REGION Network 42: Step [1102] : JOB[11] Check QR & Vision before move
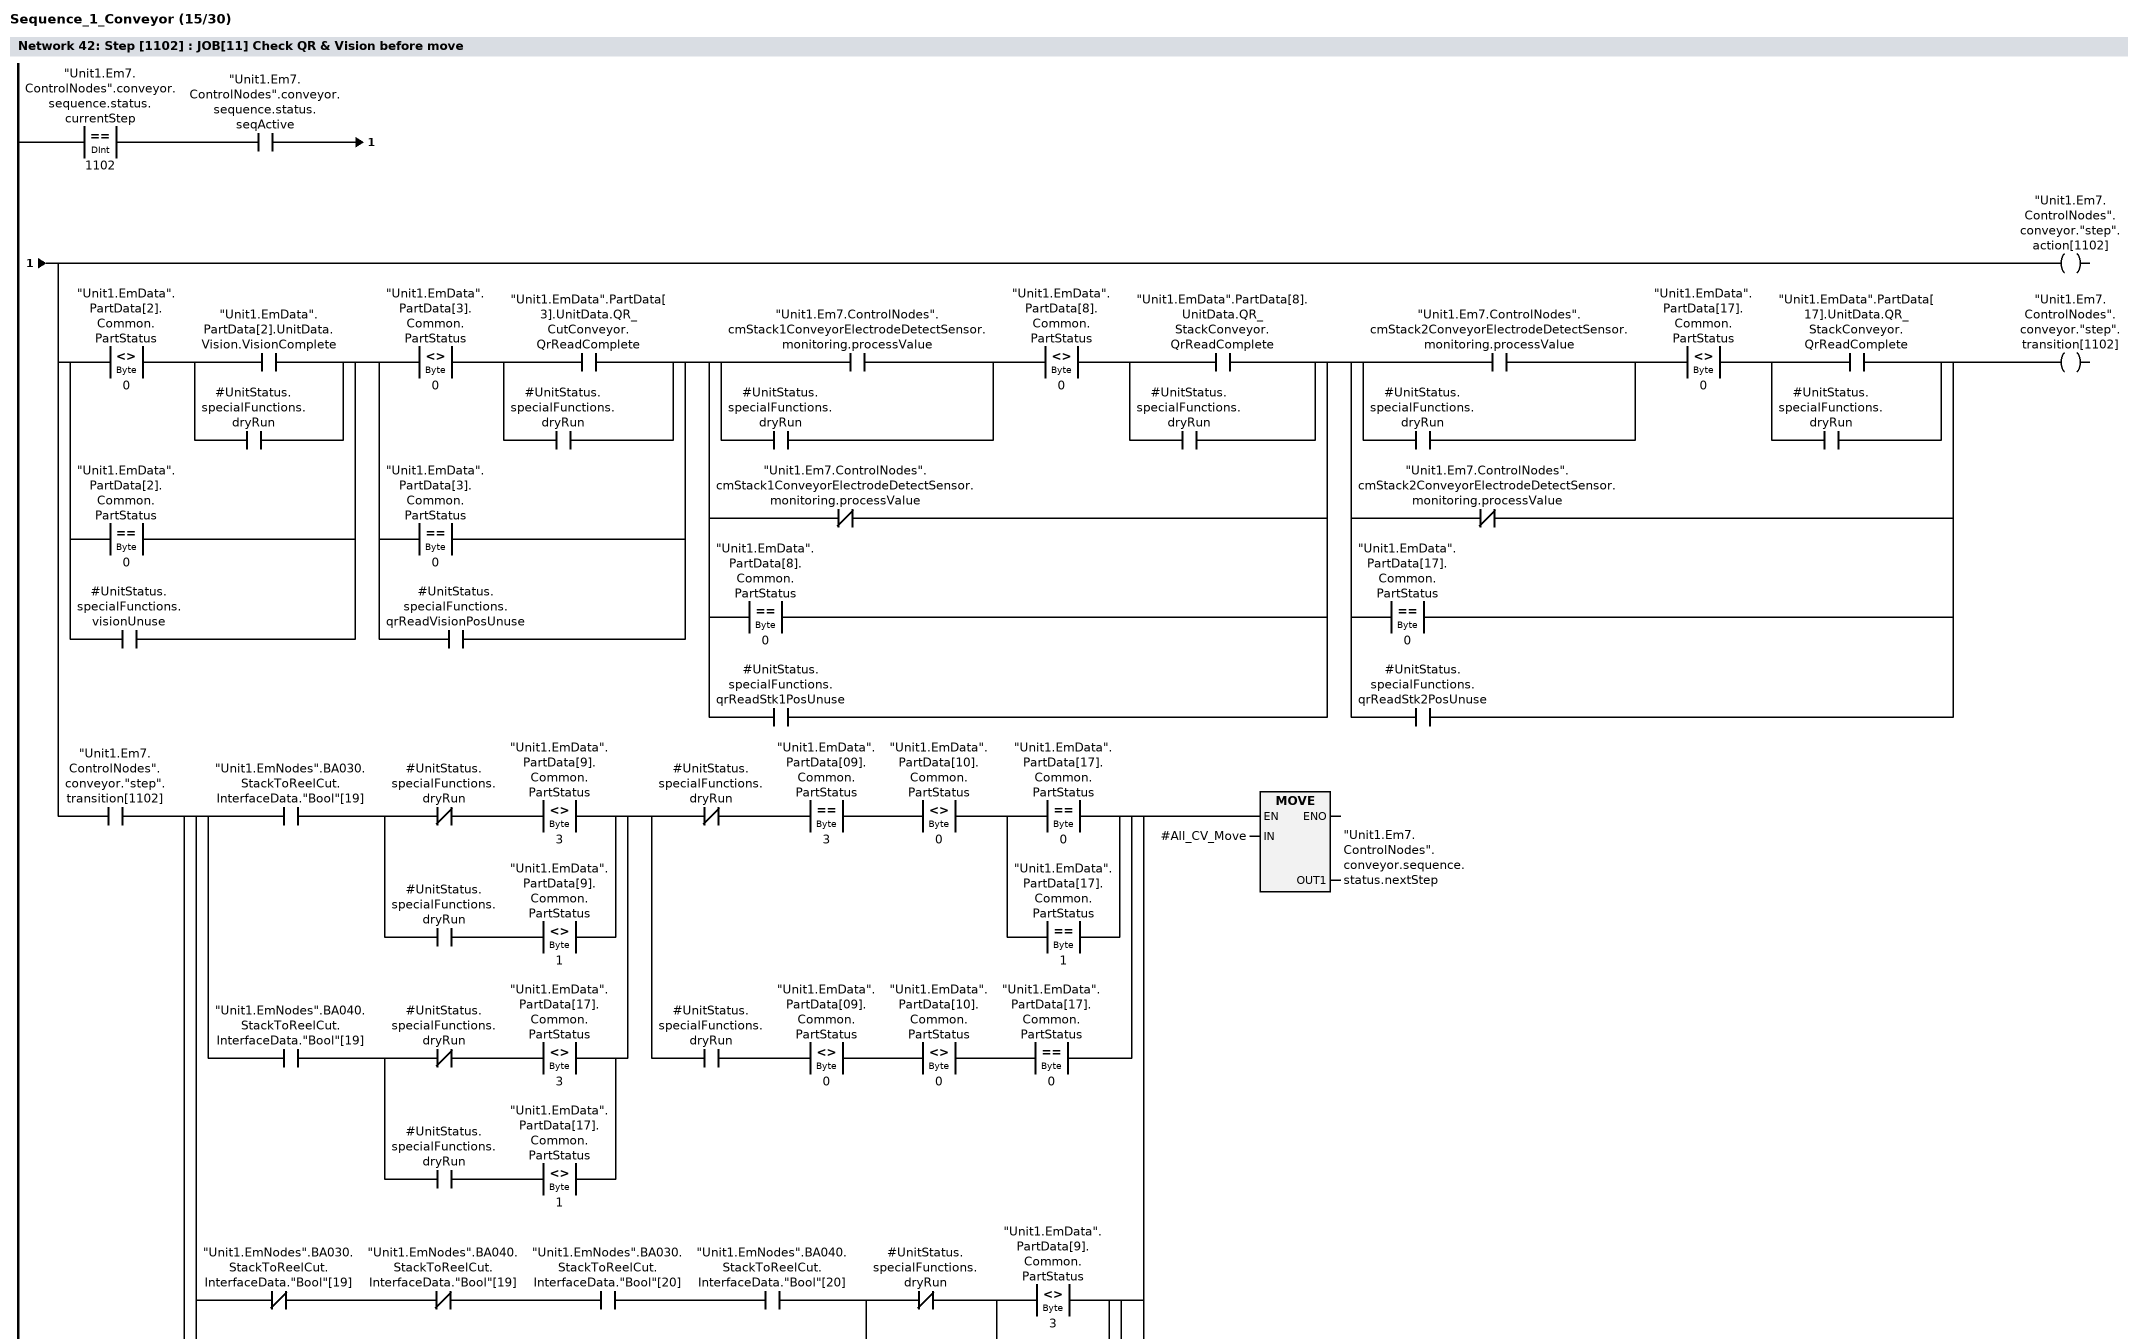
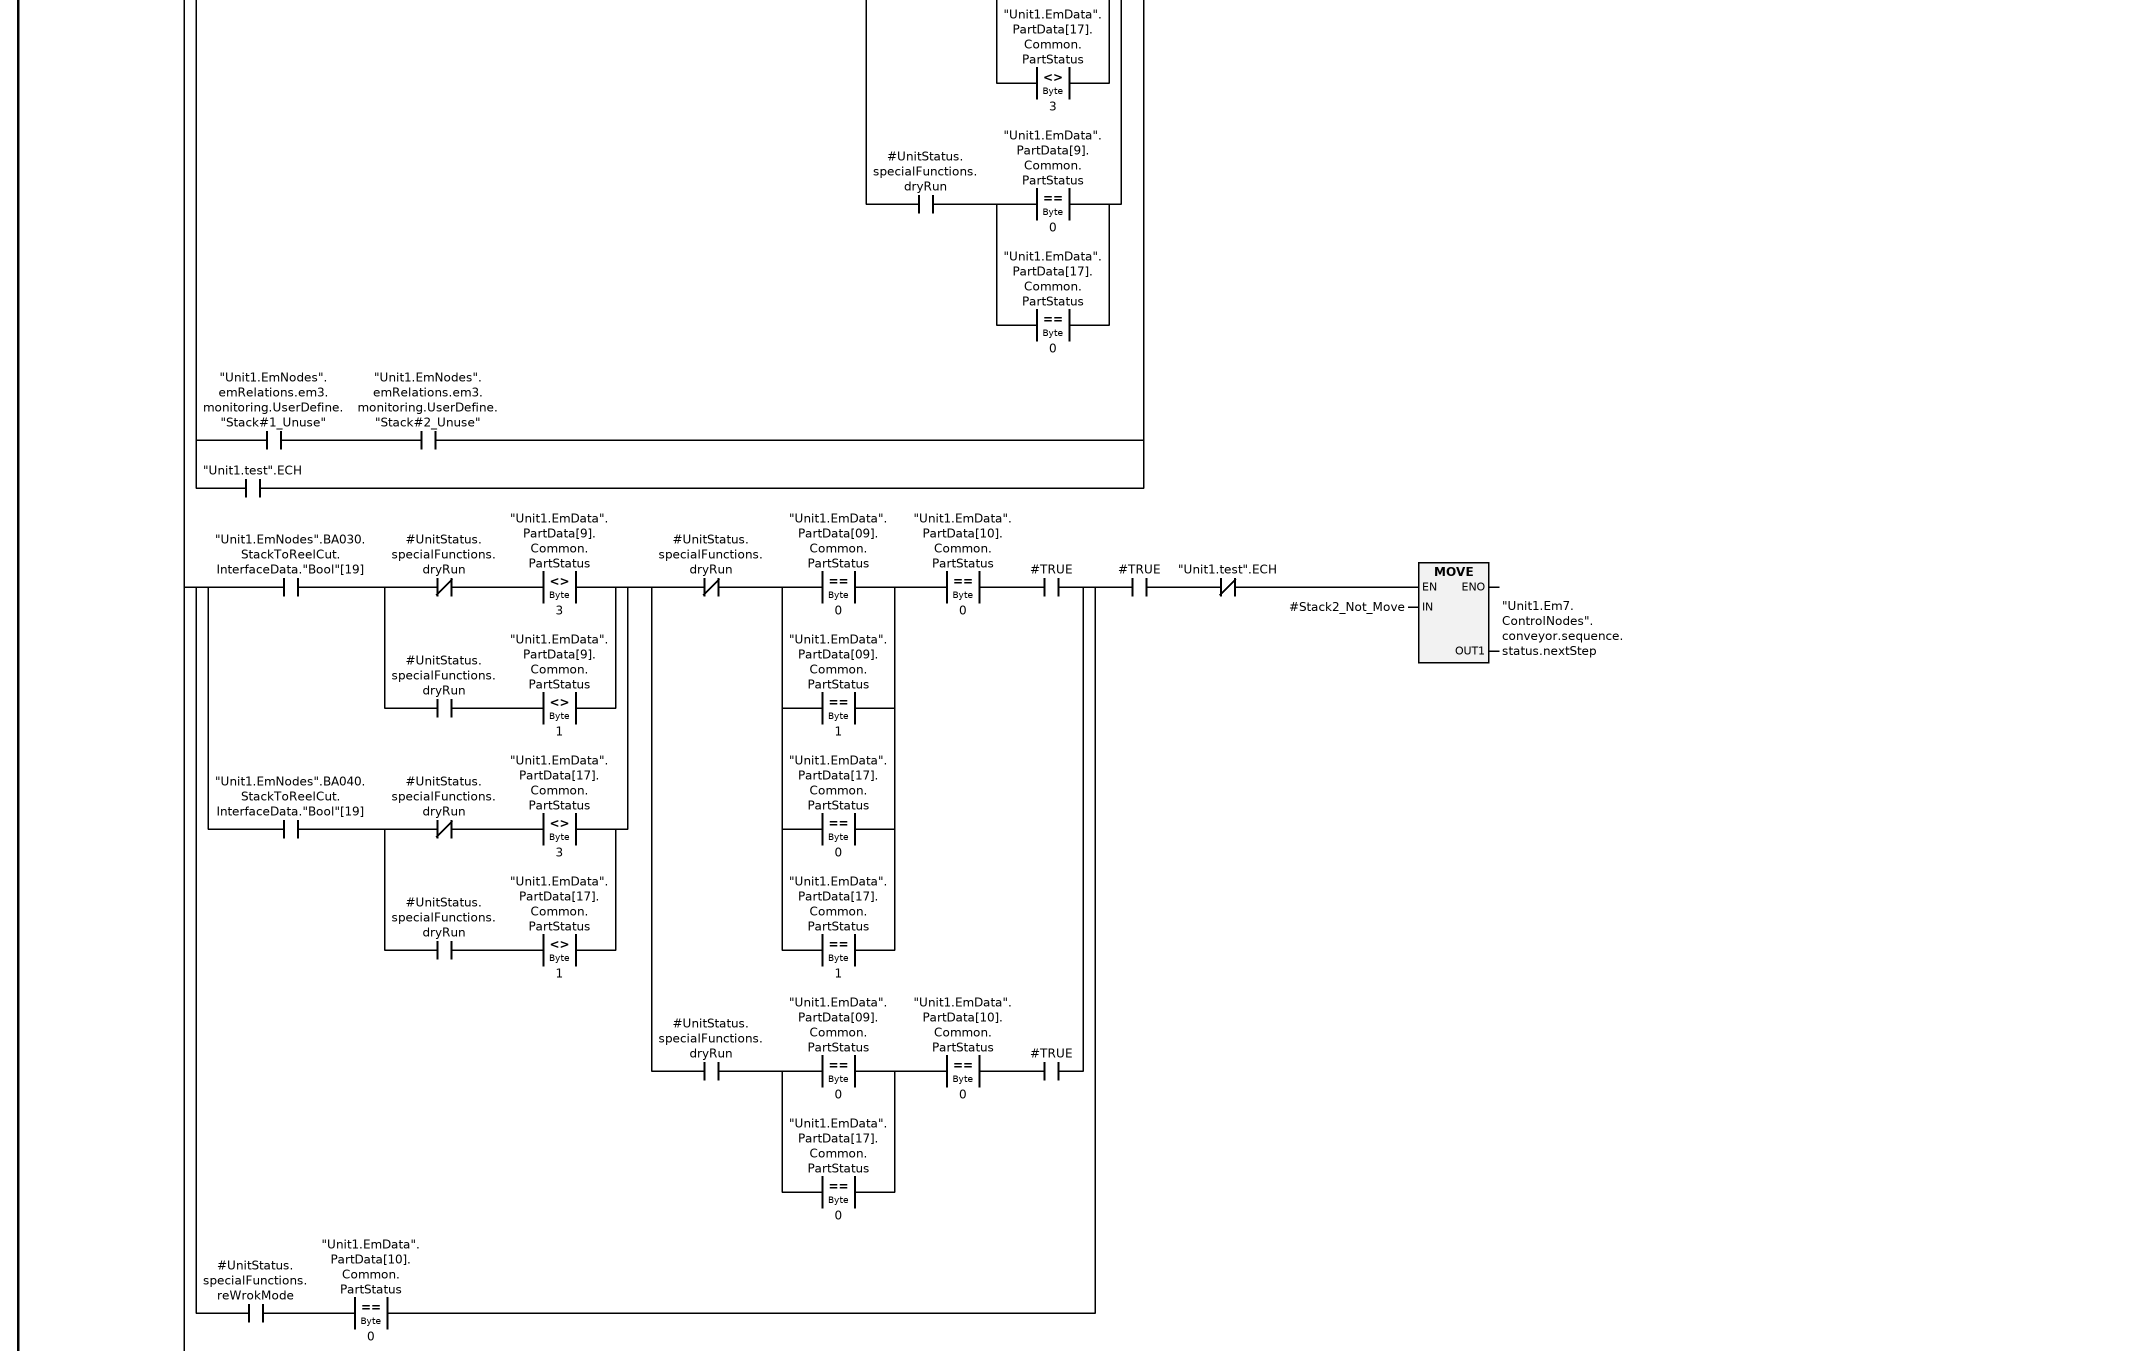
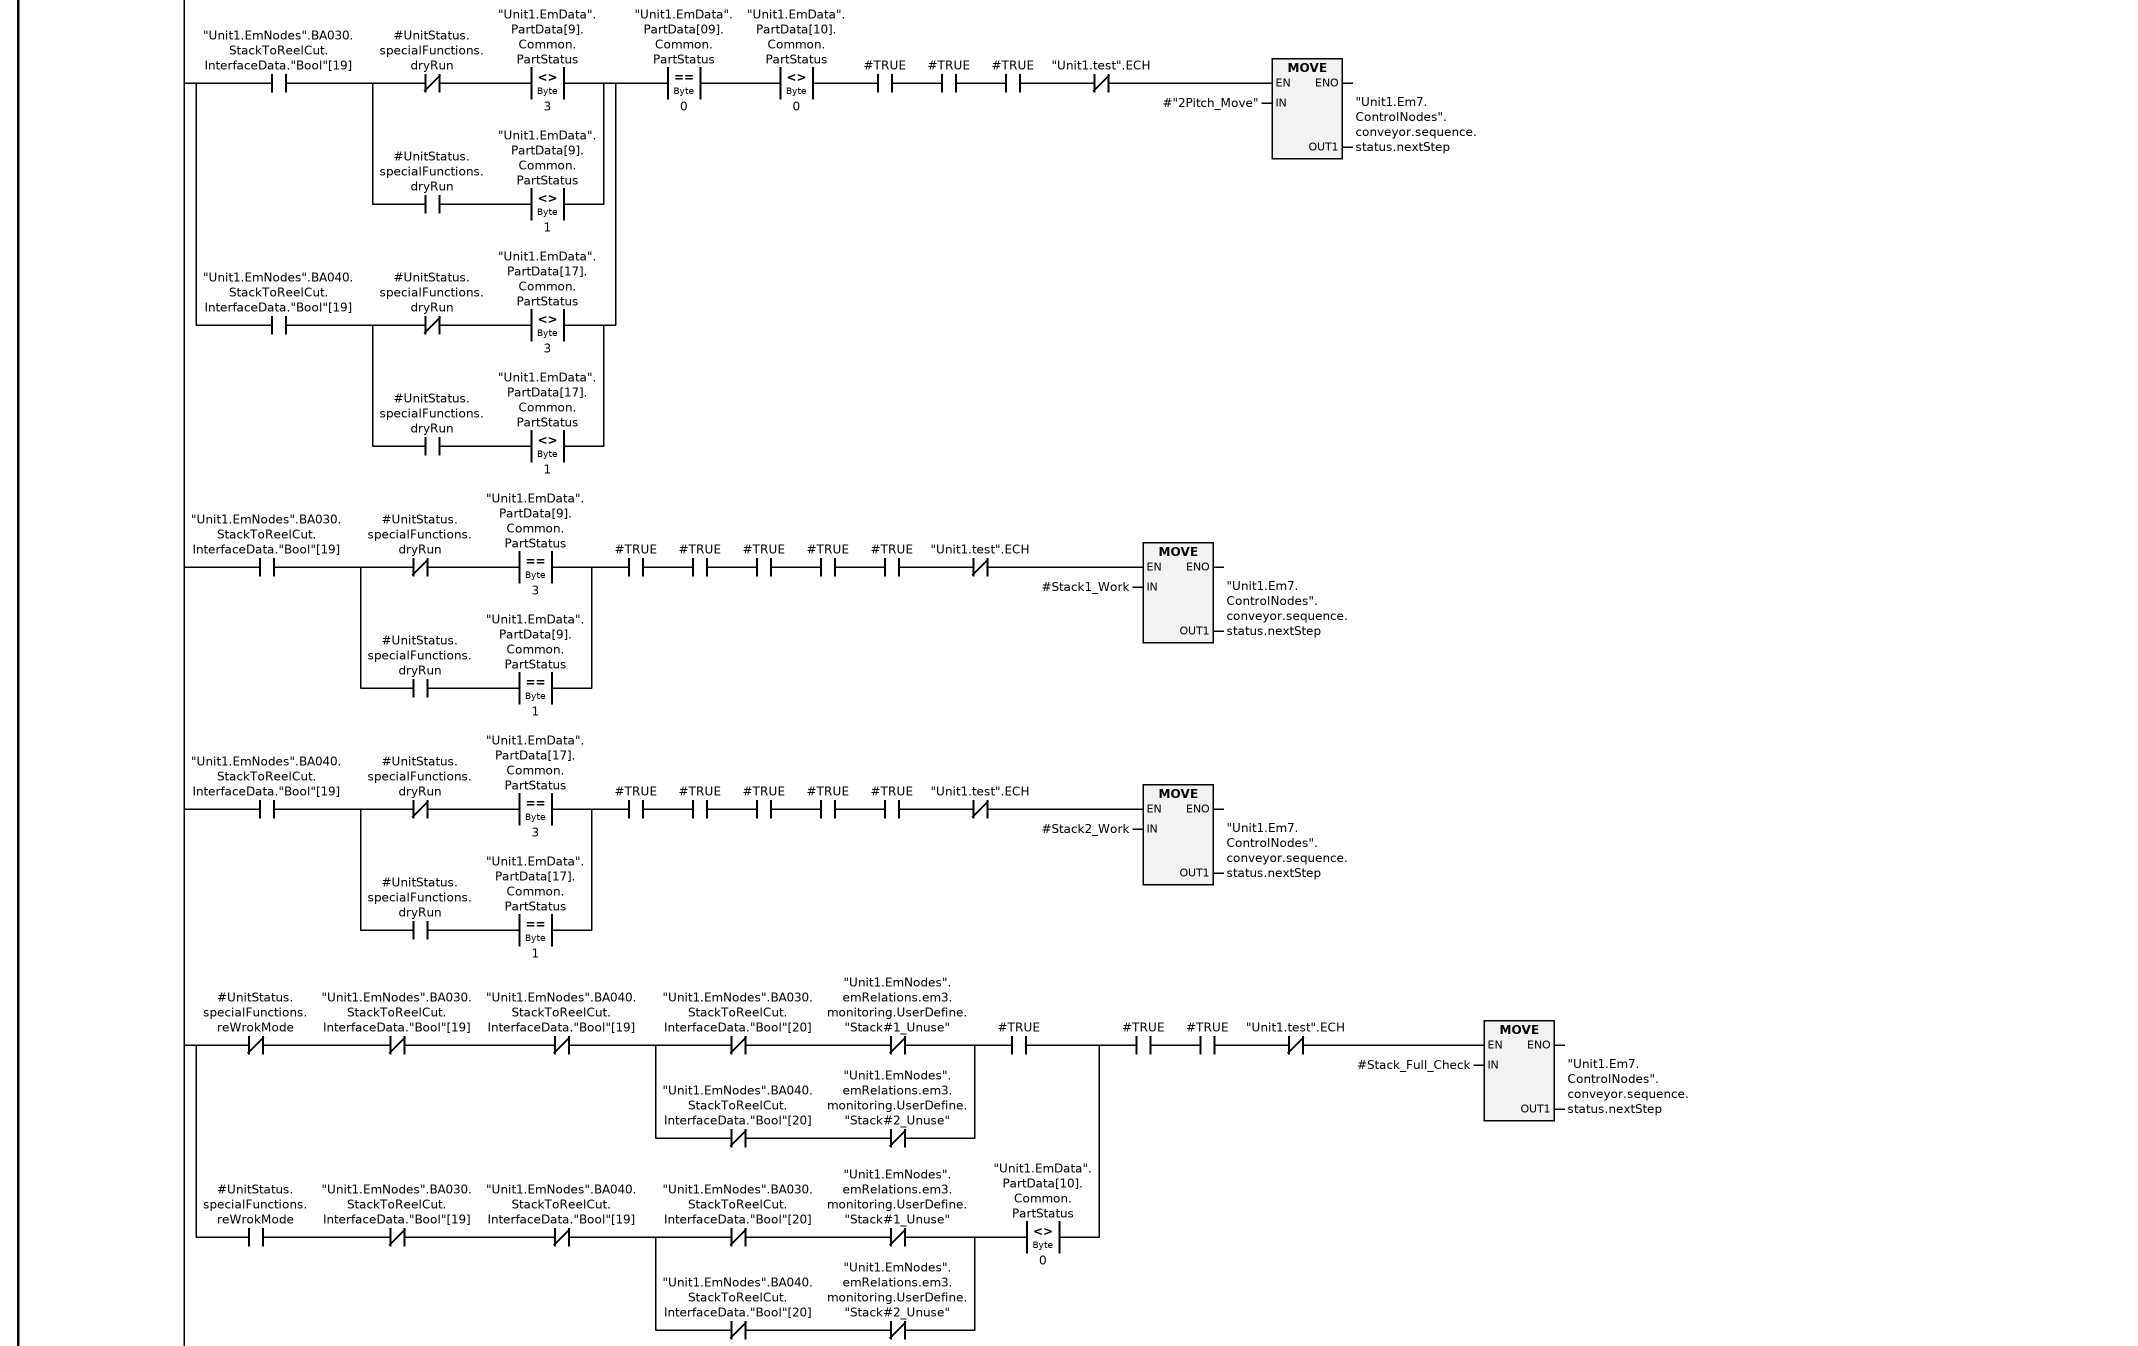
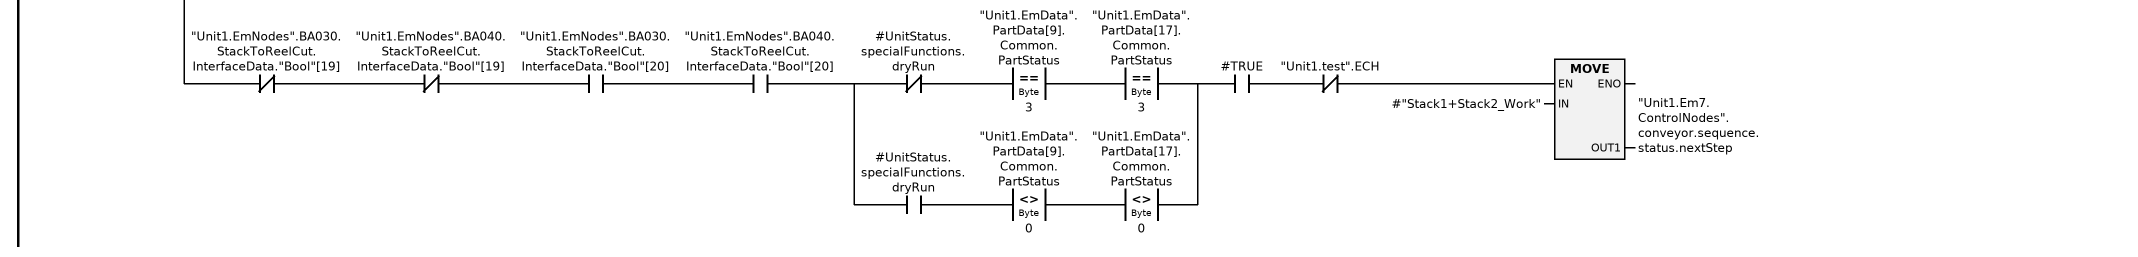
   RUNG wire#powerrail
      { S7_Templates := "SrcType := DInt" } EQ_Contact(in1 := "Unit1.Em7.ControlNodes".conveyor.sequence.status.currentStep, in2 := 1102)
      Contact( "Unit1.Em7.ControlNodes".conveyor.sequence.status.seqActive )
      wire#w1
      Coil( "Unit1.Em7.ControlNodes".conveyor."step".action[1102] )
   END_RUNG
   RUNG wire#w1
      { S7_Templates := "SrcType := Byte" } NE_Contact(in1 := "Unit1.EmData".PartData[2].Common.PartStatus, in2 := 0)
      wire#w2
      Contact( "Unit1.EmData".PartData[2].UnitData.Vision.VisionComplete )
      wire#w3
      { S7_Templates := "SrcType := Byte" } NE_Contact(in1 := "Unit1.EmData".PartData[3].Common.PartStatus, in2 := 0)
      wire#w4
      Contact( "Unit1.EmData".PartData[3].UnitData.QR_CutConveyor.QrReadComplete )
      wire#w5
      Contact( "Unit1.Em7.ControlNodes".cmStack1ConveyorElectrodeDetectSensor.monitoring.processValue )
      wire#w6
      { S7_Templates := "SrcType := Byte" } NE_Contact(in1 := "Unit1.EmData".PartData[8].Common.PartStatus, in2 := 0)
      wire#w7
      Contact( "Unit1.EmData".PartData[8].UnitData.QR_StackConveyor.QrReadComplete )
      wire#w8
      Contact( "Unit1.Em7.ControlNodes".cmStack2ConveyorElectrodeDetectSensor.monitoring.processValue )
      wire#w9
      { S7_Templates := "SrcType := Byte" } NE_Contact(in1 := "Unit1.EmData".PartData[17].Common.PartStatus, in2 := 0)
      wire#w10
      Contact( "Unit1.EmData".PartData[17].UnitData.QR_StackConveyor.QrReadComplete )
      wire#w11
      Coil( "Unit1.Em7.ControlNodes".conveyor."step".transition[1102] )
   END_RUNG
   RUNG wire#w2
      Contact( #UnitStatus.specialFunctions.dryRun )
   END_RUNG wire#w3
   RUNG wire#w1
      { S7_Templates := "SrcType := Byte" } EQ_Contact(in1 := "Unit1.EmData".PartData[2].Common.PartStatus, in2 := 0)
   END_RUNG wire#w3
   RUNG wire#w1
      Contact( #UnitStatus.specialFunctions.visionUnuse )
   END_RUNG wire#w3
   RUNG wire#w4
      Contact( #UnitStatus.specialFunctions.dryRun )
   END_RUNG wire#w5
   RUNG wire#w3
      { S7_Templates := "SrcType := Byte" } EQ_Contact(in1 := "Unit1.EmData".PartData[3].Common.PartStatus, in2 := 0)
   END_RUNG wire#w5
   RUNG wire#w3
      Contact( #UnitStatus.specialFunctions.qrReadVisionPosUnuse )
   END_RUNG wire#w5
   RUNG wire#w5
      Contact( #UnitStatus.specialFunctions.dryRun )
   END_RUNG wire#w6
   RUNG wire#w7
      Contact( #UnitStatus.specialFunctions.dryRun )
   END_RUNG wire#w8
   RUNG wire#w5
      I_Contact( "Unit1.Em7.ControlNodes".cmStack1ConveyorElectrodeDetectSensor.monitoring.processValue )
   END_RUNG wire#w8
   RUNG wire#w5
      { S7_Templates := "SrcType := Byte" } EQ_Contact(in1 := "Unit1.EmData".PartData[8].Common.PartStatus, in2 := 0)
   END_RUNG wire#w8
   RUNG wire#w5
      Contact( #UnitStatus.specialFunctions.qrReadStk1PosUnuse )
   END_RUNG wire#w8
   RUNG wire#w8
      Contact( #UnitStatus.specialFunctions.dryRun )
   END_RUNG wire#w9
   RUNG wire#w10
      Contact( #UnitStatus.specialFunctions.dryRun )
   END_RUNG wire#w11
   RUNG wire#w8
      I_Contact( "Unit1.Em7.ControlNodes".cmStack2ConveyorElectrodeDetectSensor.monitoring.processValue )
   END_RUNG wire#w11
   RUNG wire#w8
      { S7_Templates := "SrcType := Byte" } EQ_Contact(in1 := "Unit1.EmData".PartData[17].Common.PartStatus, in2 := 0)
   END_RUNG wire#w11
   RUNG wire#w8
      Contact( #UnitStatus.specialFunctions.qrReadStk2PosUnuse )
   END_RUNG wire#w11
   RUNG wire#w1
      Contact( "Unit1.Em7.ControlNodes".conveyor."step".transition[1102] )
      wire#w12
      Contact( "Unit1.EmNodes".BA030.StackToReelCut.InterfaceData."Bool"[19] )
      wire#w13
      I_Contact( #UnitStatus.specialFunctions.dryRun )
      { S7_Templates := "SrcType := Byte" } NE_Contact(in1 := "Unit1.EmData".PartData[9].Common.PartStatus, in2 := 3)
      wire#w14
      I_Contact( #UnitStatus.specialFunctions.dryRun )
      { S7_Templates := "SrcType := Byte" } EQ_Contact(in1 := "Unit1.EmData".PartData[09].Common.PartStatus, in2 := 3)
      { S7_Templates := "SrcType := Byte" } NE_Contact(in1 := "Unit1.EmData".PartData[10].Common.PartStatus, in2 := 0)
      wire#w16
      { S7_Templates := "SrcType := Byte" } EQ_Contact(in1 := "Unit1.EmData".PartData[17].Common.PartStatus, in2 := 0)
      wire#w17
      Move(in := #All_CV_Move, out1 => "Unit1.Em7.ControlNodes".conveyor.sequence.status.nextStep)
   END_RUNG
   RUNG wire#w13
      Contact( #UnitStatus.specialFunctions.dryRun )
      { S7_Templates := "SrcType := Byte" } NE_Contact(in1 := "Unit1.EmData".PartData[9].Common.PartStatus, in2 := 1)
   END_RUNG wire#w14
   RUNG wire#w12
      Contact( "Unit1.EmNodes".BA040.StackToReelCut.InterfaceData."Bool"[19] )
      wire#w15
      I_Contact( #UnitStatus.specialFunctions.dryRun )
      { S7_Templates := "SrcType := Byte" } NE_Contact(in1 := "Unit1.EmData".PartData[17].Common.PartStatus, in2 := 3)
   END_RUNG wire#w14
   RUNG wire#w15
      Contact( #UnitStatus.specialFunctions.dryRun )
      { S7_Templates := "SrcType := Byte" } NE_Contact(in1 := "Unit1.EmData".PartData[17].Common.PartStatus, in2 := 1)
   END_RUNG wire#w14
   RUNG wire#w16
      { S7_Templates := "SrcType := Byte" } EQ_Contact(in1 := "Unit1.EmData".PartData[17].Common.PartStatus, in2 := 1)
   END_RUNG wire#w17
   RUNG wire#w14
      Contact( #UnitStatus.specialFunctions.dryRun )
      { S7_Templates := "SrcType := Byte" } NE_Contact(in1 := "Unit1.EmData".PartData[09].Common.PartStatus, in2 := 0)
      { S7_Templates := "SrcType := Byte" } NE_Contact(in1 := "Unit1.EmData".PartData[10].Common.PartStatus, in2 := 0)
      { S7_Templates := "SrcType := Byte" } EQ_Contact(in1 := "Unit1.EmData".PartData[17].Common.PartStatus, in2 := 0)
   END_RUNG wire#w17
   RUNG wire#w12
      I_Contact( "Unit1.EmNodes".BA030.StackToReelCut.InterfaceData."Bool"[19] )
      I_Contact( "Unit1.EmNodes".BA040.StackToReelCut.InterfaceData."Bool"[19] )
      Contact( "Unit1.EmNodes".BA030.StackToReelCut.InterfaceData."Bool"[20] )
      Contact( "Unit1.EmNodes".BA040.StackToReelCut.InterfaceData."Bool"[20] )
      wire#w18
      I_Contact( #UnitStatus.specialFunctions.dryRun )
      wire#w19
      { S7_Templates := "SrcType := Byte" } NE_Contact(in1 := "Unit1.EmData".PartData[9].Common.PartStatus, in2 := 3)
   END_RUNG wire#w17
   RUNG wire#w19
      { S7_Templates := "SrcType := Byte" } NE_Contact(in1 := "Unit1.EmData".PartData[17].Common.PartStatus, in2 := 3)
   END_RUNG wire#w17
   RUNG wire#w18
      Contact( #UnitStatus.specialFunctions.dryRun )
      wire#w20
      { S7_Templates := "SrcType := Byte" } EQ_Contact(in1 := "Unit1.EmData".PartData[9].Common.PartStatus, in2 := 0)
   END_RUNG wire#w17
   RUNG wire#w20
      { S7_Templates := "SrcType := Byte" } EQ_Contact(in1 := "Unit1.EmData".PartData[17].Common.PartStatus, in2 := 0)
   END_RUNG wire#w17
   RUNG wire#w12
      Contact( "Unit1.EmNodes".emRelations.em3.monitoring.UserDefine."Stack#1_Unuse" )
      Contact( "Unit1.EmNodes".emRelations.em3.monitoring.UserDefine."Stack#2_Unuse" )
   END_RUNG wire#w17
   RUNG wire#w12
      Contact( "Unit1.test".ECH )
   END_RUNG wire#w17
   RUNG wire#w12
      Contact( "Unit1.EmNodes".BA030.StackToReelCut.InterfaceData."Bool"[19] )
      wire#w21
      I_Contact( #UnitStatus.specialFunctions.dryRun )
      { S7_Templates := "SrcType := Byte" } NE_Contact(in1 := "Unit1.EmData".PartData[9].Common.PartStatus, in2 := 3)
      wire#w22
      I_Contact( #UnitStatus.specialFunctions.dryRun )
      wire#w24
      { S7_Templates := "SrcType := Byte" } EQ_Contact(in1 := "Unit1.EmData".PartData[09].Common.PartStatus, in2 := 0)
      wire#w25
      { S7_Templates := "SrcType := Byte" } EQ_Contact(in1 := "Unit1.EmData".PartData[10].Common.PartStatus, in2 := 0)
      Contact( #TRUE )
      wire#w26
      Contact( #TRUE )
      I_Contact( "Unit1.test".ECH )
      Move(in := #Stack2_Not_Move, out1 => "Unit1.Em7.ControlNodes".conveyor.sequence.status.nextStep)
   END_RUNG
   RUNG wire#w21
      Contact( #UnitStatus.specialFunctions.dryRun )
      { S7_Templates := "SrcType := Byte" } NE_Contact(in1 := "Unit1.EmData".PartData[9].Common.PartStatus, in2 := 1)
   END_RUNG wire#w22
   RUNG wire#w12
      Contact( "Unit1.EmNodes".BA040.StackToReelCut.InterfaceData."Bool"[19] )
      wire#w23
      I_Contact( #UnitStatus.specialFunctions.dryRun )
      { S7_Templates := "SrcType := Byte" } NE_Contact(in1 := "Unit1.EmData".PartData[17].Common.PartStatus, in2 := 3)
   END_RUNG wire#w22
   RUNG wire#w23
      Contact( #UnitStatus.specialFunctions.dryRun )
      { S7_Templates := "SrcType := Byte" } NE_Contact(in1 := "Unit1.EmData".PartData[17].Common.PartStatus, in2 := 1)
   END_RUNG wire#w22
   RUNG wire#w24
      { S7_Templates := "SrcType := Byte" } EQ_Contact(in1 := "Unit1.EmData".PartData[09].Common.PartStatus, in2 := 1)
   END_RUNG wire#w25
   RUNG wire#w24
      { S7_Templates := "SrcType := Byte" } EQ_Contact(in1 := "Unit1.EmData".PartData[17].Common.PartStatus, in2 := 0)
   END_RUNG wire#w25
   RUNG wire#w24
      { S7_Templates := "SrcType := Byte" } EQ_Contact(in1 := "Unit1.EmData".PartData[17].Common.PartStatus, in2 := 1)
   END_RUNG wire#w25
   RUNG wire#w22
      Contact( #UnitStatus.specialFunctions.dryRun )
      wire#w27
      { S7_Templates := "SrcType := Byte" } EQ_Contact(in1 := "Unit1.EmData".PartData[09].Common.PartStatus, in2 := 0)
      wire#w28
      { S7_Templates := "SrcType := Byte" } EQ_Contact(in1 := "Unit1.EmData".PartData[10].Common.PartStatus, in2 := 0)
      Contact( #TRUE )
   END_RUNG wire#w26
   RUNG wire#w27
      { S7_Templates := "SrcType := Byte" } EQ_Contact(in1 := "Unit1.EmData".PartData[17].Common.PartStatus, in2 := 0)
   END_RUNG wire#w28
   RUNG wire#w12
      Contact( #UnitStatus.specialFunctions.reWrokMode )
      { S7_Templates := "SrcType := Byte" } EQ_Contact(in1 := "Unit1.EmData".PartData[10].Common.PartStatus, in2 := 0)
   END_RUNG wire#w26
   RUNG wire#w12
      Contact( "Unit1.EmNodes".BA030.StackToReelCut.InterfaceData."Bool"[19] )
      wire#w29
      I_Contact( #UnitStatus.specialFunctions.dryRun )
      { S7_Templates := "SrcType := Byte" } NE_Contact(in1 := "Unit1.EmData".PartData[9].Common.PartStatus, in2 := 3)
      wire#w30
      { S7_Templates := "SrcType := Byte" } EQ_Contact(in1 := "Unit1.EmData".PartData[09].Common.PartStatus, in2 := 0)
      { S7_Templates := "SrcType := Byte" } NE_Contact(in1 := "Unit1.EmData".PartData[10].Common.PartStatus, in2 := 0)
      Contact( #TRUE )
      Contact( #TRUE )
      Contact( #TRUE )
      I_Contact( "Unit1.test".ECH )
      Move(in := #"2Pitch_Move", out1 => "Unit1.Em7.ControlNodes".conveyor.sequence.status.nextStep)
   END_RUNG
   RUNG wire#w29
      Contact( #UnitStatus.specialFunctions.dryRun )
      { S7_Templates := "SrcType := Byte" } NE_Contact(in1 := "Unit1.EmData".PartData[9].Common.PartStatus, in2 := 1)
   END_RUNG wire#w30
   RUNG wire#w12
      Contact( "Unit1.EmNodes".BA040.StackToReelCut.InterfaceData."Bool"[19] )
      wire#w31
      I_Contact( #UnitStatus.specialFunctions.dryRun )
      { S7_Templates := "SrcType := Byte" } NE_Contact(in1 := "Unit1.EmData".PartData[17].Common.PartStatus, in2 := 3)
   END_RUNG wire#w30
   RUNG wire#w31
      Contact( #UnitStatus.specialFunctions.dryRun )
      { S7_Templates := "SrcType := Byte" } NE_Contact(in1 := "Unit1.EmData".PartData[17].Common.PartStatus, in2 := 1)
   END_RUNG wire#w30
   RUNG wire#w12
      Contact( "Unit1.EmNodes".BA030.StackToReelCut.InterfaceData."Bool"[19] )
      wire#w32
      I_Contact( #UnitStatus.specialFunctions.dryRun )
      { S7_Templates := "SrcType := Byte" } EQ_Contact(in1 := "Unit1.EmData".PartData[9].Common.PartStatus, in2 := 3)
      wire#w33
      Contact( #TRUE )
      Contact( #TRUE )
      Contact( #TRUE )
      Contact( #TRUE )
      Contact( #TRUE )
      I_Contact( "Unit1.test".ECH )
      Move(in := #Stack1_Work, out1 => "Unit1.Em7.ControlNodes".conveyor.sequence.status.nextStep)
   END_RUNG
   RUNG wire#w32
      Contact( #UnitStatus.specialFunctions.dryRun )
      { S7_Templates := "SrcType := Byte" } EQ_Contact(in1 := "Unit1.EmData".PartData[9].Common.PartStatus, in2 := 1)
   END_RUNG wire#w33
   RUNG wire#w12
      Contact( "Unit1.EmNodes".BA040.StackToReelCut.InterfaceData."Bool"[19] )
      wire#w34
      I_Contact( #UnitStatus.specialFunctions.dryRun )
      { S7_Templates := "SrcType := Byte" } EQ_Contact(in1 := "Unit1.EmData".PartData[17].Common.PartStatus, in2 := 3)
      wire#w35
      Contact( #TRUE )
      Contact( #TRUE )
      Contact( #TRUE )
      Contact( #TRUE )
      Contact( #TRUE )
      I_Contact( "Unit1.test".ECH )
      Move(in := #Stack2_Work, out1 => "Unit1.Em7.ControlNodes".conveyor.sequence.status.nextStep)
   END_RUNG
   RUNG wire#w34
      Contact( #UnitStatus.specialFunctions.dryRun )
      { S7_Templates := "SrcType := Byte" } EQ_Contact(in1 := "Unit1.EmData".PartData[17].Common.PartStatus, in2 := 1)
   END_RUNG wire#w35
   RUNG wire#w12
      I_Contact( #UnitStatus.specialFunctions.reWrokMode )
      I_Contact( "Unit1.EmNodes".BA030.StackToReelCut.InterfaceData."Bool"[19] )
      I_Contact( "Unit1.EmNodes".BA040.StackToReelCut.InterfaceData."Bool"[19] )
      wire#w36
      I_Contact( "Unit1.EmNodes".BA030.StackToReelCut.InterfaceData."Bool"[20] )
      I_Contact( "Unit1.EmNodes".emRelations.em3.monitoring.UserDefine."Stack#1_Unuse" )
      wire#w37
      Contact( #TRUE )
      wire#w38
      Contact( #TRUE )
      Contact( #TRUE )
      I_Contact( "Unit1.test".ECH )
      Move(in := #Stack_Full_Check, out1 => "Unit1.Em7.ControlNodes".conveyor.sequence.status.nextStep)
   END_RUNG
   RUNG wire#w36
      I_Contact( "Unit1.EmNodes".BA040.StackToReelCut.InterfaceData."Bool"[20] )
      I_Contact( "Unit1.EmNodes".emRelations.em3.monitoring.UserDefine."Stack#2_Unuse" )
   END_RUNG wire#w37
   RUNG wire#w12
      Contact( #UnitStatus.specialFunctions.reWrokMode )
      I_Contact( "Unit1.EmNodes".BA030.StackToReelCut.InterfaceData."Bool"[19] )
      I_Contact( "Unit1.EmNodes".BA040.StackToReelCut.InterfaceData."Bool"[19] )
      wire#w39
      I_Contact( "Unit1.EmNodes".BA030.StackToReelCut.InterfaceData."Bool"[20] )
      I_Contact( "Unit1.EmNodes".emRelations.em3.monitoring.UserDefine."Stack#1_Unuse" )
      wire#w40
      { S7_Templates := "SrcType := Byte" } NE_Contact(in1 := "Unit1.EmData".PartData[10].Common.PartStatus, in2 := 0)
   END_RUNG wire#w38
   RUNG wire#w39
      I_Contact( "Unit1.EmNodes".BA040.StackToReelCut.InterfaceData."Bool"[20] )
      I_Contact( "Unit1.EmNodes".emRelations.em3.monitoring.UserDefine."Stack#2_Unuse" )
   END_RUNG wire#w40
   RUNG wire#w12
      I_Contact( "Unit1.EmNodes".BA030.StackToReelCut.InterfaceData."Bool"[19] )
      I_Contact( "Unit1.EmNodes".BA040.StackToReelCut.InterfaceData."Bool"[19] )
      Contact( "Unit1.EmNodes".BA030.StackToReelCut.InterfaceData."Bool"[20] )
      Contact( "Unit1.EmNodes".BA040.StackToReelCut.InterfaceData."Bool"[20] )
      wire#w41
      I_Contact( #UnitStatus.specialFunctions.dryRun )
      { S7_Templates := "SrcType := Byte" } EQ_Contact(in1 := "Unit1.EmData".PartData[9].Common.PartStatus, in2 := 3)
      { S7_Templates := "SrcType := Byte" } EQ_Contact(in1 := "Unit1.EmData".PartData[17].Common.PartStatus, in2 := 3)
      wire#w42
      Contact( #TRUE )
      I_Contact( "Unit1.test".ECH )
      Move(in := #"Stack1+Stack2_Work", out1 => "Unit1.Em7.ControlNodes".conveyor.sequence.status.nextStep)
   END_RUNG
   RUNG wire#w41
      Contact( #UnitStatus.specialFunctions.dryRun )
      { S7_Templates := "SrcType := Byte" } NE_Contact(in1 := "Unit1.EmData".PartData[9].Common.PartStatus, in2 := 0)
      { S7_Templates := "SrcType := Byte" } NE_Contact(in1 := "Unit1.EmData".PartData[17].Common.PartStatus, in2 := 0)
   END_RUNG wire#w42
   // the same network as SCL:
   "Unit1.Em7.ControlNodes".conveyor."step".action[1102] := ("Unit1.Em7.ControlNodes".conveyor.sequence.status.currentStep = 1102) AND "Unit1.Em7.ControlNodes".conveyor.sequence.status.seqActive;
   "Unit1.Em7.ControlNodes".conveyor."step".transition[1102] := ("Unit1.Em7.ControlNodes".conveyor.sequence.status.currentStep = 1102) AND "Unit1.Em7.ControlNodes".conveyor.sequence.status.seqActive AND ((("Unit1.EmData".PartData[2].Common.PartStatus <> 0) AND ("Unit1.EmData".PartData[2].UnitData.Vision.VisionComplete OR #UnitStatus.specialFunctions.dryRun)) OR ("Unit1.EmData".PartData[2].Common.PartStatus = 0) OR #UnitStatus.specialFunctions.visionUnuse) AND ((("Unit1.EmData".PartData[3].Common.PartStatus <> 0) AND ("Unit1.EmData".PartData[3].UnitData.QR_CutConveyor.QrReadComplete OR #UnitStatus.specialFunctions.dryRun)) OR ("Unit1.EmData".PartData[3].Common.PartStatus = 0) OR #UnitStatus.specialFunctions.qrReadVisionPosUnuse) AND ((("Unit1.Em7.ControlNodes".cmStack1ConveyorElectrodeDetectSensor.monitoring.processValue OR #UnitStatus.specialFunctions.dryRun) AND ("Unit1.EmData".PartData[8].Common.PartStatus <> 0) AND ("Unit1.EmData".PartData[8].UnitData.QR_StackConveyor.QrReadComplete OR #UnitStatus.specialFunctions.dryRun)) OR NOT "Unit1.Em7.ControlNodes".cmStack1ConveyorElectrodeDetectSensor.monitoring.processValue OR ("Unit1.EmData".PartData[8].Common.PartStatus = 0) OR #UnitStatus.specialFunctions.qrReadStk1PosUnuse) AND ((("Unit1.Em7.ControlNodes".cmStack2ConveyorElectrodeDetectSensor.monitoring.processValue OR #UnitStatus.specialFunctions.dryRun) AND ("Unit1.EmData".PartData[17].Common.PartStatus <> 0) AND ("Unit1.EmData".PartData[17].UnitData.QR_StackConveyor.QrReadComplete OR #UnitStatus.specialFunctions.dryRun)) OR NOT "Unit1.Em7.ControlNodes".cmStack2ConveyorElectrodeDetectSensor.monitoring.processValue OR ("Unit1.EmData".PartData[17].Common.PartStatus = 0) OR #UnitStatus.specialFunctions.qrReadStk2PosUnuse);
   #_w1 := ("Unit1.Em7.ControlNodes".conveyor.sequence.status.currentStep = 1102) AND "Unit1.Em7.ControlNodes".conveyor.sequence.status.seqActive AND "Unit1.Em7.ControlNodes".conveyor."step".transition[1102];
   IF #_w1 AND (((("Unit1.EmNodes".BA030.StackToReelCut.InterfaceData."Bool"[19] AND ((NOT #UnitStatus.specialFunctions.dryRun AND ("Unit1.EmData".PartData[9].Common.PartStatus <> 3)) OR (#UnitStatus.specialFunctions.dryRun AND ("Unit1.EmData".PartData[9].Common.PartStatus <> 1)))) OR ("Unit1.EmNodes".BA040.StackToReelCut.InterfaceData."Bool"[19] AND ((NOT #UnitStatus.specialFunctions.dryRun AND ("Unit1.EmData".PartData[17].Common.PartStatus <> 3)) OR (#UnitStatus.specialFunctions.dryRun AND ("Unit1.EmData".PartData[17].Common.PartStatus <> 1))))) AND ((NOT #UnitStatus.specialFunctions.dryRun AND ("Unit1.EmData".PartData[09].Common.PartStatus = 3) AND ("Unit1.EmData".PartData[10].Common.PartStatus <> 0) AND (("Unit1.EmData".PartData[17].Common.PartStatus = 0) OR ("Unit1.EmData".PartData[17].Common.PartStatus = 1))) OR (#UnitStatus.specialFunctions.dryRun AND ("Unit1.EmData".PartData[09].Common.PartStatus <> 0) AND ("Unit1.EmData".PartData[10].Common.PartStatus <> 0) AND ("Unit1.EmData".PartData[17].Common.PartStatus = 0)))) OR (NOT "Unit1.EmNodes".BA030.StackToReelCut.InterfaceData."Bool"[19] AND NOT "Unit1.EmNodes".BA040.StackToReelCut.InterfaceData."Bool"[19] AND "Unit1.EmNodes".BA030.StackToReelCut.InterfaceData."Bool"[20] AND "Unit1.EmNodes".BA040.StackToReelCut.InterfaceData."Bool"[20] AND ((NOT #UnitStatus.specialFunctions.dryRun AND (("Unit1.EmData".PartData[9].Common.PartStatus <> 3) OR ("Unit1.EmData".PartData[17].Common.PartStatus <> 3))) OR (#UnitStatus.specialFunctions.dryRun AND (("Unit1.EmData".PartData[9].Common.PartStatus = 0) OR ("Unit1.EmData".PartData[17].Common.PartStatus = 0))))) OR ("Unit1.EmNodes".emRelations.em3.monitoring.UserDefine."Stack#1_Unuse" AND "Unit1.EmNodes".emRelations.em3.monitoring.UserDefine."Stack#2_Unuse") OR "Unit1.test".ECH) THEN
       "Unit1.Em7.ControlNodes".conveyor.sequence.status.nextStep := #All_CV_Move;
   END_IF;
   IF #_w1 AND (((("Unit1.EmNodes".BA030.StackToReelCut.InterfaceData."Bool"[19] AND ((NOT #UnitStatus.specialFunctions.dryRun AND ("Unit1.EmData".PartData[9].Common.PartStatus <> 3)) OR (#UnitStatus.specialFunctions.dryRun AND ("Unit1.EmData".PartData[9].Common.PartStatus <> 1)))) OR ("Unit1.EmNodes".BA040.StackToReelCut.InterfaceData."Bool"[19] AND ((NOT #UnitStatus.specialFunctions.dryRun AND ("Unit1.EmData".PartData[17].Common.PartStatus <> 3)) OR (#UnitStatus.specialFunctions.dryRun AND ("Unit1.EmData".PartData[17].Common.PartStatus <> 1))))) AND ((NOT #UnitStatus.specialFunctions.dryRun AND (("Unit1.EmData".PartData[09].Common.PartStatus = 0) OR ("Unit1.EmData".PartData[09].Common.PartStatus = 1) OR ("Unit1.EmData".PartData[17].Common.PartStatus = 0) OR ("Unit1.EmData".PartData[17].Common.PartStatus = 1)) AND ("Unit1.EmData".PartData[10].Common.PartStatus = 0) AND #TRUE) OR (#UnitStatus.specialFunctions.dryRun AND (("Unit1.EmData".PartData[09].Common.PartStatus = 0) OR ("Unit1.EmData".PartData[17].Common.PartStatus = 0)) AND ("Unit1.EmData".PartData[10].Common.PartStatus = 0) AND #TRUE))) OR (#UnitStatus.specialFunctions.reWrokMode AND ("Unit1.EmData".PartData[10].Common.PartStatus = 0))) AND #TRUE AND NOT "Unit1.test".ECH THEN
       "Unit1.Em7.ControlNodes".conveyor.sequence.status.nextStep := #Stack2_Not_Move;
   END_IF;
   IF #_w1 AND (("Unit1.EmNodes".BA030.StackToReelCut.InterfaceData."Bool"[19] AND ((NOT #UnitStatus.specialFunctions.dryRun AND ("Unit1.EmData".PartData[9].Common.PartStatus <> 3)) OR (#UnitStatus.specialFunctions.dryRun AND ("Unit1.EmData".PartData[9].Common.PartStatus <> 1)))) OR ("Unit1.EmNodes".BA040.StackToReelCut.InterfaceData."Bool"[19] AND ((NOT #UnitStatus.specialFunctions.dryRun AND ("Unit1.EmData".PartData[17].Common.PartStatus <> 3)) OR (#UnitStatus.specialFunctions.dryRun AND ("Unit1.EmData".PartData[17].Common.PartStatus <> 1))))) AND ("Unit1.EmData".PartData[09].Common.PartStatus = 0) AND ("Unit1.EmData".PartData[10].Common.PartStatus <> 0) AND #TRUE AND #TRUE AND #TRUE AND NOT "Unit1.test".ECH THEN
       "Unit1.Em7.ControlNodes".conveyor.sequence.status.nextStep := #"2Pitch_Move";
   END_IF;
   IF #_w1 AND "Unit1.EmNodes".BA030.StackToReelCut.InterfaceData."Bool"[19] AND ((NOT #UnitStatus.specialFunctions.dryRun AND ("Unit1.EmData".PartData[9].Common.PartStatus = 3)) OR (#UnitStatus.specialFunctions.dryRun AND ("Unit1.EmData".PartData[9].Common.PartStatus = 1))) AND #TRUE AND #TRUE AND #TRUE AND #TRUE AND #TRUE AND NOT "Unit1.test".ECH THEN
       "Unit1.Em7.ControlNodes".conveyor.sequence.status.nextStep := #Stack1_Work;
   END_IF;
   IF #_w1 AND "Unit1.EmNodes".BA040.StackToReelCut.InterfaceData."Bool"[19] AND ((NOT #UnitStatus.specialFunctions.dryRun AND ("Unit1.EmData".PartData[17].Common.PartStatus = 3)) OR (#UnitStatus.specialFunctions.dryRun AND ("Unit1.EmData".PartData[17].Common.PartStatus = 1))) AND #TRUE AND #TRUE AND #TRUE AND #TRUE AND #TRUE AND NOT "Unit1.test".ECH THEN
       "Unit1.Em7.ControlNodes".conveyor.sequence.status.nextStep := #Stack2_Work;
   END_IF;
   IF #_w1 AND ((NOT #UnitStatus.specialFunctions.reWrokMode AND NOT "Unit1.EmNodes".BA030.StackToReelCut.InterfaceData."Bool"[19] AND NOT "Unit1.EmNodes".BA040.StackToReelCut.InterfaceData."Bool"[19] AND ((NOT "Unit1.EmNodes".BA030.StackToReelCut.InterfaceData."Bool"[20] AND NOT "Unit1.EmNodes".emRelations.em3.monitoring.UserDefine."Stack#1_Unuse") OR (NOT "Unit1.EmNodes".BA040.StackToReelCut.InterfaceData."Bool"[20] AND NOT "Unit1.EmNodes".emRelations.em3.monitoring.UserDefine."Stack#2_Unuse")) AND #TRUE) OR (#UnitStatus.specialFunctions.reWrokMode AND NOT "Unit1.EmNodes".BA030.StackToReelCut.InterfaceData."Bool"[19] AND NOT "Unit1.EmNodes".BA040.StackToReelCut.InterfaceData."Bool"[19] AND ((NOT "Unit1.EmNodes".BA030.StackToReelCut.InterfaceData."Bool"[20] AND NOT "Unit1.EmNodes".emRelations.em3.monitoring.UserDefine."Stack#1_Unuse") OR (NOT "Unit1.EmNodes".BA040.StackToReelCut.InterfaceData."Bool"[20] AND NOT "Unit1.EmNodes".emRelations.em3.monitoring.UserDefine."Stack#2_Unuse")) AND ("Unit1.EmData".PartData[10].Common.PartStatus <> 0))) AND #TRUE AND #TRUE AND NOT "Unit1.test".ECH THEN
       "Unit1.Em7.ControlNodes".conveyor.sequence.status.nextStep := #Stack_Full_Check;
   END_IF;
   IF #_w1 AND NOT "Unit1.EmNodes".BA030.StackToReelCut.InterfaceData."Bool"[19] AND NOT "Unit1.EmNodes".BA040.StackToReelCut.InterfaceData."Bool"[19] AND "Unit1.EmNodes".BA030.StackToReelCut.InterfaceData."Bool"[20] AND "Unit1.EmNodes".BA040.StackToReelCut.InterfaceData."Bool"[20] AND ((NOT #UnitStatus.specialFunctions.dryRun AND ("Unit1.EmData".PartData[9].Common.PartStatus = 3) AND ("Unit1.EmData".PartData[17].Common.PartStatus = 3)) OR (#UnitStatus.specialFunctions.dryRun AND ("Unit1.EmData".PartData[9].Common.PartStatus <> 0) AND ("Unit1.EmData".PartData[17].Common.PartStatus <> 0))) AND #TRUE AND NOT "Unit1.test".ECH THEN
       "Unit1.Em7.ControlNodes".conveyor.sequence.status.nextStep := #"Stack1+Stack2_Work";
   END_IF;
END_REGION

REGION Network 43: Step [1103] : JOB[11] All C/V Move One Pitch Feeding
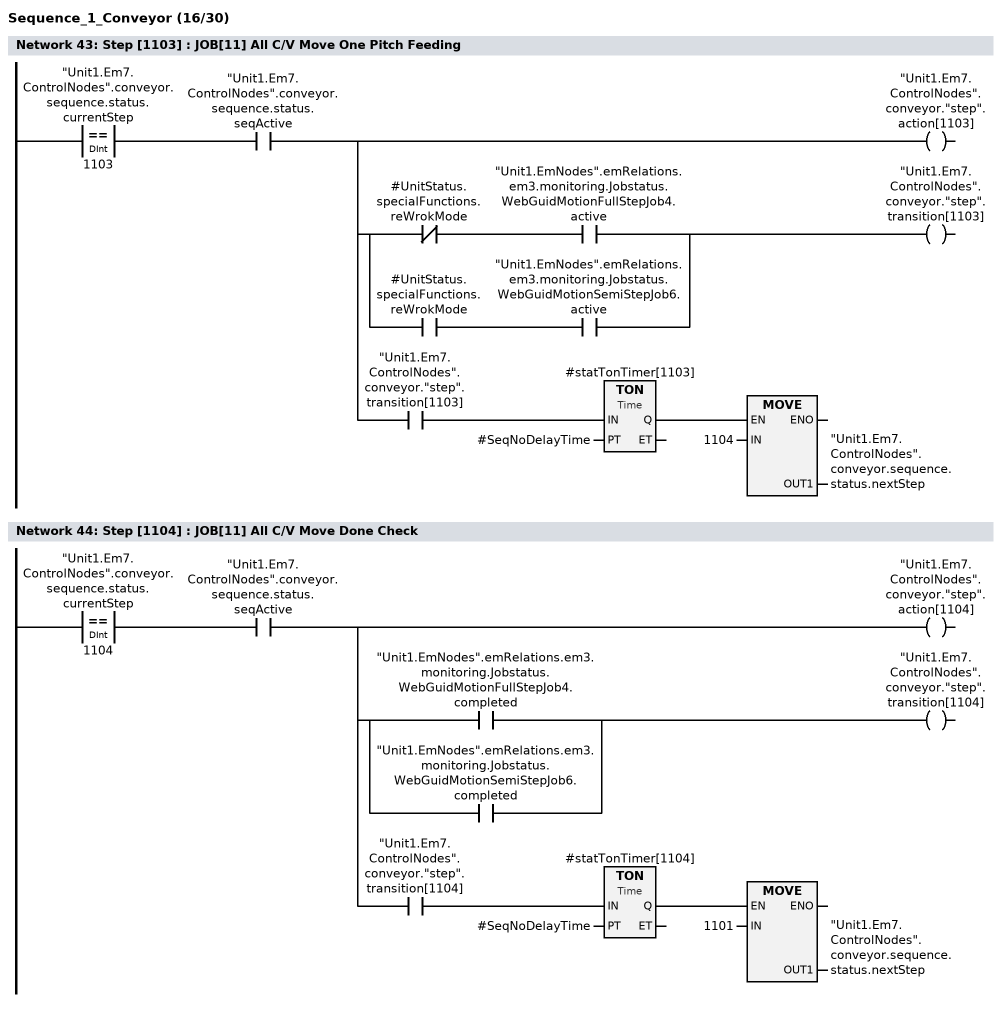
   RUNG wire#powerrail
      { S7_Templates := "SrcType := DInt" } EQ_Contact(in1 := "Unit1.Em7.ControlNodes".conveyor.sequence.status.currentStep, in2 := 1103)
      Contact( "Unit1.Em7.ControlNodes".conveyor.sequence.status.seqActive )
      wire#w1
      Coil( "Unit1.Em7.ControlNodes".conveyor."step".action[1103] )
   END_RUNG
   RUNG wire#w1
      I_Contact( #UnitStatus.specialFunctions.reWrokMode )
      Contact( "Unit1.EmNodes".emRelations.em3.monitoring.Jobstatus.WebGuidMotionFullStepJob4.active )
      wire#w2
      Coil( "Unit1.Em7.ControlNodes".conveyor."step".transition[1103] )
   END_RUNG
   RUNG wire#w1
      Contact( #UnitStatus.specialFunctions.reWrokMode )
      Contact( "Unit1.EmNodes".emRelations.em3.monitoring.Jobstatus.WebGuidMotionSemiStepJob6.active )
   END_RUNG wire#w2
   RUNG wire#w1
      Contact( "Unit1.Em7.ControlNodes".conveyor."step".transition[1103] )
      { S7_Templates := "time_type := Time" } #statTonTimer[1103].TON(pt := #SeqNoDelayTime, et =>)
      Move(in := 1104, out1 => "Unit1.Em7.ControlNodes".conveyor.sequence.status.nextStep)
   END_RUNG
   // the same network as SCL:
   "Unit1.Em7.ControlNodes".conveyor."step".action[1103] := ("Unit1.Em7.ControlNodes".conveyor.sequence.status.currentStep = 1103) AND "Unit1.Em7.ControlNodes".conveyor.sequence.status.seqActive;
   "Unit1.Em7.ControlNodes".conveyor."step".transition[1103] := ("Unit1.Em7.ControlNodes".conveyor.sequence.status.currentStep = 1103) AND "Unit1.Em7.ControlNodes".conveyor.sequence.status.seqActive AND ((NOT #UnitStatus.specialFunctions.reWrokMode AND "Unit1.EmNodes".emRelations.em3.monitoring.Jobstatus.WebGuidMotionFullStepJob4.active) OR (#UnitStatus.specialFunctions.reWrokMode AND "Unit1.EmNodes".emRelations.em3.monitoring.Jobstatus.WebGuidMotionSemiStepJob6.active));
   #statTonTimer[1103].TON(IN := ("Unit1.Em7.ControlNodes".conveyor.sequence.status.currentStep = 1103) AND "Unit1.Em7.ControlNodes".conveyor.sequence.status.seqActive AND "Unit1.Em7.ControlNodes".conveyor."step".transition[1103],
                           PT := #SeqNoDelayTime);
   IF #statTonTimer[1103].Q THEN "Unit1.Em7.ControlNodes".conveyor.sequence.status.nextStep := 1104; END_IF;
END_REGION

REGION Network 44: Step [1104] : JOB[11] All C/V Move Done Check
   RUNG wire#powerrail
      { S7_Templates := "SrcType := DInt" } EQ_Contact(in1 := "Unit1.Em7.ControlNodes".conveyor.sequence.status.currentStep, in2 := 1104)
      Contact( "Unit1.Em7.ControlNodes".conveyor.sequence.status.seqActive )
      wire#w1
      Coil( "Unit1.Em7.ControlNodes".conveyor."step".action[1104] )
   END_RUNG
   RUNG wire#w1
      Contact( "Unit1.EmNodes".emRelations.em3.monitoring.Jobstatus.WebGuidMotionFullStepJob4.completed )
      wire#w2
      Coil( "Unit1.Em7.ControlNodes".conveyor."step".transition[1104] )
   END_RUNG
   RUNG wire#w1
      Contact( "Unit1.EmNodes".emRelations.em3.monitoring.Jobstatus.WebGuidMotionSemiStepJob6.completed )
   END_RUNG wire#w2
   RUNG wire#w1
      Contact( "Unit1.Em7.ControlNodes".conveyor."step".transition[1104] )
      { S7_Templates := "time_type := Time" } #statTonTimer[1104].TON(pt := #SeqNoDelayTime, et =>)
      Move(in := 1101, out1 => "Unit1.Em7.ControlNodes".conveyor.sequence.status.nextStep)
   END_RUNG
   // the same network as SCL:
   "Unit1.Em7.ControlNodes".conveyor."step".action[1104] := ("Unit1.Em7.ControlNodes".conveyor.sequence.status.currentStep = 1104) AND "Unit1.Em7.ControlNodes".conveyor.sequence.status.seqActive;
   "Unit1.Em7.ControlNodes".conveyor."step".transition[1104] := ("Unit1.Em7.ControlNodes".conveyor.sequence.status.currentStep = 1104) AND "Unit1.Em7.ControlNodes".conveyor.sequence.status.seqActive AND ("Unit1.EmNodes".emRelations.em3.monitoring.Jobstatus.WebGuidMotionFullStepJob4.completed OR "Unit1.EmNodes".emRelations.em3.monitoring.Jobstatus.WebGuidMotionSemiStepJob6.completed);
   #statTonTimer[1104].TON(IN := ("Unit1.Em7.ControlNodes".conveyor.sequence.status.currentStep = 1104) AND "Unit1.Em7.ControlNodes".conveyor.sequence.status.seqActive AND "Unit1.Em7.ControlNodes".conveyor."step".transition[1104],
                           PT := #SeqNoDelayTime);
   IF #statTonTimer[1104].Q THEN "Unit1.Em7.ControlNodes".conveyor.sequence.status.nextStep := 1101; END_IF;
END_REGION

REGION Network 45: Step [1105] : JOB[11] Stack#2 C/V Not move / The others C/V move 1 pitch
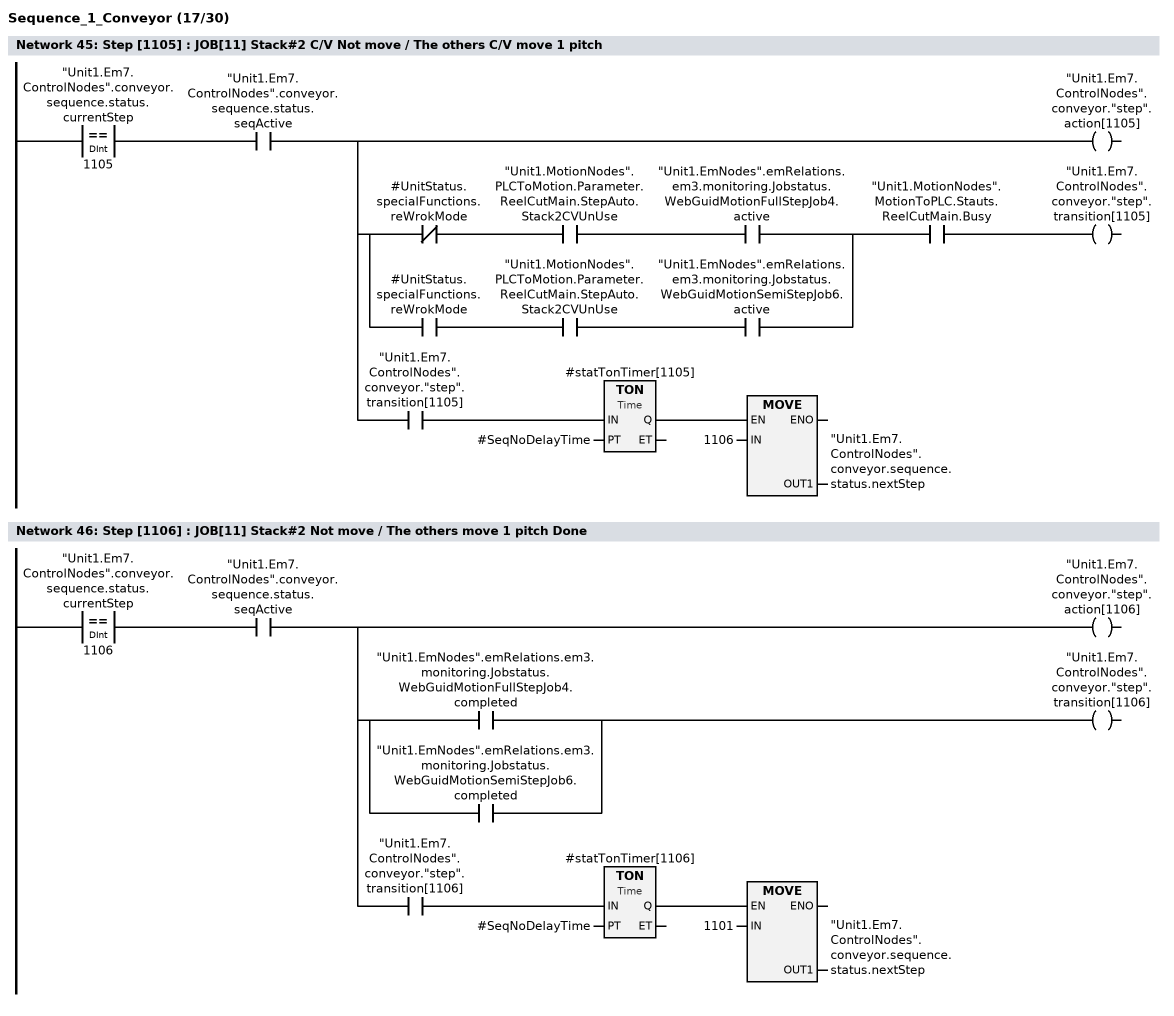
   RUNG wire#powerrail
      { S7_Templates := "SrcType := DInt" } EQ_Contact(in1 := "Unit1.Em7.ControlNodes".conveyor.sequence.status.currentStep, in2 := 1105)
      Contact( "Unit1.Em7.ControlNodes".conveyor.sequence.status.seqActive )
      wire#w1
      Coil( "Unit1.Em7.ControlNodes".conveyor."step".action[1105] )
   END_RUNG
   RUNG wire#w1
      I_Contact( #UnitStatus.specialFunctions.reWrokMode )
      Contact( "Unit1.MotionNodes".PLCToMotion.Parameter.ReelCutMain.StepAuto.Stack2CVUnUse )
      Contact( "Unit1.EmNodes".emRelations.em3.monitoring.Jobstatus.WebGuidMotionFullStepJob4.active )
      wire#w2
      Contact( "Unit1.MotionNodes".MotionToPLC.Stauts.ReelCutMain.Busy )
      Coil( "Unit1.Em7.ControlNodes".conveyor."step".transition[1105] )
   END_RUNG
   RUNG wire#w1
      Contact( #UnitStatus.specialFunctions.reWrokMode )
      Contact( "Unit1.MotionNodes".PLCToMotion.Parameter.ReelCutMain.StepAuto.Stack2CVUnUse )
      Contact( "Unit1.EmNodes".emRelations.em3.monitoring.Jobstatus.WebGuidMotionSemiStepJob6.active )
   END_RUNG wire#w2
   RUNG wire#w1
      Contact( "Unit1.Em7.ControlNodes".conveyor."step".transition[1105] )
      { S7_Templates := "time_type := Time" } #statTonTimer[1105].TON(pt := #SeqNoDelayTime, et =>)
      Move(in := 1106, out1 => "Unit1.Em7.ControlNodes".conveyor.sequence.status.nextStep)
   END_RUNG
   // the same network as SCL:
   "Unit1.Em7.ControlNodes".conveyor."step".action[1105] := ("Unit1.Em7.ControlNodes".conveyor.sequence.status.currentStep = 1105) AND "Unit1.Em7.ControlNodes".conveyor.sequence.status.seqActive;
   "Unit1.Em7.ControlNodes".conveyor."step".transition[1105] := ("Unit1.Em7.ControlNodes".conveyor.sequence.status.currentStep = 1105) AND "Unit1.Em7.ControlNodes".conveyor.sequence.status.seqActive AND ((NOT #UnitStatus.specialFunctions.reWrokMode AND "Unit1.MotionNodes".PLCToMotion.Parameter.ReelCutMain.StepAuto.Stack2CVUnUse AND "Unit1.EmNodes".emRelations.em3.monitoring.Jobstatus.WebGuidMotionFullStepJob4.active) OR (#UnitStatus.specialFunctions.reWrokMode AND "Unit1.MotionNodes".PLCToMotion.Parameter.ReelCutMain.StepAuto.Stack2CVUnUse AND "Unit1.EmNodes".emRelations.em3.monitoring.Jobstatus.WebGuidMotionSemiStepJob6.active)) AND "Unit1.MotionNodes".MotionToPLC.Stauts.ReelCutMain.Busy;
   #statTonTimer[1105].TON(IN := ("Unit1.Em7.ControlNodes".conveyor.sequence.status.currentStep = 1105) AND "Unit1.Em7.ControlNodes".conveyor.sequence.status.seqActive AND "Unit1.Em7.ControlNodes".conveyor."step".transition[1105],
                           PT := #SeqNoDelayTime);
   IF #statTonTimer[1105].Q THEN "Unit1.Em7.ControlNodes".conveyor.sequence.status.nextStep := 1106; END_IF;
END_REGION

REGION Network 46: Step [1106] : JOB[11] Stack#2 Not move / The others move 1 pitch Done
   RUNG wire#powerrail
      { S7_Templates := "SrcType := DInt" } EQ_Contact(in1 := "Unit1.Em7.ControlNodes".conveyor.sequence.status.currentStep, in2 := 1106)
      Contact( "Unit1.Em7.ControlNodes".conveyor.sequence.status.seqActive )
      wire#w1
      Coil( "Unit1.Em7.ControlNodes".conveyor."step".action[1106] )
   END_RUNG
   RUNG wire#w1
      Contact( "Unit1.EmNodes".emRelations.em3.monitoring.Jobstatus.WebGuidMotionFullStepJob4.completed )
      wire#w2
      Coil( "Unit1.Em7.ControlNodes".conveyor."step".transition[1106] )
   END_RUNG
   RUNG wire#w1
      Contact( "Unit1.EmNodes".emRelations.em3.monitoring.Jobstatus.WebGuidMotionSemiStepJob6.completed )
   END_RUNG wire#w2
   RUNG wire#w1
      Contact( "Unit1.Em7.ControlNodes".conveyor."step".transition[1106] )
      { S7_Templates := "time_type := Time" } #statTonTimer[1106].TON(pt := #SeqNoDelayTime, et =>)
      Move(in := 1101, out1 => "Unit1.Em7.ControlNodes".conveyor.sequence.status.nextStep)
   END_RUNG
   // the same network as SCL:
   "Unit1.Em7.ControlNodes".conveyor."step".action[1106] := ("Unit1.Em7.ControlNodes".conveyor.sequence.status.currentStep = 1106) AND "Unit1.Em7.ControlNodes".conveyor.sequence.status.seqActive;
   "Unit1.Em7.ControlNodes".conveyor."step".transition[1106] := ("Unit1.Em7.ControlNodes".conveyor.sequence.status.currentStep = 1106) AND "Unit1.Em7.ControlNodes".conveyor.sequence.status.seqActive AND ("Unit1.EmNodes".emRelations.em3.monitoring.Jobstatus.WebGuidMotionFullStepJob4.completed OR "Unit1.EmNodes".emRelations.em3.monitoring.Jobstatus.WebGuidMotionSemiStepJob6.completed);
   #statTonTimer[1106].TON(IN := ("Unit1.Em7.ControlNodes".conveyor.sequence.status.currentStep = 1106) AND "Unit1.Em7.ControlNodes".conveyor.sequence.status.seqActive AND "Unit1.Em7.ControlNodes".conveyor."step".transition[1106],
                           PT := #SeqNoDelayTime);
   IF #statTonTimer[1106].Q THEN "Unit1.Em7.ControlNodes".conveyor.sequence.status.nextStep := 1101; END_IF;
END_REGION

REGION Network 47: Step [1110] : JOB[11] Call Stack#1 Work CMD
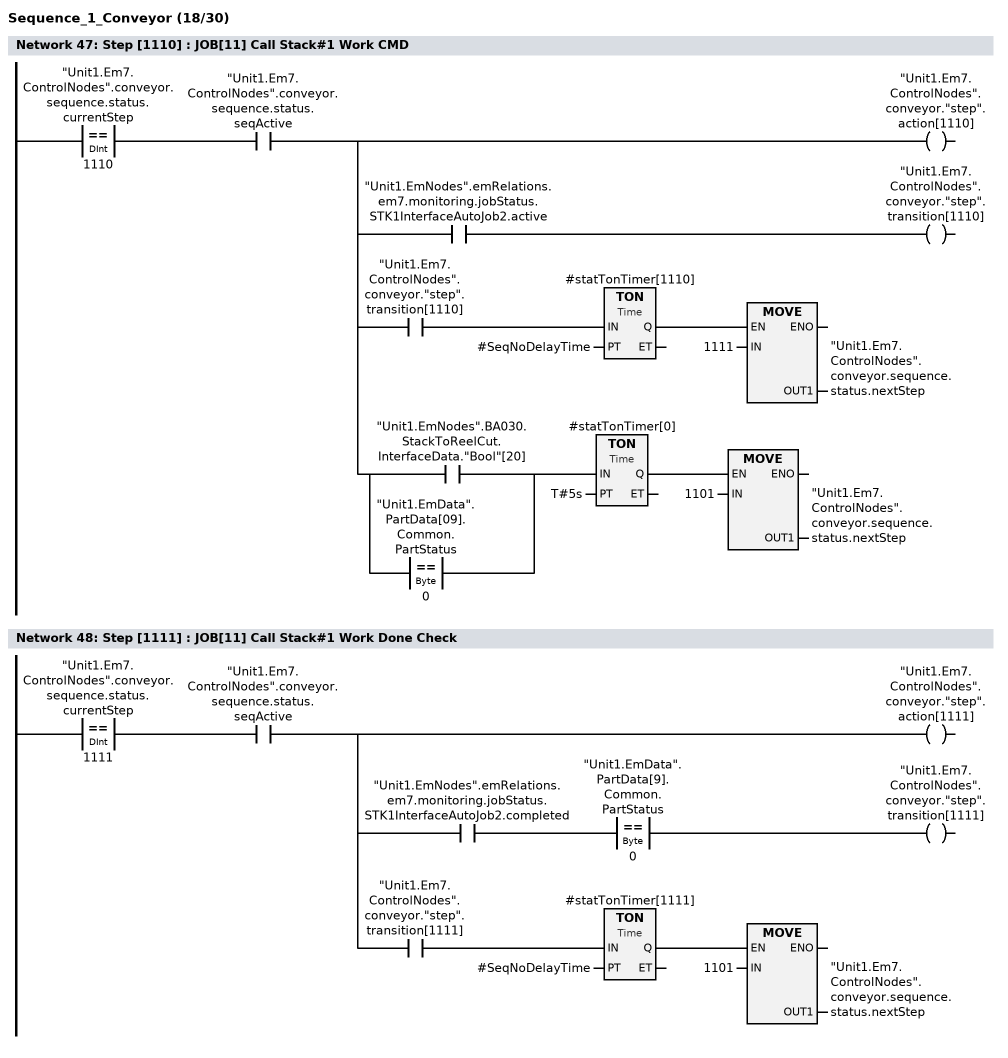
   RUNG wire#powerrail
      { S7_Templates := "SrcType := DInt" } EQ_Contact(in1 := "Unit1.Em7.ControlNodes".conveyor.sequence.status.currentStep, in2 := 1110)
      Contact( "Unit1.Em7.ControlNodes".conveyor.sequence.status.seqActive )
      wire#w1
      Coil( "Unit1.Em7.ControlNodes".conveyor."step".action[1110] )
   END_RUNG
   RUNG wire#w1
      Contact( "Unit1.EmNodes".emRelations.em7.monitoring.jobStatus.STK1InterfaceAutoJob2.active )
      Coil( "Unit1.Em7.ControlNodes".conveyor."step".transition[1110] )
   END_RUNG
   RUNG wire#w1
      Contact( "Unit1.Em7.ControlNodes".conveyor."step".transition[1110] )
      { S7_Templates := "time_type := Time" } #statTonTimer[1110].TON(pt := #SeqNoDelayTime, et =>)
      Move(in := 1111, out1 => "Unit1.Em7.ControlNodes".conveyor.sequence.status.nextStep)
   END_RUNG
   RUNG wire#w1
      Contact( "Unit1.EmNodes".BA030.StackToReelCut.InterfaceData."Bool"[20] )
      wire#w2
      { S7_Templates := "time_type := Time" } #statTonTimer[0].TON(pt := T#5s, et =>)
      Move(in := 1101, out1 => "Unit1.Em7.ControlNodes".conveyor.sequence.status.nextStep)
   END_RUNG
   RUNG wire#w1
      { S7_Templates := "SrcType := Byte" } EQ_Contact(in1 := "Unit1.EmData".PartData[09].Common.PartStatus, in2 := 0)
   END_RUNG wire#w2
   // the same network as SCL:
   "Unit1.Em7.ControlNodes".conveyor."step".action[1110] := ("Unit1.Em7.ControlNodes".conveyor.sequence.status.currentStep = 1110) AND "Unit1.Em7.ControlNodes".conveyor.sequence.status.seqActive;
   "Unit1.Em7.ControlNodes".conveyor."step".transition[1110] := ("Unit1.Em7.ControlNodes".conveyor.sequence.status.currentStep = 1110) AND "Unit1.Em7.ControlNodes".conveyor.sequence.status.seqActive AND "Unit1.EmNodes".emRelations.em7.monitoring.jobStatus.STK1InterfaceAutoJob2.active;
   #statTonTimer[1110].TON(IN := ("Unit1.Em7.ControlNodes".conveyor.sequence.status.currentStep = 1110) AND "Unit1.Em7.ControlNodes".conveyor.sequence.status.seqActive AND "Unit1.Em7.ControlNodes".conveyor."step".transition[1110],
                           PT := #SeqNoDelayTime);
   IF #statTonTimer[1110].Q THEN "Unit1.Em7.ControlNodes".conveyor.sequence.status.nextStep := 1111; END_IF;
   #statTonTimer[0].TON(IN := ("Unit1.Em7.ControlNodes".conveyor.sequence.status.currentStep = 1110) AND "Unit1.Em7.ControlNodes".conveyor.sequence.status.seqActive AND ("Unit1.EmNodes".BA030.StackToReelCut.InterfaceData."Bool"[20] OR ("Unit1.EmData".PartData[09].Common.PartStatus = 0)),
                        PT := T#5s);
   IF #statTonTimer[0].Q THEN "Unit1.Em7.ControlNodes".conveyor.sequence.status.nextStep := 1101; END_IF;
END_REGION

REGION Network 48: Step [1111] : JOB[11] Call Stack#1 Work Done Check
   RUNG wire#powerrail
      { S7_Templates := "SrcType := DInt" } EQ_Contact(in1 := "Unit1.Em7.ControlNodes".conveyor.sequence.status.currentStep, in2 := 1111)
      Contact( "Unit1.Em7.ControlNodes".conveyor.sequence.status.seqActive )
      wire#w1
      Coil( "Unit1.Em7.ControlNodes".conveyor."step".action[1111] )
   END_RUNG
   RUNG wire#w1
      Contact( "Unit1.EmNodes".emRelations.em7.monitoring.jobStatus.STK1InterfaceAutoJob2.completed )
      { S7_Templates := "SrcType := Byte" } EQ_Contact(in1 := "Unit1.EmData".PartData[9].Common.PartStatus, in2 := 0)
      Coil( "Unit1.Em7.ControlNodes".conveyor."step".transition[1111] )
   END_RUNG
   RUNG wire#w1
      Contact( "Unit1.Em7.ControlNodes".conveyor."step".transition[1111] )
      { S7_Templates := "time_type := Time" } #statTonTimer[1111].TON(pt := #SeqNoDelayTime, et =>)
      Move(in := 1101, out1 => "Unit1.Em7.ControlNodes".conveyor.sequence.status.nextStep)
   END_RUNG
   // the same network as SCL:
   "Unit1.Em7.ControlNodes".conveyor."step".action[1111] := ("Unit1.Em7.ControlNodes".conveyor.sequence.status.currentStep = 1111) AND "Unit1.Em7.ControlNodes".conveyor.sequence.status.seqActive;
   "Unit1.Em7.ControlNodes".conveyor."step".transition[1111] := ("Unit1.Em7.ControlNodes".conveyor.sequence.status.currentStep = 1111) AND "Unit1.Em7.ControlNodes".conveyor.sequence.status.seqActive AND "Unit1.EmNodes".emRelations.em7.monitoring.jobStatus.STK1InterfaceAutoJob2.completed AND ("Unit1.EmData".PartData[9].Common.PartStatus = 0);
   #statTonTimer[1111].TON(IN := ("Unit1.Em7.ControlNodes".conveyor.sequence.status.currentStep = 1111) AND "Unit1.Em7.ControlNodes".conveyor.sequence.status.seqActive AND "Unit1.Em7.ControlNodes".conveyor."step".transition[1111],
                           PT := #SeqNoDelayTime);
   IF #statTonTimer[1111].Q THEN "Unit1.Em7.ControlNodes".conveyor.sequence.status.nextStep := 1101; END_IF;
END_REGION

REGION Network 49: Step [1115] : JOB[11] Call Stack#2 Work CMD
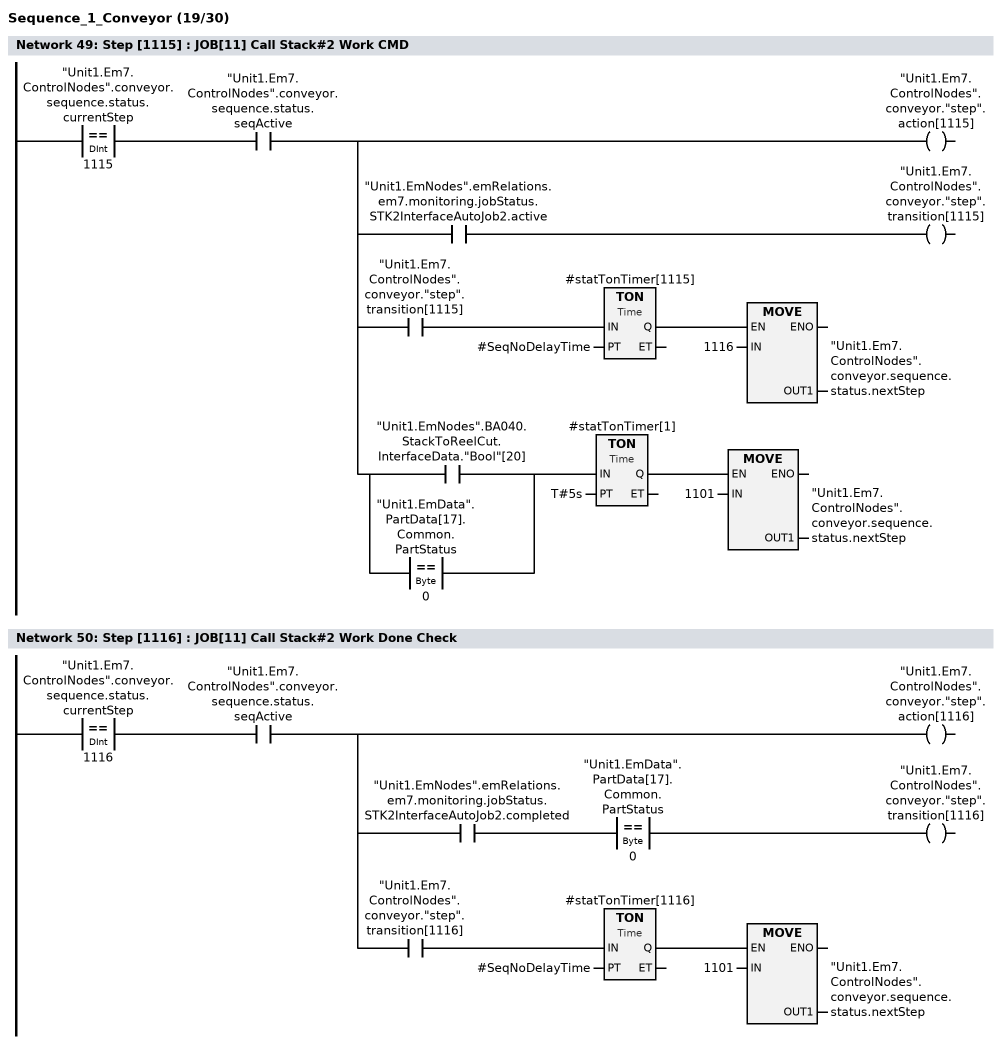
   RUNG wire#powerrail
      { S7_Templates := "SrcType := DInt" } EQ_Contact(in1 := "Unit1.Em7.ControlNodes".conveyor.sequence.status.currentStep, in2 := 1115)
      Contact( "Unit1.Em7.ControlNodes".conveyor.sequence.status.seqActive )
      wire#w1
      Coil( "Unit1.Em7.ControlNodes".conveyor."step".action[1115] )
   END_RUNG
   RUNG wire#w1
      Contact( "Unit1.EmNodes".emRelations.em7.monitoring.jobStatus.STK2InterfaceAutoJob2.active )
      Coil( "Unit1.Em7.ControlNodes".conveyor."step".transition[1115] )
   END_RUNG
   RUNG wire#w1
      Contact( "Unit1.Em7.ControlNodes".conveyor."step".transition[1115] )
      { S7_Templates := "time_type := Time" } #statTonTimer[1115].TON(pt := #SeqNoDelayTime, et =>)
      Move(in := 1116, out1 => "Unit1.Em7.ControlNodes".conveyor.sequence.status.nextStep)
   END_RUNG
   RUNG wire#w1
      Contact( "Unit1.EmNodes".BA040.StackToReelCut.InterfaceData."Bool"[20] )
      wire#w2
      { S7_Templates := "time_type := Time" } #statTonTimer[1].TON(pt := T#5s, et =>)
      Move(in := 1101, out1 => "Unit1.Em7.ControlNodes".conveyor.sequence.status.nextStep)
   END_RUNG
   RUNG wire#w1
      { S7_Templates := "SrcType := Byte" } EQ_Contact(in1 := "Unit1.EmData".PartData[17].Common.PartStatus, in2 := 0)
   END_RUNG wire#w2
   // the same network as SCL:
   "Unit1.Em7.ControlNodes".conveyor."step".action[1115] := ("Unit1.Em7.ControlNodes".conveyor.sequence.status.currentStep = 1115) AND "Unit1.Em7.ControlNodes".conveyor.sequence.status.seqActive;
   "Unit1.Em7.ControlNodes".conveyor."step".transition[1115] := ("Unit1.Em7.ControlNodes".conveyor.sequence.status.currentStep = 1115) AND "Unit1.Em7.ControlNodes".conveyor.sequence.status.seqActive AND "Unit1.EmNodes".emRelations.em7.monitoring.jobStatus.STK2InterfaceAutoJob2.active;
   #statTonTimer[1115].TON(IN := ("Unit1.Em7.ControlNodes".conveyor.sequence.status.currentStep = 1115) AND "Unit1.Em7.ControlNodes".conveyor.sequence.status.seqActive AND "Unit1.Em7.ControlNodes".conveyor."step".transition[1115],
                           PT := #SeqNoDelayTime);
   IF #statTonTimer[1115].Q THEN "Unit1.Em7.ControlNodes".conveyor.sequence.status.nextStep := 1116; END_IF;
   #statTonTimer[1].TON(IN := ("Unit1.Em7.ControlNodes".conveyor.sequence.status.currentStep = 1115) AND "Unit1.Em7.ControlNodes".conveyor.sequence.status.seqActive AND ("Unit1.EmNodes".BA040.StackToReelCut.InterfaceData."Bool"[20] OR ("Unit1.EmData".PartData[17].Common.PartStatus = 0)),
                        PT := T#5s);
   IF #statTonTimer[1].Q THEN "Unit1.Em7.ControlNodes".conveyor.sequence.status.nextStep := 1101; END_IF;
END_REGION

REGION Network 50: Step [1116] : JOB[11] Call Stack#2 Work Done Check
   RUNG wire#powerrail
      { S7_Templates := "SrcType := DInt" } EQ_Contact(in1 := "Unit1.Em7.ControlNodes".conveyor.sequence.status.currentStep, in2 := 1116)
      Contact( "Unit1.Em7.ControlNodes".conveyor.sequence.status.seqActive )
      wire#w1
      Coil( "Unit1.Em7.ControlNodes".conveyor."step".action[1116] )
   END_RUNG
   RUNG wire#w1
      Contact( "Unit1.EmNodes".emRelations.em7.monitoring.jobStatus.STK2InterfaceAutoJob2.completed )
      { S7_Templates := "SrcType := Byte" } EQ_Contact(in1 := "Unit1.EmData".PartData[17].Common.PartStatus, in2 := 0)
      Coil( "Unit1.Em7.ControlNodes".conveyor."step".transition[1116] )
   END_RUNG
   RUNG wire#w1
      Contact( "Unit1.Em7.ControlNodes".conveyor."step".transition[1116] )
      { S7_Templates := "time_type := Time" } #statTonTimer[1116].TON(pt := #SeqNoDelayTime, et =>)
      Move(in := 1101, out1 => "Unit1.Em7.ControlNodes".conveyor.sequence.status.nextStep)
   END_RUNG
   // the same network as SCL:
   "Unit1.Em7.ControlNodes".conveyor."step".action[1116] := ("Unit1.Em7.ControlNodes".conveyor.sequence.status.currentStep = 1116) AND "Unit1.Em7.ControlNodes".conveyor.sequence.status.seqActive;
   "Unit1.Em7.ControlNodes".conveyor."step".transition[1116] := ("Unit1.Em7.ControlNodes".conveyor.sequence.status.currentStep = 1116) AND "Unit1.Em7.ControlNodes".conveyor.sequence.status.seqActive AND "Unit1.EmNodes".emRelations.em7.monitoring.jobStatus.STK2InterfaceAutoJob2.completed AND ("Unit1.EmData".PartData[17].Common.PartStatus = 0);
   #statTonTimer[1116].TON(IN := ("Unit1.Em7.ControlNodes".conveyor.sequence.status.currentStep = 1116) AND "Unit1.Em7.ControlNodes".conveyor.sequence.status.seqActive AND "Unit1.Em7.ControlNodes".conveyor."step".transition[1116],
                           PT := #SeqNoDelayTime);
   IF #statTonTimer[1116].Q THEN "Unit1.Em7.ControlNodes".conveyor.sequence.status.nextStep := 1101; END_IF;
END_REGION

REGION Network 51: Step [1120] : JOB[11] Call Success -> Stack Full Check
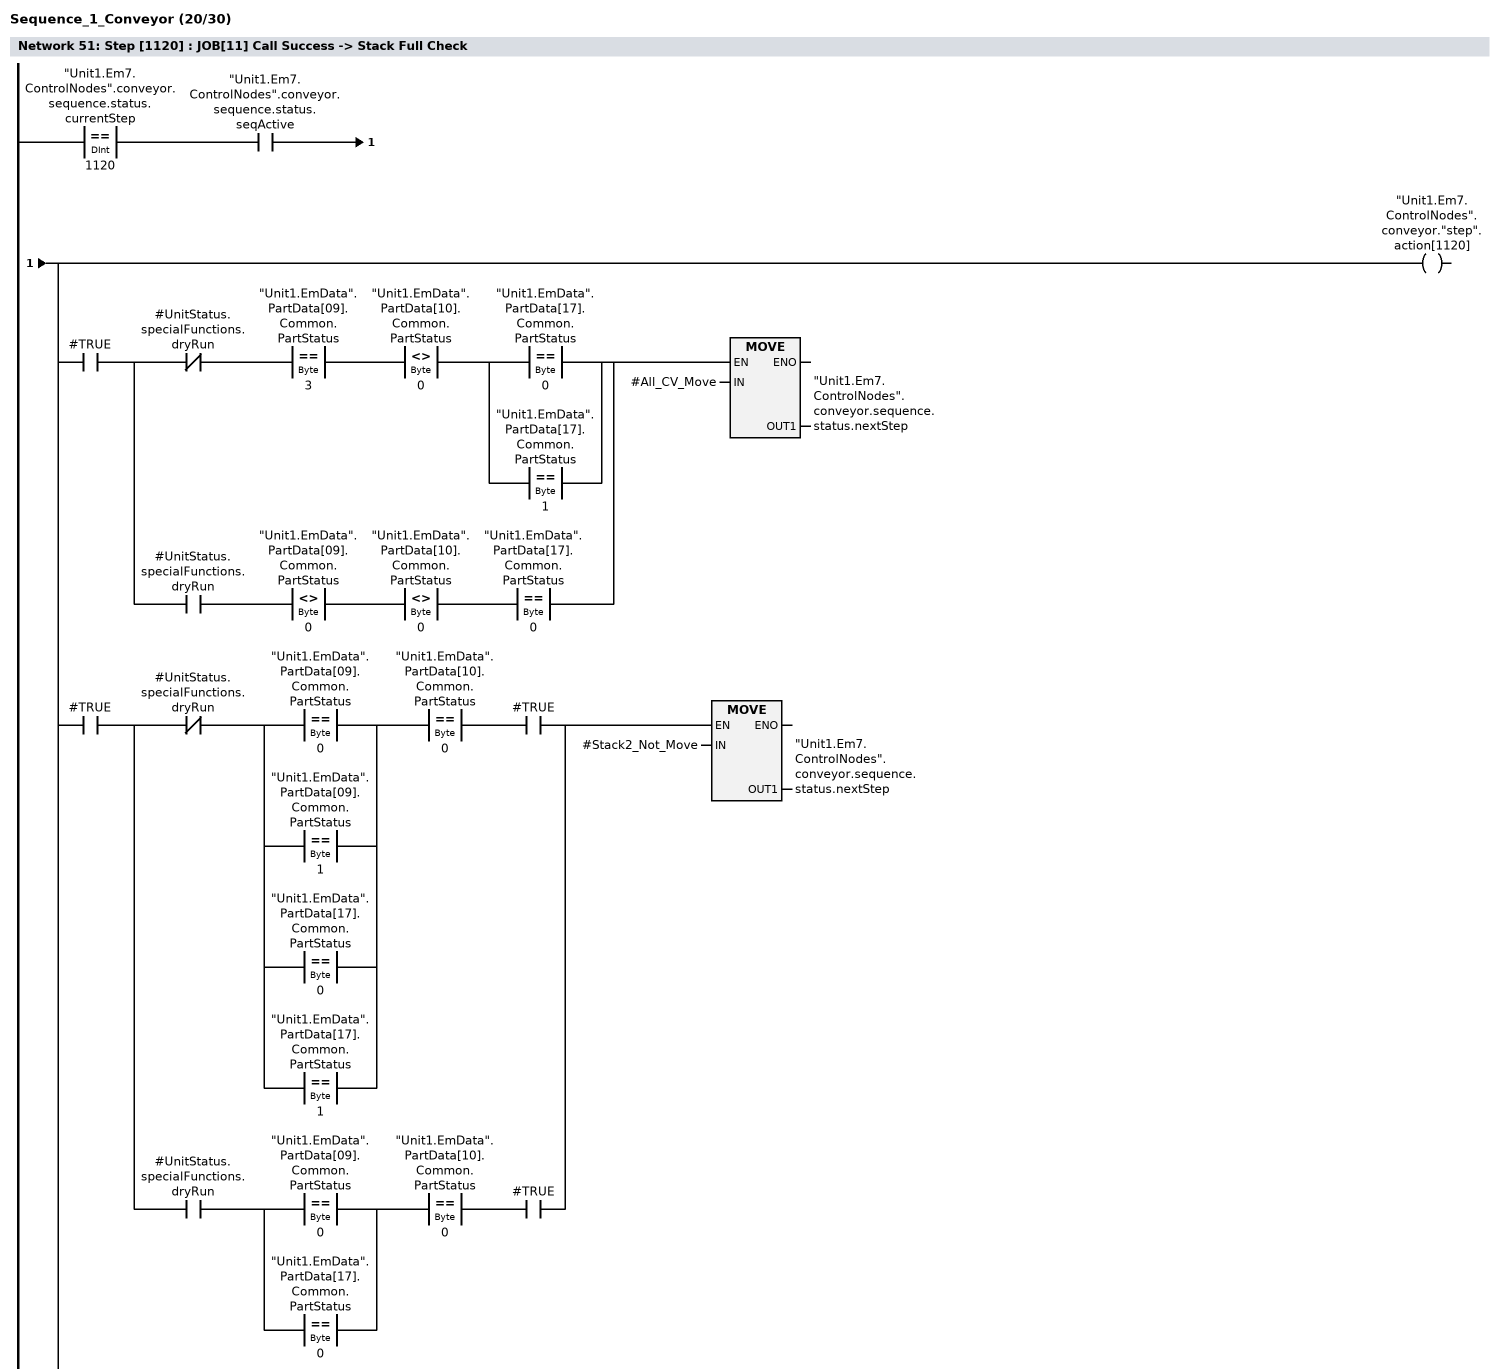
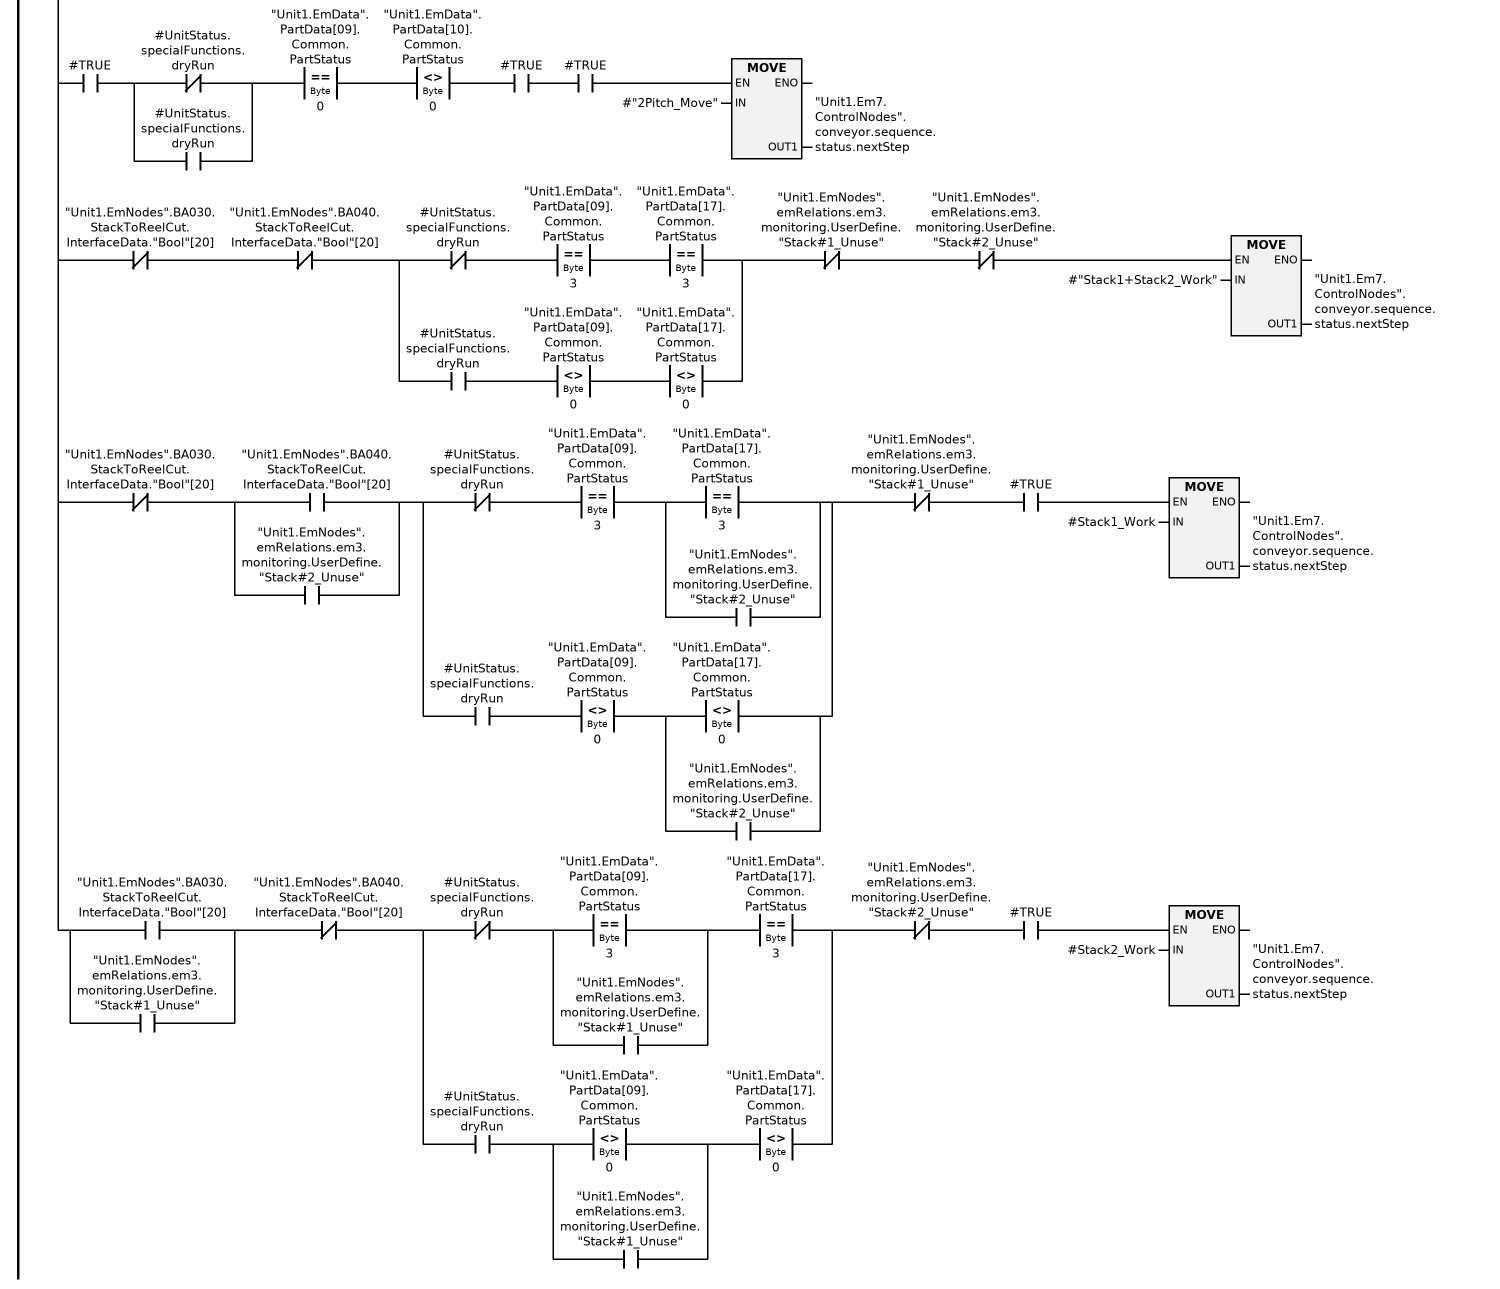
   RUNG wire#powerrail
      { S7_Templates := "SrcType := DInt" } EQ_Contact(in1 := "Unit1.Em7.ControlNodes".conveyor.sequence.status.currentStep, in2 := 1120)
      Contact( "Unit1.Em7.ControlNodes".conveyor.sequence.status.seqActive )
      wire#w1
      Coil( "Unit1.Em7.ControlNodes".conveyor."step".action[1120] )
   END_RUNG
   RUNG wire#w1
      Contact( #TRUE )
      wire#w2
      I_Contact( #UnitStatus.specialFunctions.dryRun )
      { S7_Templates := "SrcType := Byte" } EQ_Contact(in1 := "Unit1.EmData".PartData[09].Common.PartStatus, in2 := 3)
      { S7_Templates := "SrcType := Byte" } NE_Contact(in1 := "Unit1.EmData".PartData[10].Common.PartStatus, in2 := 0)
      wire#w3
      { S7_Templates := "SrcType := Byte" } EQ_Contact(in1 := "Unit1.EmData".PartData[17].Common.PartStatus, in2 := 0)
      wire#w4
      Move(in := #All_CV_Move, out1 => "Unit1.Em7.ControlNodes".conveyor.sequence.status.nextStep)
   END_RUNG
   RUNG wire#w3
      { S7_Templates := "SrcType := Byte" } EQ_Contact(in1 := "Unit1.EmData".PartData[17].Common.PartStatus, in2 := 1)
   END_RUNG wire#w4
   RUNG wire#w2
      Contact( #UnitStatus.specialFunctions.dryRun )
      { S7_Templates := "SrcType := Byte" } NE_Contact(in1 := "Unit1.EmData".PartData[09].Common.PartStatus, in2 := 0)
      { S7_Templates := "SrcType := Byte" } NE_Contact(in1 := "Unit1.EmData".PartData[10].Common.PartStatus, in2 := 0)
      { S7_Templates := "SrcType := Byte" } EQ_Contact(in1 := "Unit1.EmData".PartData[17].Common.PartStatus, in2 := 0)
   END_RUNG wire#w4
   RUNG wire#w1
      Contact( #TRUE )
      wire#w5
      I_Contact( #UnitStatus.specialFunctions.dryRun )
      wire#w6
      { S7_Templates := "SrcType := Byte" } EQ_Contact(in1 := "Unit1.EmData".PartData[09].Common.PartStatus, in2 := 0)
      wire#w7
      { S7_Templates := "SrcType := Byte" } EQ_Contact(in1 := "Unit1.EmData".PartData[10].Common.PartStatus, in2 := 0)
      Contact( #TRUE )
      wire#w8
      Move(in := #Stack2_Not_Move, out1 => "Unit1.Em7.ControlNodes".conveyor.sequence.status.nextStep)
   END_RUNG
   RUNG wire#w6
      { S7_Templates := "SrcType := Byte" } EQ_Contact(in1 := "Unit1.EmData".PartData[09].Common.PartStatus, in2 := 1)
   END_RUNG wire#w7
   RUNG wire#w6
      { S7_Templates := "SrcType := Byte" } EQ_Contact(in1 := "Unit1.EmData".PartData[17].Common.PartStatus, in2 := 0)
   END_RUNG wire#w7
   RUNG wire#w6
      { S7_Templates := "SrcType := Byte" } EQ_Contact(in1 := "Unit1.EmData".PartData[17].Common.PartStatus, in2 := 1)
   END_RUNG wire#w7
   RUNG wire#w5
      Contact( #UnitStatus.specialFunctions.dryRun )
      wire#w9
      { S7_Templates := "SrcType := Byte" } EQ_Contact(in1 := "Unit1.EmData".PartData[09].Common.PartStatus, in2 := 0)
      wire#w10
      { S7_Templates := "SrcType := Byte" } EQ_Contact(in1 := "Unit1.EmData".PartData[10].Common.PartStatus, in2 := 0)
      Contact( #TRUE )
   END_RUNG wire#w8
   RUNG wire#w9
      { S7_Templates := "SrcType := Byte" } EQ_Contact(in1 := "Unit1.EmData".PartData[17].Common.PartStatus, in2 := 0)
   END_RUNG wire#w10
   RUNG wire#w1
      Contact( #TRUE )
      wire#w11
      I_Contact( #UnitStatus.specialFunctions.dryRun )
      wire#w12
      { S7_Templates := "SrcType := Byte" } EQ_Contact(in1 := "Unit1.EmData".PartData[09].Common.PartStatus, in2 := 0)
      { S7_Templates := "SrcType := Byte" } NE_Contact(in1 := "Unit1.EmData".PartData[10].Common.PartStatus, in2 := 0)
      Contact( #TRUE )
      Contact( #TRUE )
      Move(in := #"2Pitch_Move", out1 => "Unit1.Em7.ControlNodes".conveyor.sequence.status.nextStep)
   END_RUNG
   RUNG wire#w11
      Contact( #UnitStatus.specialFunctions.dryRun )
   END_RUNG wire#w12
   RUNG wire#w1
      I_Contact( "Unit1.EmNodes".BA030.StackToReelCut.InterfaceData."Bool"[20] )
      I_Contact( "Unit1.EmNodes".BA040.StackToReelCut.InterfaceData."Bool"[20] )
      wire#w13
      I_Contact( #UnitStatus.specialFunctions.dryRun )
      { S7_Templates := "SrcType := Byte" } EQ_Contact(in1 := "Unit1.EmData".PartData[09].Common.PartStatus, in2 := 3)
      { S7_Templates := "SrcType := Byte" } EQ_Contact(in1 := "Unit1.EmData".PartData[17].Common.PartStatus, in2 := 3)
      wire#w14
      I_Contact( "Unit1.EmNodes".emRelations.em3.monitoring.UserDefine."Stack#1_Unuse" )
      I_Contact( "Unit1.EmNodes".emRelations.em3.monitoring.UserDefine."Stack#2_Unuse" )
      Move(in := #"Stack1+Stack2_Work", out1 => "Unit1.Em7.ControlNodes".conveyor.sequence.status.nextStep)
   END_RUNG
   RUNG wire#w13
      Contact( #UnitStatus.specialFunctions.dryRun )
      { S7_Templates := "SrcType := Byte" } NE_Contact(in1 := "Unit1.EmData".PartData[09].Common.PartStatus, in2 := 0)
      { S7_Templates := "SrcType := Byte" } NE_Contact(in1 := "Unit1.EmData".PartData[17].Common.PartStatus, in2 := 0)
   END_RUNG wire#w14
   RUNG wire#w1
      I_Contact( "Unit1.EmNodes".BA030.StackToReelCut.InterfaceData."Bool"[20] )
      wire#w15
      Contact( "Unit1.EmNodes".BA040.StackToReelCut.InterfaceData."Bool"[20] )
      wire#w16
      I_Contact( #UnitStatus.specialFunctions.dryRun )
      { S7_Templates := "SrcType := Byte" } EQ_Contact(in1 := "Unit1.EmData".PartData[09].Common.PartStatus, in2 := 3)
      wire#w17
      { S7_Templates := "SrcType := Byte" } EQ_Contact(in1 := "Unit1.EmData".PartData[17].Common.PartStatus, in2 := 3)
      wire#w18
      I_Contact( "Unit1.EmNodes".emRelations.em3.monitoring.UserDefine."Stack#1_Unuse" )
      Contact( #TRUE )
      Move(in := #Stack1_Work, out1 => "Unit1.Em7.ControlNodes".conveyor.sequence.status.nextStep)
   END_RUNG
   RUNG wire#w15
      Contact( "Unit1.EmNodes".emRelations.em3.monitoring.UserDefine."Stack#2_Unuse" )
   END_RUNG wire#w16
   RUNG wire#w17
      Contact( "Unit1.EmNodes".emRelations.em3.monitoring.UserDefine."Stack#2_Unuse" )
   END_RUNG wire#w18
   RUNG wire#w16
      Contact( #UnitStatus.specialFunctions.dryRun )
      { S7_Templates := "SrcType := Byte" } NE_Contact(in1 := "Unit1.EmData".PartData[09].Common.PartStatus, in2 := 0)
      wire#w19
      { S7_Templates := "SrcType := Byte" } NE_Contact(in1 := "Unit1.EmData".PartData[17].Common.PartStatus, in2 := 0)
   END_RUNG wire#w18
   RUNG wire#w19
      Contact( "Unit1.EmNodes".emRelations.em3.monitoring.UserDefine."Stack#2_Unuse" )
   END_RUNG wire#w18
   RUNG wire#w1
      Contact( "Unit1.EmNodes".BA030.StackToReelCut.InterfaceData."Bool"[20] )
      wire#w20
      I_Contact( "Unit1.EmNodes".BA040.StackToReelCut.InterfaceData."Bool"[20] )
      wire#w21
      I_Contact( #UnitStatus.specialFunctions.dryRun )
      wire#w22
      { S7_Templates := "SrcType := Byte" } EQ_Contact(in1 := "Unit1.EmData".PartData[09].Common.PartStatus, in2 := 3)
      wire#w23
      { S7_Templates := "SrcType := Byte" } EQ_Contact(in1 := "Unit1.EmData".PartData[17].Common.PartStatus, in2 := 3)
      wire#w24
      I_Contact( "Unit1.EmNodes".emRelations.em3.monitoring.UserDefine."Stack#2_Unuse" )
      Contact( #TRUE )
      Move(in := #Stack2_Work, out1 => "Unit1.Em7.ControlNodes".conveyor.sequence.status.nextStep)
   END_RUNG
   RUNG wire#w1
      Contact( "Unit1.EmNodes".emRelations.em3.monitoring.UserDefine."Stack#1_Unuse" )
   END_RUNG wire#w20
   RUNG wire#w22
      Contact( "Unit1.EmNodes".emRelations.em3.monitoring.UserDefine."Stack#1_Unuse" )
   END_RUNG wire#w23
   RUNG wire#w21
      Contact( #UnitStatus.specialFunctions.dryRun )
      wire#w25
      { S7_Templates := "SrcType := Byte" } NE_Contact(in1 := "Unit1.EmData".PartData[09].Common.PartStatus, in2 := 0)
      wire#w26
      { S7_Templates := "SrcType := Byte" } NE_Contact(in1 := "Unit1.EmData".PartData[17].Common.PartStatus, in2 := 0)
   END_RUNG wire#w24
   RUNG wire#w25
      Contact( "Unit1.EmNodes".emRelations.em3.monitoring.UserDefine."Stack#1_Unuse" )
   END_RUNG wire#w26
   // the same network as SCL:
   "Unit1.Em7.ControlNodes".conveyor."step".action[1120] := ("Unit1.Em7.ControlNodes".conveyor.sequence.status.currentStep = 1120) AND "Unit1.Em7.ControlNodes".conveyor.sequence.status.seqActive;
   IF ("Unit1.Em7.ControlNodes".conveyor.sequence.status.currentStep = 1120) AND "Unit1.Em7.ControlNodes".conveyor.sequence.status.seqActive AND #TRUE AND ((NOT #UnitStatus.specialFunctions.dryRun AND ("Unit1.EmData".PartData[09].Common.PartStatus = 3) AND ("Unit1.EmData".PartData[10].Common.PartStatus <> 0) AND (("Unit1.EmData".PartData[17].Common.PartStatus = 0) OR ("Unit1.EmData".PartData[17].Common.PartStatus = 1))) OR (#UnitStatus.specialFunctions.dryRun AND ("Unit1.EmData".PartData[09].Common.PartStatus <> 0) AND ("Unit1.EmData".PartData[10].Common.PartStatus <> 0) AND ("Unit1.EmData".PartData[17].Common.PartStatus = 0))) THEN
       "Unit1.Em7.ControlNodes".conveyor.sequence.status.nextStep := #All_CV_Move;
   END_IF;
   IF ("Unit1.Em7.ControlNodes".conveyor.sequence.status.currentStep = 1120) AND "Unit1.Em7.ControlNodes".conveyor.sequence.status.seqActive AND #TRUE AND ((NOT #UnitStatus.specialFunctions.dryRun AND (("Unit1.EmData".PartData[09].Common.PartStatus = 0) OR ("Unit1.EmData".PartData[09].Common.PartStatus = 1) OR ("Unit1.EmData".PartData[17].Common.PartStatus = 0) OR ("Unit1.EmData".PartData[17].Common.PartStatus = 1)) AND ("Unit1.EmData".PartData[10].Common.PartStatus = 0) AND #TRUE) OR (#UnitStatus.specialFunctions.dryRun AND (("Unit1.EmData".PartData[09].Common.PartStatus = 0) OR ("Unit1.EmData".PartData[17].Common.PartStatus = 0)) AND ("Unit1.EmData".PartData[10].Common.PartStatus = 0) AND #TRUE)) THEN
       "Unit1.Em7.ControlNodes".conveyor.sequence.status.nextStep := #Stack2_Not_Move;
   END_IF;
   IF ("Unit1.Em7.ControlNodes".conveyor.sequence.status.currentStep = 1120) AND "Unit1.Em7.ControlNodes".conveyor.sequence.status.seqActive AND #TRUE AND (NOT #UnitStatus.specialFunctions.dryRun OR #UnitStatus.specialFunctions.dryRun) AND ("Unit1.EmData".PartData[09].Common.PartStatus = 0) AND ("Unit1.EmData".PartData[10].Common.PartStatus <> 0) AND #TRUE AND #TRUE THEN
       "Unit1.Em7.ControlNodes".conveyor.sequence.status.nextStep := #"2Pitch_Move";
   END_IF;
   IF ("Unit1.Em7.ControlNodes".conveyor.sequence.status.currentStep = 1120) AND "Unit1.Em7.ControlNodes".conveyor.sequence.status.seqActive AND NOT "Unit1.EmNodes".BA030.StackToReelCut.InterfaceData."Bool"[20] AND NOT "Unit1.EmNodes".BA040.StackToReelCut.InterfaceData."Bool"[20] AND ((NOT #UnitStatus.specialFunctions.dryRun AND ("Unit1.EmData".PartData[09].Common.PartStatus = 3) AND ("Unit1.EmData".PartData[17].Common.PartStatus = 3)) OR (#UnitStatus.specialFunctions.dryRun AND ("Unit1.EmData".PartData[09].Common.PartStatus <> 0) AND ("Unit1.EmData".PartData[17].Common.PartStatus <> 0))) AND NOT "Unit1.EmNodes".emRelations.em3.monitoring.UserDefine."Stack#1_Unuse" AND NOT "Unit1.EmNodes".emRelations.em3.monitoring.UserDefine."Stack#2_Unuse" THEN
       "Unit1.Em7.ControlNodes".conveyor.sequence.status.nextStep := #"Stack1+Stack2_Work";
   END_IF;
   IF ("Unit1.Em7.ControlNodes".conveyor.sequence.status.currentStep = 1120) AND "Unit1.Em7.ControlNodes".conveyor.sequence.status.seqActive AND NOT "Unit1.EmNodes".BA030.StackToReelCut.InterfaceData."Bool"[20] AND ("Unit1.EmNodes".BA040.StackToReelCut.InterfaceData."Bool"[20] OR "Unit1.EmNodes".emRelations.em3.monitoring.UserDefine."Stack#2_Unuse") AND ((NOT #UnitStatus.specialFunctions.dryRun AND ("Unit1.EmData".PartData[09].Common.PartStatus = 3) AND (("Unit1.EmData".PartData[17].Common.PartStatus = 3) OR "Unit1.EmNodes".emRelations.em3.monitoring.UserDefine."Stack#2_Unuse")) OR (#UnitStatus.specialFunctions.dryRun AND ("Unit1.EmData".PartData[09].Common.PartStatus <> 0) AND (("Unit1.EmData".PartData[17].Common.PartStatus <> 0) OR "Unit1.EmNodes".emRelations.em3.monitoring.UserDefine."Stack#2_Unuse"))) AND NOT "Unit1.EmNodes".emRelations.em3.monitoring.UserDefine."Stack#1_Unuse" AND #TRUE THEN
       "Unit1.Em7.ControlNodes".conveyor.sequence.status.nextStep := #Stack1_Work;
   END_IF;
   IF ("Unit1.Em7.ControlNodes".conveyor.sequence.status.currentStep = 1120) AND "Unit1.Em7.ControlNodes".conveyor.sequence.status.seqActive AND ("Unit1.EmNodes".BA030.StackToReelCut.InterfaceData."Bool"[20] OR "Unit1.EmNodes".emRelations.em3.monitoring.UserDefine."Stack#1_Unuse") AND NOT "Unit1.EmNodes".BA040.StackToReelCut.InterfaceData."Bool"[20] AND ((NOT #UnitStatus.specialFunctions.dryRun AND (("Unit1.EmData".PartData[09].Common.PartStatus = 3) OR "Unit1.EmNodes".emRelations.em3.monitoring.UserDefine."Stack#1_Unuse") AND ("Unit1.EmData".PartData[17].Common.PartStatus = 3)) OR (#UnitStatus.specialFunctions.dryRun AND (("Unit1.EmData".PartData[09].Common.PartStatus <> 0) OR "Unit1.EmNodes".emRelations.em3.monitoring.UserDefine."Stack#1_Unuse") AND ("Unit1.EmData".PartData[17].Common.PartStatus <> 0))) AND NOT "Unit1.EmNodes".emRelations.em3.monitoring.UserDefine."Stack#2_Unuse" AND #TRUE THEN
       "Unit1.Em7.ControlNodes".conveyor.sequence.status.nextStep := #Stack2_Work;
   END_IF;
END_REGION

REGION Network 52: Step [1130] : All C/V Move One Pitch Feeding
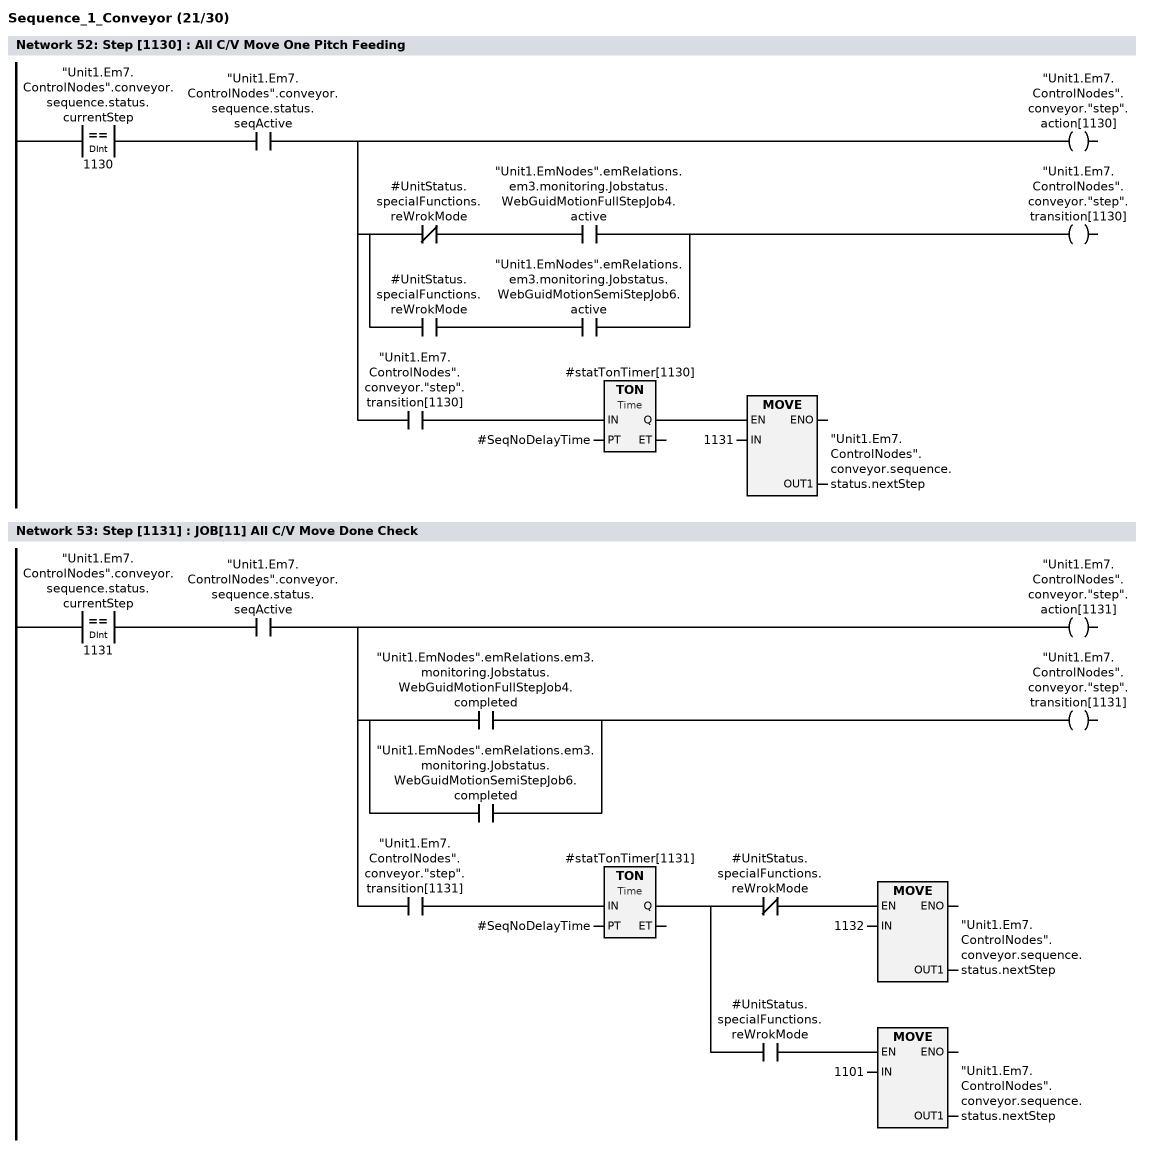
   RUNG wire#powerrail
      { S7_Templates := "SrcType := DInt" } EQ_Contact(in1 := "Unit1.Em7.ControlNodes".conveyor.sequence.status.currentStep, in2 := 1130)
      Contact( "Unit1.Em7.ControlNodes".conveyor.sequence.status.seqActive )
      wire#w1
      Coil( "Unit1.Em7.ControlNodes".conveyor."step".action[1130] )
   END_RUNG
   RUNG wire#w1
      I_Contact( #UnitStatus.specialFunctions.reWrokMode )
      Contact( "Unit1.EmNodes".emRelations.em3.monitoring.Jobstatus.WebGuidMotionFullStepJob4.active )
      wire#w2
      Coil( "Unit1.Em7.ControlNodes".conveyor."step".transition[1130] )
   END_RUNG
   RUNG wire#w1
      Contact( #UnitStatus.specialFunctions.reWrokMode )
      Contact( "Unit1.EmNodes".emRelations.em3.monitoring.Jobstatus.WebGuidMotionSemiStepJob6.active )
   END_RUNG wire#w2
   RUNG wire#w1
      Contact( "Unit1.Em7.ControlNodes".conveyor."step".transition[1130] )
      { S7_Templates := "time_type := Time" } #statTonTimer[1130].TON(pt := #SeqNoDelayTime, et =>)
      Move(in := 1131, out1 => "Unit1.Em7.ControlNodes".conveyor.sequence.status.nextStep)
   END_RUNG
   // the same network as SCL:
   "Unit1.Em7.ControlNodes".conveyor."step".action[1130] := ("Unit1.Em7.ControlNodes".conveyor.sequence.status.currentStep = 1130) AND "Unit1.Em7.ControlNodes".conveyor.sequence.status.seqActive;
   "Unit1.Em7.ControlNodes".conveyor."step".transition[1130] := ("Unit1.Em7.ControlNodes".conveyor.sequence.status.currentStep = 1130) AND "Unit1.Em7.ControlNodes".conveyor.sequence.status.seqActive AND ((NOT #UnitStatus.specialFunctions.reWrokMode AND "Unit1.EmNodes".emRelations.em3.monitoring.Jobstatus.WebGuidMotionFullStepJob4.active) OR (#UnitStatus.specialFunctions.reWrokMode AND "Unit1.EmNodes".emRelations.em3.monitoring.Jobstatus.WebGuidMotionSemiStepJob6.active));
   #statTonTimer[1130].TON(IN := ("Unit1.Em7.ControlNodes".conveyor.sequence.status.currentStep = 1130) AND "Unit1.Em7.ControlNodes".conveyor.sequence.status.seqActive AND "Unit1.Em7.ControlNodes".conveyor."step".transition[1130],
                           PT := #SeqNoDelayTime);
   IF #statTonTimer[1130].Q THEN "Unit1.Em7.ControlNodes".conveyor.sequence.status.nextStep := 1131; END_IF;
END_REGION

REGION Network 53: Step [1131] : JOB[11] All C/V Move Done Check
   RUNG wire#powerrail
      { S7_Templates := "SrcType := DInt" } EQ_Contact(in1 := "Unit1.Em7.ControlNodes".conveyor.sequence.status.currentStep, in2 := 1131)
      Contact( "Unit1.Em7.ControlNodes".conveyor.sequence.status.seqActive )
      wire#w1
      Coil( "Unit1.Em7.ControlNodes".conveyor."step".action[1131] )
   END_RUNG
   RUNG wire#w1
      Contact( "Unit1.EmNodes".emRelations.em3.monitoring.Jobstatus.WebGuidMotionFullStepJob4.completed )
      wire#w2
      Coil( "Unit1.Em7.ControlNodes".conveyor."step".transition[1131] )
   END_RUNG
   RUNG wire#w1
      Contact( "Unit1.EmNodes".emRelations.em3.monitoring.Jobstatus.WebGuidMotionSemiStepJob6.completed )
   END_RUNG wire#w2
   RUNG wire#w1
      Contact( "Unit1.Em7.ControlNodes".conveyor."step".transition[1131] )
      { S7_Templates := "time_type := Time" } #statTonTimer[1131].TON(pt := #SeqNoDelayTime, et =>)
      wire#w3
      I_Contact( #UnitStatus.specialFunctions.reWrokMode )
      Move(in := 1132, out1 => "Unit1.Em7.ControlNodes".conveyor.sequence.status.nextStep)
   END_RUNG
   RUNG wire#w3
      Contact( #UnitStatus.specialFunctions.reWrokMode )
      Move(in := 1101, out1 => "Unit1.Em7.ControlNodes".conveyor.sequence.status.nextStep)
   END_RUNG
   // the same network as SCL:
   "Unit1.Em7.ControlNodes".conveyor."step".action[1131] := ("Unit1.Em7.ControlNodes".conveyor.sequence.status.currentStep = 1131) AND "Unit1.Em7.ControlNodes".conveyor.sequence.status.seqActive;
   "Unit1.Em7.ControlNodes".conveyor."step".transition[1131] := ("Unit1.Em7.ControlNodes".conveyor.sequence.status.currentStep = 1131) AND "Unit1.Em7.ControlNodes".conveyor.sequence.status.seqActive AND ("Unit1.EmNodes".emRelations.em3.monitoring.Jobstatus.WebGuidMotionFullStepJob4.completed OR "Unit1.EmNodes".emRelations.em3.monitoring.Jobstatus.WebGuidMotionSemiStepJob6.completed);
   #statTonTimer[1131].TON(IN := ("Unit1.Em7.ControlNodes".conveyor.sequence.status.currentStep = 1131) AND "Unit1.Em7.ControlNodes".conveyor.sequence.status.seqActive AND "Unit1.Em7.ControlNodes".conveyor."step".transition[1131],
                           PT := #SeqNoDelayTime);
   IF #statTonTimer[1131].Q AND NOT #UnitStatus.specialFunctions.reWrokMode THEN
       "Unit1.Em7.ControlNodes".conveyor.sequence.status.nextStep := 1132;
   END_IF;
   IF #statTonTimer[1131].Q AND #UnitStatus.specialFunctions.reWrokMode THEN
       "Unit1.Em7.ControlNodes".conveyor.sequence.status.nextStep := 1101;
   END_IF;
END_REGION

REGION Network 54: Step [1132] : JOB[11] Stack#2 C/V Not move / The others C/V move 1 pitch
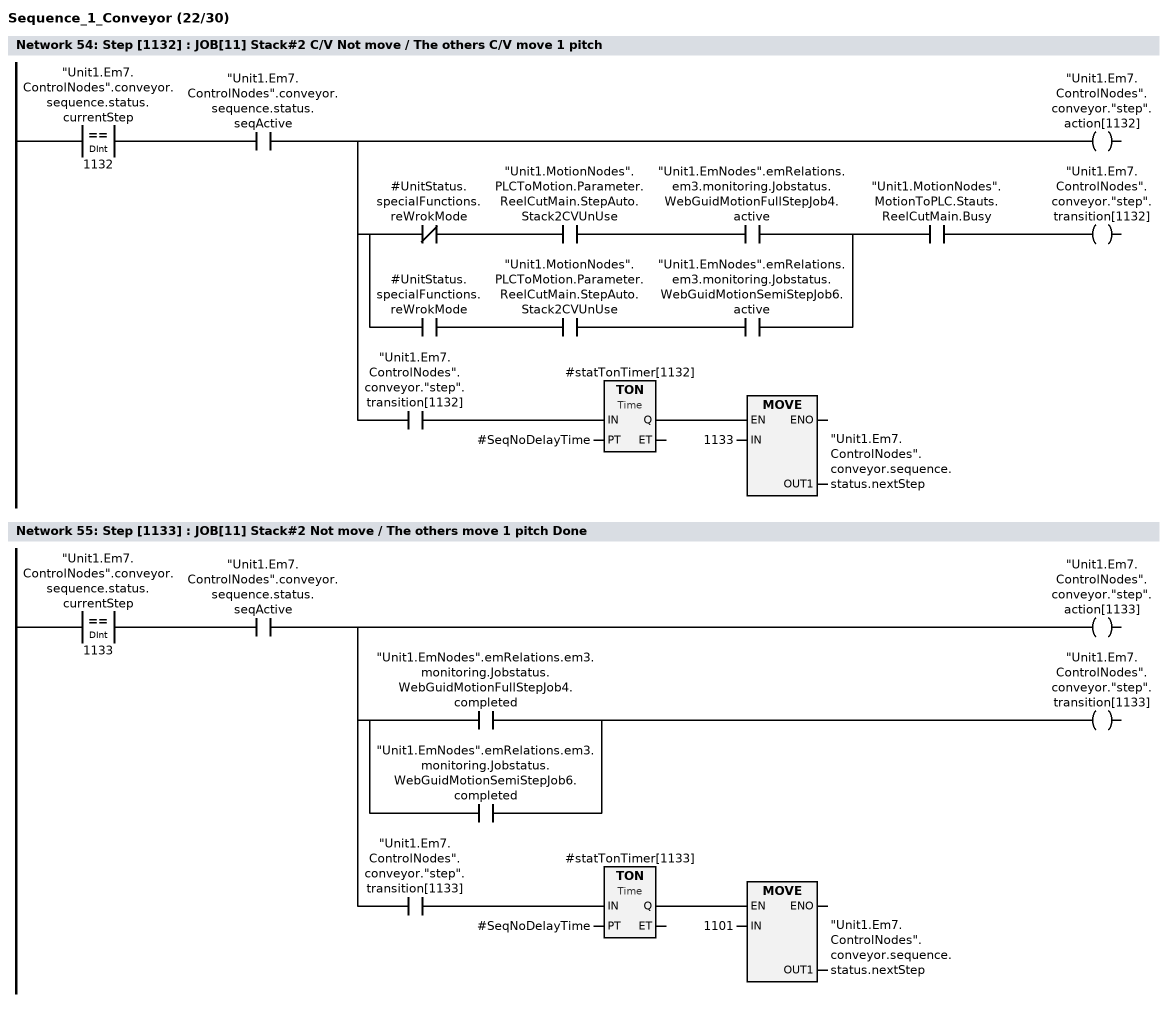
   RUNG wire#powerrail
      { S7_Templates := "SrcType := DInt" } EQ_Contact(in1 := "Unit1.Em7.ControlNodes".conveyor.sequence.status.currentStep, in2 := 1132)
      Contact( "Unit1.Em7.ControlNodes".conveyor.sequence.status.seqActive )
      wire#w1
      Coil( "Unit1.Em7.ControlNodes".conveyor."step".action[1132] )
   END_RUNG
   RUNG wire#w1
      I_Contact( #UnitStatus.specialFunctions.reWrokMode )
      Contact( "Unit1.MotionNodes".PLCToMotion.Parameter.ReelCutMain.StepAuto.Stack2CVUnUse )
      Contact( "Unit1.EmNodes".emRelations.em3.monitoring.Jobstatus.WebGuidMotionFullStepJob4.active )
      wire#w2
      Contact( "Unit1.MotionNodes".MotionToPLC.Stauts.ReelCutMain.Busy )
      Coil( "Unit1.Em7.ControlNodes".conveyor."step".transition[1132] )
   END_RUNG
   RUNG wire#w1
      Contact( #UnitStatus.specialFunctions.reWrokMode )
      Contact( "Unit1.MotionNodes".PLCToMotion.Parameter.ReelCutMain.StepAuto.Stack2CVUnUse )
      Contact( "Unit1.EmNodes".emRelations.em3.monitoring.Jobstatus.WebGuidMotionSemiStepJob6.active )
   END_RUNG wire#w2
   RUNG wire#w1
      Contact( "Unit1.Em7.ControlNodes".conveyor."step".transition[1132] )
      { S7_Templates := "time_type := Time" } #statTonTimer[1132].TON(pt := #SeqNoDelayTime, et =>)
      Move(in := 1133, out1 => "Unit1.Em7.ControlNodes".conveyor.sequence.status.nextStep)
   END_RUNG
   // the same network as SCL:
   "Unit1.Em7.ControlNodes".conveyor."step".action[1132] := ("Unit1.Em7.ControlNodes".conveyor.sequence.status.currentStep = 1132) AND "Unit1.Em7.ControlNodes".conveyor.sequence.status.seqActive;
   "Unit1.Em7.ControlNodes".conveyor."step".transition[1132] := ("Unit1.Em7.ControlNodes".conveyor.sequence.status.currentStep = 1132) AND "Unit1.Em7.ControlNodes".conveyor.sequence.status.seqActive AND ((NOT #UnitStatus.specialFunctions.reWrokMode AND "Unit1.MotionNodes".PLCToMotion.Parameter.ReelCutMain.StepAuto.Stack2CVUnUse AND "Unit1.EmNodes".emRelations.em3.monitoring.Jobstatus.WebGuidMotionFullStepJob4.active) OR (#UnitStatus.specialFunctions.reWrokMode AND "Unit1.MotionNodes".PLCToMotion.Parameter.ReelCutMain.StepAuto.Stack2CVUnUse AND "Unit1.EmNodes".emRelations.em3.monitoring.Jobstatus.WebGuidMotionSemiStepJob6.active)) AND "Unit1.MotionNodes".MotionToPLC.Stauts.ReelCutMain.Busy;
   #statTonTimer[1132].TON(IN := ("Unit1.Em7.ControlNodes".conveyor.sequence.status.currentStep = 1132) AND "Unit1.Em7.ControlNodes".conveyor.sequence.status.seqActive AND "Unit1.Em7.ControlNodes".conveyor."step".transition[1132],
                           PT := #SeqNoDelayTime);
   IF #statTonTimer[1132].Q THEN "Unit1.Em7.ControlNodes".conveyor.sequence.status.nextStep := 1133; END_IF;
END_REGION

REGION Network 55: Step [1133] : JOB[11] Stack#2 Not move / The others move 1 pitch Done
   RUNG wire#powerrail
      { S7_Templates := "SrcType := DInt" } EQ_Contact(in1 := "Unit1.Em7.ControlNodes".conveyor.sequence.status.currentStep, in2 := 1133)
      Contact( "Unit1.Em7.ControlNodes".conveyor.sequence.status.seqActive )
      wire#w1
      Coil( "Unit1.Em7.ControlNodes".conveyor."step".action[1133] )
   END_RUNG
   RUNG wire#w1
      Contact( "Unit1.EmNodes".emRelations.em3.monitoring.Jobstatus.WebGuidMotionFullStepJob4.completed )
      wire#w2
      Coil( "Unit1.Em7.ControlNodes".conveyor."step".transition[1133] )
   END_RUNG
   RUNG wire#w1
      Contact( "Unit1.EmNodes".emRelations.em3.monitoring.Jobstatus.WebGuidMotionSemiStepJob6.completed )
   END_RUNG wire#w2
   RUNG wire#w1
      Contact( "Unit1.Em7.ControlNodes".conveyor."step".transition[1133] )
      { S7_Templates := "time_type := Time" } #statTonTimer[1133].TON(pt := #SeqNoDelayTime, et =>)
      Move(in := 1101, out1 => "Unit1.Em7.ControlNodes".conveyor.sequence.status.nextStep)
   END_RUNG
   // the same network as SCL:
   "Unit1.Em7.ControlNodes".conveyor."step".action[1133] := ("Unit1.Em7.ControlNodes".conveyor.sequence.status.currentStep = 1133) AND "Unit1.Em7.ControlNodes".conveyor.sequence.status.seqActive;
   "Unit1.Em7.ControlNodes".conveyor."step".transition[1133] := ("Unit1.Em7.ControlNodes".conveyor.sequence.status.currentStep = 1133) AND "Unit1.Em7.ControlNodes".conveyor.sequence.status.seqActive AND ("Unit1.EmNodes".emRelations.em3.monitoring.Jobstatus.WebGuidMotionFullStepJob4.completed OR "Unit1.EmNodes".emRelations.em3.monitoring.Jobstatus.WebGuidMotionSemiStepJob6.completed);
   #statTonTimer[1133].TON(IN := ("Unit1.Em7.ControlNodes".conveyor.sequence.status.currentStep = 1133) AND "Unit1.Em7.ControlNodes".conveyor.sequence.status.seqActive AND "Unit1.Em7.ControlNodes".conveyor."step".transition[1133],
                           PT := #SeqNoDelayTime);
   IF #statTonTimer[1133].Q THEN "Unit1.Em7.ControlNodes".conveyor.sequence.status.nextStep := 1101; END_IF;
END_REGION

REGION Network 56: Step [1140] : JOB[11] Stack#1 Work CMD + Stack#2 Work CMD
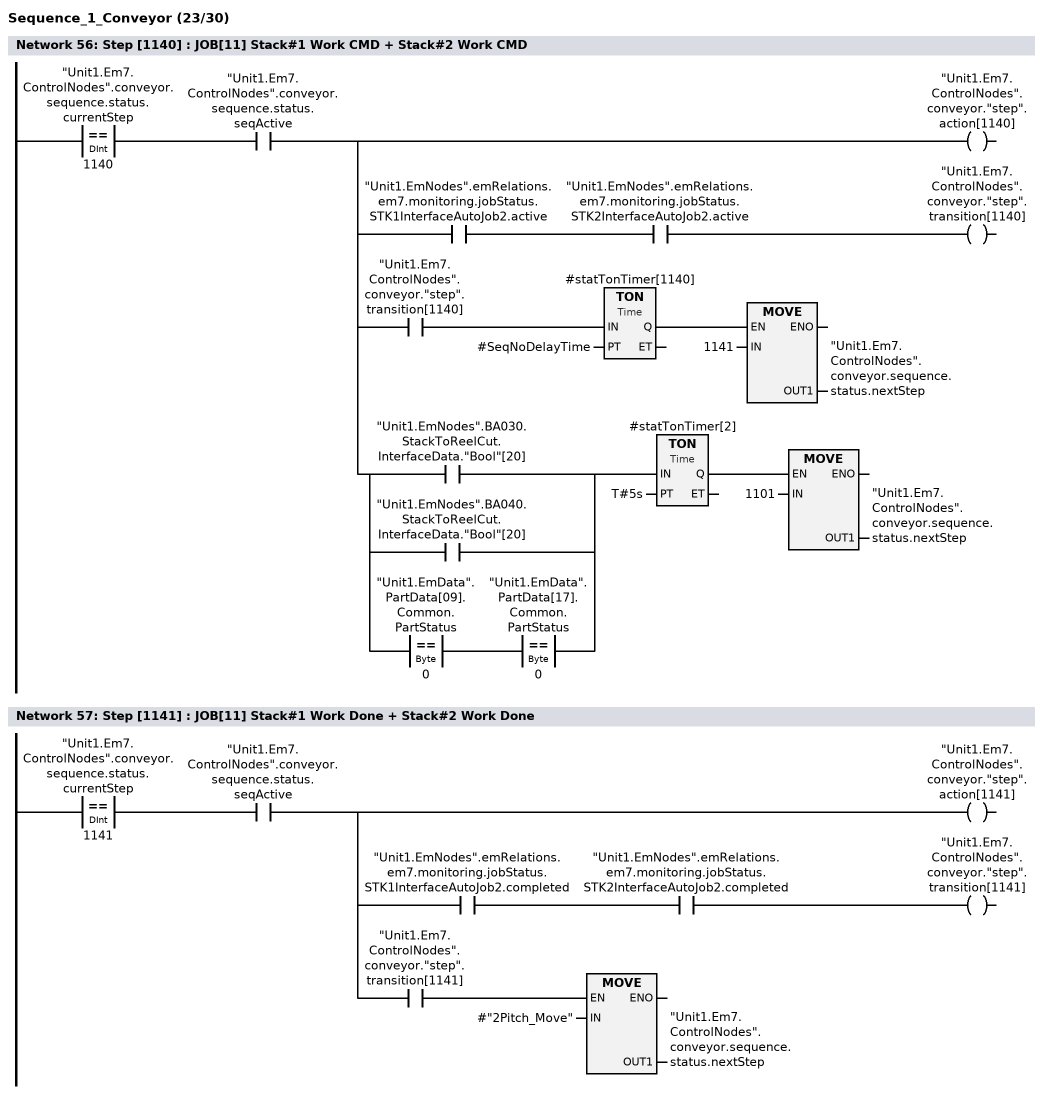
   RUNG wire#powerrail
      { S7_Templates := "SrcType := DInt" } EQ_Contact(in1 := "Unit1.Em7.ControlNodes".conveyor.sequence.status.currentStep, in2 := 1140)
      Contact( "Unit1.Em7.ControlNodes".conveyor.sequence.status.seqActive )
      wire#w1
      Coil( "Unit1.Em7.ControlNodes".conveyor."step".action[1140] )
   END_RUNG
   RUNG wire#w1
      Contact( "Unit1.EmNodes".emRelations.em7.monitoring.jobStatus.STK1InterfaceAutoJob2.active )
      Contact( "Unit1.EmNodes".emRelations.em7.monitoring.jobStatus.STK2InterfaceAutoJob2.active )
      Coil( "Unit1.Em7.ControlNodes".conveyor."step".transition[1140] )
   END_RUNG
   RUNG wire#w1
      Contact( "Unit1.Em7.ControlNodes".conveyor."step".transition[1140] )
      { S7_Templates := "time_type := Time" } #statTonTimer[1140].TON(pt := #SeqNoDelayTime, et =>)
      Move(in := 1141, out1 => "Unit1.Em7.ControlNodes".conveyor.sequence.status.nextStep)
   END_RUNG
   RUNG wire#w1
      Contact( "Unit1.EmNodes".BA030.StackToReelCut.InterfaceData."Bool"[20] )
      wire#w2
      { S7_Templates := "time_type := Time" } #statTonTimer[2].TON(pt := T#5s, et =>)
      Move(in := 1101, out1 => "Unit1.Em7.ControlNodes".conveyor.sequence.status.nextStep)
   END_RUNG
   RUNG wire#w1
      Contact( "Unit1.EmNodes".BA040.StackToReelCut.InterfaceData."Bool"[20] )
   END_RUNG wire#w2
   RUNG wire#w1
      { S7_Templates := "SrcType := Byte" } EQ_Contact(in1 := "Unit1.EmData".PartData[09].Common.PartStatus, in2 := 0)
      { S7_Templates := "SrcType := Byte" } EQ_Contact(in1 := "Unit1.EmData".PartData[17].Common.PartStatus, in2 := 0)
   END_RUNG wire#w2
   // the same network as SCL:
   "Unit1.Em7.ControlNodes".conveyor."step".action[1140] := ("Unit1.Em7.ControlNodes".conveyor.sequence.status.currentStep = 1140) AND "Unit1.Em7.ControlNodes".conveyor.sequence.status.seqActive;
   "Unit1.Em7.ControlNodes".conveyor."step".transition[1140] := ("Unit1.Em7.ControlNodes".conveyor.sequence.status.currentStep = 1140) AND "Unit1.Em7.ControlNodes".conveyor.sequence.status.seqActive AND "Unit1.EmNodes".emRelations.em7.monitoring.jobStatus.STK1InterfaceAutoJob2.active AND "Unit1.EmNodes".emRelations.em7.monitoring.jobStatus.STK2InterfaceAutoJob2.active;
   #statTonTimer[1140].TON(IN := ("Unit1.Em7.ControlNodes".conveyor.sequence.status.currentStep = 1140) AND "Unit1.Em7.ControlNodes".conveyor.sequence.status.seqActive AND "Unit1.Em7.ControlNodes".conveyor."step".transition[1140],
                           PT := #SeqNoDelayTime);
   IF #statTonTimer[1140].Q THEN "Unit1.Em7.ControlNodes".conveyor.sequence.status.nextStep := 1141; END_IF;
   #statTonTimer[2].TON(IN := ("Unit1.Em7.ControlNodes".conveyor.sequence.status.currentStep = 1140) AND "Unit1.Em7.ControlNodes".conveyor.sequence.status.seqActive AND ("Unit1.EmNodes".BA030.StackToReelCut.InterfaceData."Bool"[20] OR "Unit1.EmNodes".BA040.StackToReelCut.InterfaceData."Bool"[20] OR (("Unit1.EmData".PartData[09].Common.PartStatus = 0) AND ("Unit1.EmData".PartData[17].Common.PartStatus = 0))),
                        PT := T#5s);
   IF #statTonTimer[2].Q THEN "Unit1.Em7.ControlNodes".conveyor.sequence.status.nextStep := 1101; END_IF;
END_REGION

REGION Network 57: Step [1141] : JOB[11] Stack#1 Work Done + Stack#2 Work Done
   RUNG wire#powerrail
      { S7_Templates := "SrcType := DInt" } EQ_Contact(in1 := "Unit1.Em7.ControlNodes".conveyor.sequence.status.currentStep, in2 := 1141)
      Contact( "Unit1.Em7.ControlNodes".conveyor.sequence.status.seqActive )
      wire#w1
      Coil( "Unit1.Em7.ControlNodes".conveyor."step".action[1141] )
   END_RUNG
   RUNG wire#w1
      Contact( "Unit1.EmNodes".emRelations.em7.monitoring.jobStatus.STK1InterfaceAutoJob2.completed )
      Contact( "Unit1.EmNodes".emRelations.em7.monitoring.jobStatus.STK2InterfaceAutoJob2.completed )
      Coil( "Unit1.Em7.ControlNodes".conveyor."step".transition[1141] )
   END_RUNG
   RUNG wire#w1
      Contact( "Unit1.Em7.ControlNodes".conveyor."step".transition[1141] )
      Move(in := #"2Pitch_Move", out1 => "Unit1.Em7.ControlNodes".conveyor.sequence.status.nextStep)
   END_RUNG
   // the same network as SCL:
   "Unit1.Em7.ControlNodes".conveyor."step".action[1141] := ("Unit1.Em7.ControlNodes".conveyor.sequence.status.currentStep = 1141) AND "Unit1.Em7.ControlNodes".conveyor.sequence.status.seqActive;
   "Unit1.Em7.ControlNodes".conveyor."step".transition[1141] := ("Unit1.Em7.ControlNodes".conveyor.sequence.status.currentStep = 1141) AND "Unit1.Em7.ControlNodes".conveyor.sequence.status.seqActive AND "Unit1.EmNodes".emRelations.em7.monitoring.jobStatus.STK1InterfaceAutoJob2.completed AND "Unit1.EmNodes".emRelations.em7.monitoring.jobStatus.STK2InterfaceAutoJob2.completed;
   IF ("Unit1.Em7.ControlNodes".conveyor.sequence.status.currentStep = 1141) AND "Unit1.Em7.ControlNodes".conveyor.sequence.status.seqActive AND "Unit1.Em7.ControlNodes".conveyor."step".transition[1141] THEN
       "Unit1.Em7.ControlNodes".conveyor.sequence.status.nextStep := #"2Pitch_Move";
   END_IF;
END_REGION

REGION Network 58: Step [1190] : JOB[11] QR read & Vision Complete Check Before Step End
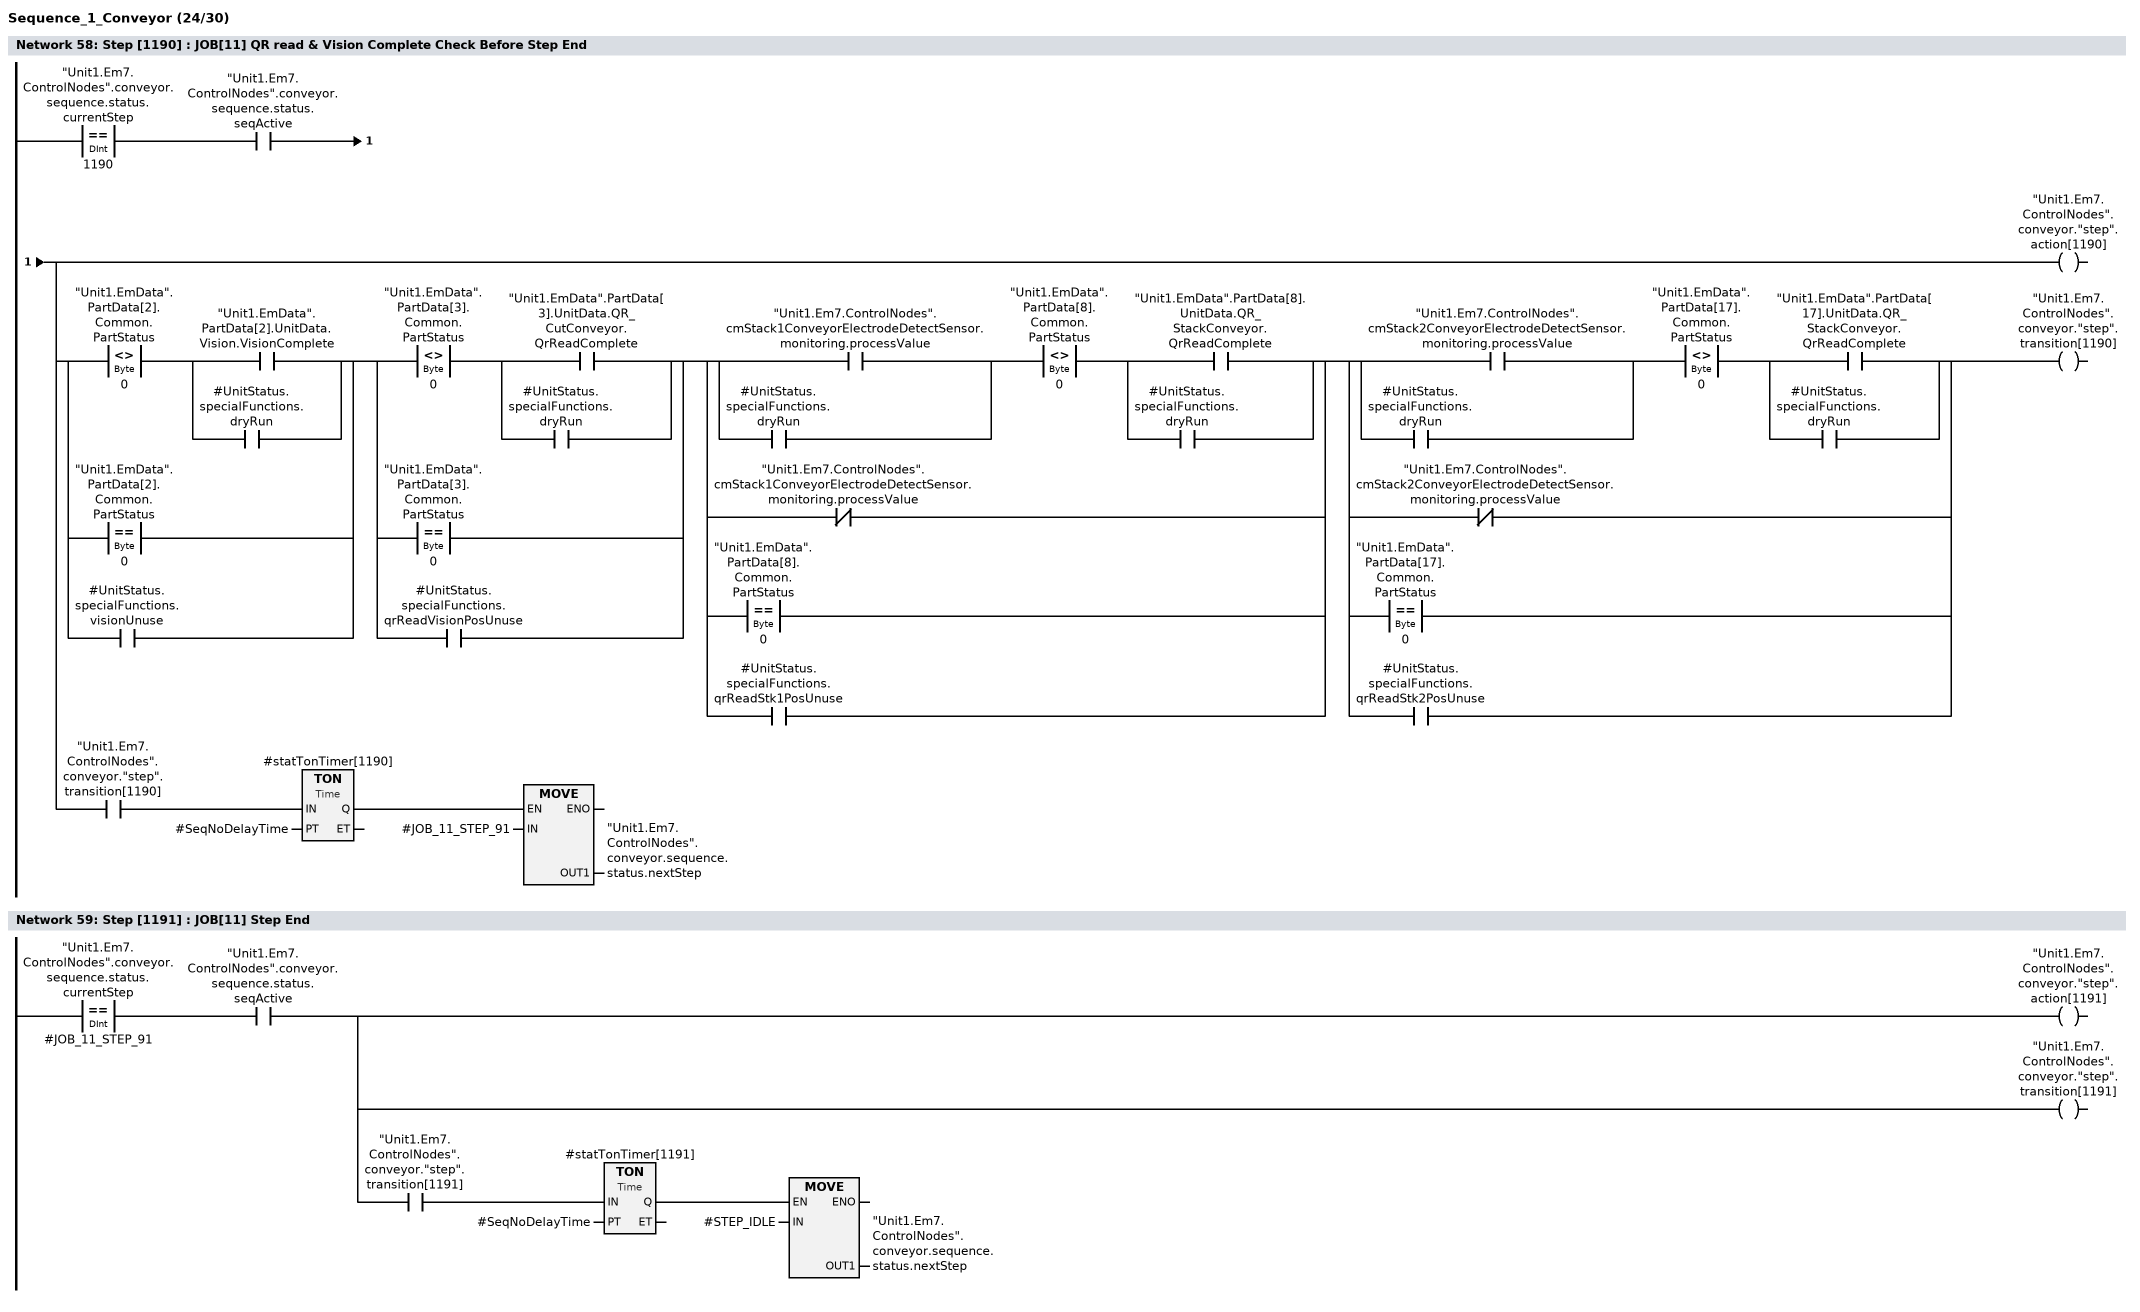
   RUNG wire#powerrail
      { S7_Templates := "SrcType := DInt" } EQ_Contact(in1 := "Unit1.Em7.ControlNodes".conveyor.sequence.status.currentStep, in2 := 1190)
      Contact( "Unit1.Em7.ControlNodes".conveyor.sequence.status.seqActive )
      wire#w1
      Coil( "Unit1.Em7.ControlNodes".conveyor."step".action[1190] )
   END_RUNG
   RUNG wire#w1
      { S7_Templates := "SrcType := Byte" } NE_Contact(in1 := "Unit1.EmData".PartData[2].Common.PartStatus, in2 := 0)
      wire#w2
      Contact( "Unit1.EmData".PartData[2].UnitData.Vision.VisionComplete )
      wire#w3
      { S7_Templates := "SrcType := Byte" } NE_Contact(in1 := "Unit1.EmData".PartData[3].Common.PartStatus, in2 := 0)
      wire#w4
      Contact( "Unit1.EmData".PartData[3].UnitData.QR_CutConveyor.QrReadComplete )
      wire#w5
      Contact( "Unit1.Em7.ControlNodes".cmStack1ConveyorElectrodeDetectSensor.monitoring.processValue )
      wire#w6
      { S7_Templates := "SrcType := Byte" } NE_Contact(in1 := "Unit1.EmData".PartData[8].Common.PartStatus, in2 := 0)
      wire#w7
      Contact( "Unit1.EmData".PartData[8].UnitData.QR_StackConveyor.QrReadComplete )
      wire#w8
      Contact( "Unit1.Em7.ControlNodes".cmStack2ConveyorElectrodeDetectSensor.monitoring.processValue )
      wire#w9
      { S7_Templates := "SrcType := Byte" } NE_Contact(in1 := "Unit1.EmData".PartData[17].Common.PartStatus, in2 := 0)
      wire#w10
      Contact( "Unit1.EmData".PartData[17].UnitData.QR_StackConveyor.QrReadComplete )
      wire#w11
      Coil( "Unit1.Em7.ControlNodes".conveyor."step".transition[1190] )
   END_RUNG
   RUNG wire#w2
      Contact( #UnitStatus.specialFunctions.dryRun )
   END_RUNG wire#w3
   RUNG wire#w1
      { S7_Templates := "SrcType := Byte" } EQ_Contact(in1 := "Unit1.EmData".PartData[2].Common.PartStatus, in2 := 0)
   END_RUNG wire#w3
   RUNG wire#w1
      Contact( #UnitStatus.specialFunctions.visionUnuse )
   END_RUNG wire#w3
   RUNG wire#w4
      Contact( #UnitStatus.specialFunctions.dryRun )
   END_RUNG wire#w5
   RUNG wire#w3
      { S7_Templates := "SrcType := Byte" } EQ_Contact(in1 := "Unit1.EmData".PartData[3].Common.PartStatus, in2 := 0)
   END_RUNG wire#w5
   RUNG wire#w3
      Contact( #UnitStatus.specialFunctions.qrReadVisionPosUnuse )
   END_RUNG wire#w5
   RUNG wire#w5
      Contact( #UnitStatus.specialFunctions.dryRun )
   END_RUNG wire#w6
   RUNG wire#w7
      Contact( #UnitStatus.specialFunctions.dryRun )
   END_RUNG wire#w8
   RUNG wire#w5
      I_Contact( "Unit1.Em7.ControlNodes".cmStack1ConveyorElectrodeDetectSensor.monitoring.processValue )
   END_RUNG wire#w8
   RUNG wire#w5
      { S7_Templates := "SrcType := Byte" } EQ_Contact(in1 := "Unit1.EmData".PartData[8].Common.PartStatus, in2 := 0)
   END_RUNG wire#w8
   RUNG wire#w5
      Contact( #UnitStatus.specialFunctions.qrReadStk1PosUnuse )
   END_RUNG wire#w8
   RUNG wire#w8
      Contact( #UnitStatus.specialFunctions.dryRun )
   END_RUNG wire#w9
   RUNG wire#w10
      Contact( #UnitStatus.specialFunctions.dryRun )
   END_RUNG wire#w11
   RUNG wire#w8
      I_Contact( "Unit1.Em7.ControlNodes".cmStack2ConveyorElectrodeDetectSensor.monitoring.processValue )
   END_RUNG wire#w11
   RUNG wire#w8
      { S7_Templates := "SrcType := Byte" } EQ_Contact(in1 := "Unit1.EmData".PartData[17].Common.PartStatus, in2 := 0)
   END_RUNG wire#w11
   RUNG wire#w8
      Contact( #UnitStatus.specialFunctions.qrReadStk2PosUnuse )
   END_RUNG wire#w11
   RUNG wire#w1
      Contact( "Unit1.Em7.ControlNodes".conveyor."step".transition[1190] )
      { S7_Templates := "time_type := Time" } #statTonTimer[1190].TON(pt := #SeqNoDelayTime, et =>)
      Move(in := #JOB_11_STEP_91, out1 => "Unit1.Em7.ControlNodes".conveyor.sequence.status.nextStep)
   END_RUNG
   // the same network as SCL:
   "Unit1.Em7.ControlNodes".conveyor."step".action[1190] := ("Unit1.Em7.ControlNodes".conveyor.sequence.status.currentStep = 1190) AND "Unit1.Em7.ControlNodes".conveyor.sequence.status.seqActive;
   "Unit1.Em7.ControlNodes".conveyor."step".transition[1190] := ("Unit1.Em7.ControlNodes".conveyor.sequence.status.currentStep = 1190) AND "Unit1.Em7.ControlNodes".conveyor.sequence.status.seqActive AND ((("Unit1.EmData".PartData[2].Common.PartStatus <> 0) AND ("Unit1.EmData".PartData[2].UnitData.Vision.VisionComplete OR #UnitStatus.specialFunctions.dryRun)) OR ("Unit1.EmData".PartData[2].Common.PartStatus = 0) OR #UnitStatus.specialFunctions.visionUnuse) AND ((("Unit1.EmData".PartData[3].Common.PartStatus <> 0) AND ("Unit1.EmData".PartData[3].UnitData.QR_CutConveyor.QrReadComplete OR #UnitStatus.specialFunctions.dryRun)) OR ("Unit1.EmData".PartData[3].Common.PartStatus = 0) OR #UnitStatus.specialFunctions.qrReadVisionPosUnuse) AND ((("Unit1.Em7.ControlNodes".cmStack1ConveyorElectrodeDetectSensor.monitoring.processValue OR #UnitStatus.specialFunctions.dryRun) AND ("Unit1.EmData".PartData[8].Common.PartStatus <> 0) AND ("Unit1.EmData".PartData[8].UnitData.QR_StackConveyor.QrReadComplete OR #UnitStatus.specialFunctions.dryRun)) OR NOT "Unit1.Em7.ControlNodes".cmStack1ConveyorElectrodeDetectSensor.monitoring.processValue OR ("Unit1.EmData".PartData[8].Common.PartStatus = 0) OR #UnitStatus.specialFunctions.qrReadStk1PosUnuse) AND ((("Unit1.Em7.ControlNodes".cmStack2ConveyorElectrodeDetectSensor.monitoring.processValue OR #UnitStatus.specialFunctions.dryRun) AND ("Unit1.EmData".PartData[17].Common.PartStatus <> 0) AND ("Unit1.EmData".PartData[17].UnitData.QR_StackConveyor.QrReadComplete OR #UnitStatus.specialFunctions.dryRun)) OR NOT "Unit1.Em7.ControlNodes".cmStack2ConveyorElectrodeDetectSensor.monitoring.processValue OR ("Unit1.EmData".PartData[17].Common.PartStatus = 0) OR #UnitStatus.specialFunctions.qrReadStk2PosUnuse);
   #statTonTimer[1190].TON(IN := ("Unit1.Em7.ControlNodes".conveyor.sequence.status.currentStep = 1190) AND "Unit1.Em7.ControlNodes".conveyor.sequence.status.seqActive AND "Unit1.Em7.ControlNodes".conveyor."step".transition[1190],
                           PT := #SeqNoDelayTime);
   IF #statTonTimer[1190].Q THEN
       "Unit1.Em7.ControlNodes".conveyor.sequence.status.nextStep := #JOB_11_STEP_91;
   END_IF;
END_REGION

REGION Network 59: Step [1191] : JOB[11] Step End
   RUNG wire#powerrail
      { S7_Templates := "SrcType := DInt" } EQ_Contact(in1 := "Unit1.Em7.ControlNodes".conveyor.sequence.status.currentStep, in2 := #JOB_11_STEP_91)
      Contact( "Unit1.Em7.ControlNodes".conveyor.sequence.status.seqActive )
      wire#w1
      Coil( "Unit1.Em7.ControlNodes".conveyor."step".action[1191] )
   END_RUNG
   RUNG wire#w1
      Coil( "Unit1.Em7.ControlNodes".conveyor."step".transition[1191] )
   END_RUNG
   RUNG wire#w1
      Contact( "Unit1.Em7.ControlNodes".conveyor."step".transition[1191] )
      { S7_Templates := "time_type := Time" } #statTonTimer[1191].TON(pt := #SeqNoDelayTime, et =>)
      Move(in := #STEP_IDLE, out1 => "Unit1.Em7.ControlNodes".conveyor.sequence.status.nextStep)
   END_RUNG
   // the same network as SCL:
   "Unit1.Em7.ControlNodes".conveyor."step".action[1191] := ("Unit1.Em7.ControlNodes".conveyor.sequence.status.currentStep = #JOB_11_STEP_91) AND "Unit1.Em7.ControlNodes".conveyor.sequence.status.seqActive;
   "Unit1.Em7.ControlNodes".conveyor."step".transition[1191] := ("Unit1.Em7.ControlNodes".conveyor.sequence.status.currentStep = #JOB_11_STEP_91) AND "Unit1.Em7.ControlNodes".conveyor.sequence.status.seqActive;
   #statTonTimer[1191].TON(IN := ("Unit1.Em7.ControlNodes".conveyor.sequence.status.currentStep = #JOB_11_STEP_91) AND "Unit1.Em7.ControlNodes".conveyor.sequence.status.seqActive AND "Unit1.Em7.ControlNodes".conveyor."step".transition[1191],
                           PT := #SeqNoDelayTime);
   IF #statTonTimer[1191].Q THEN
       "Unit1.Em7.ControlNodes".conveyor.sequence.status.nextStep := #STEP_IDLE;
   END_IF;
END_REGION

REGION Network 60: ******************** JOB[12] Stack Gauge R&R Auto ********************
END_REGION

REGION Network 61: Step[1201] : JOB[12] Condition
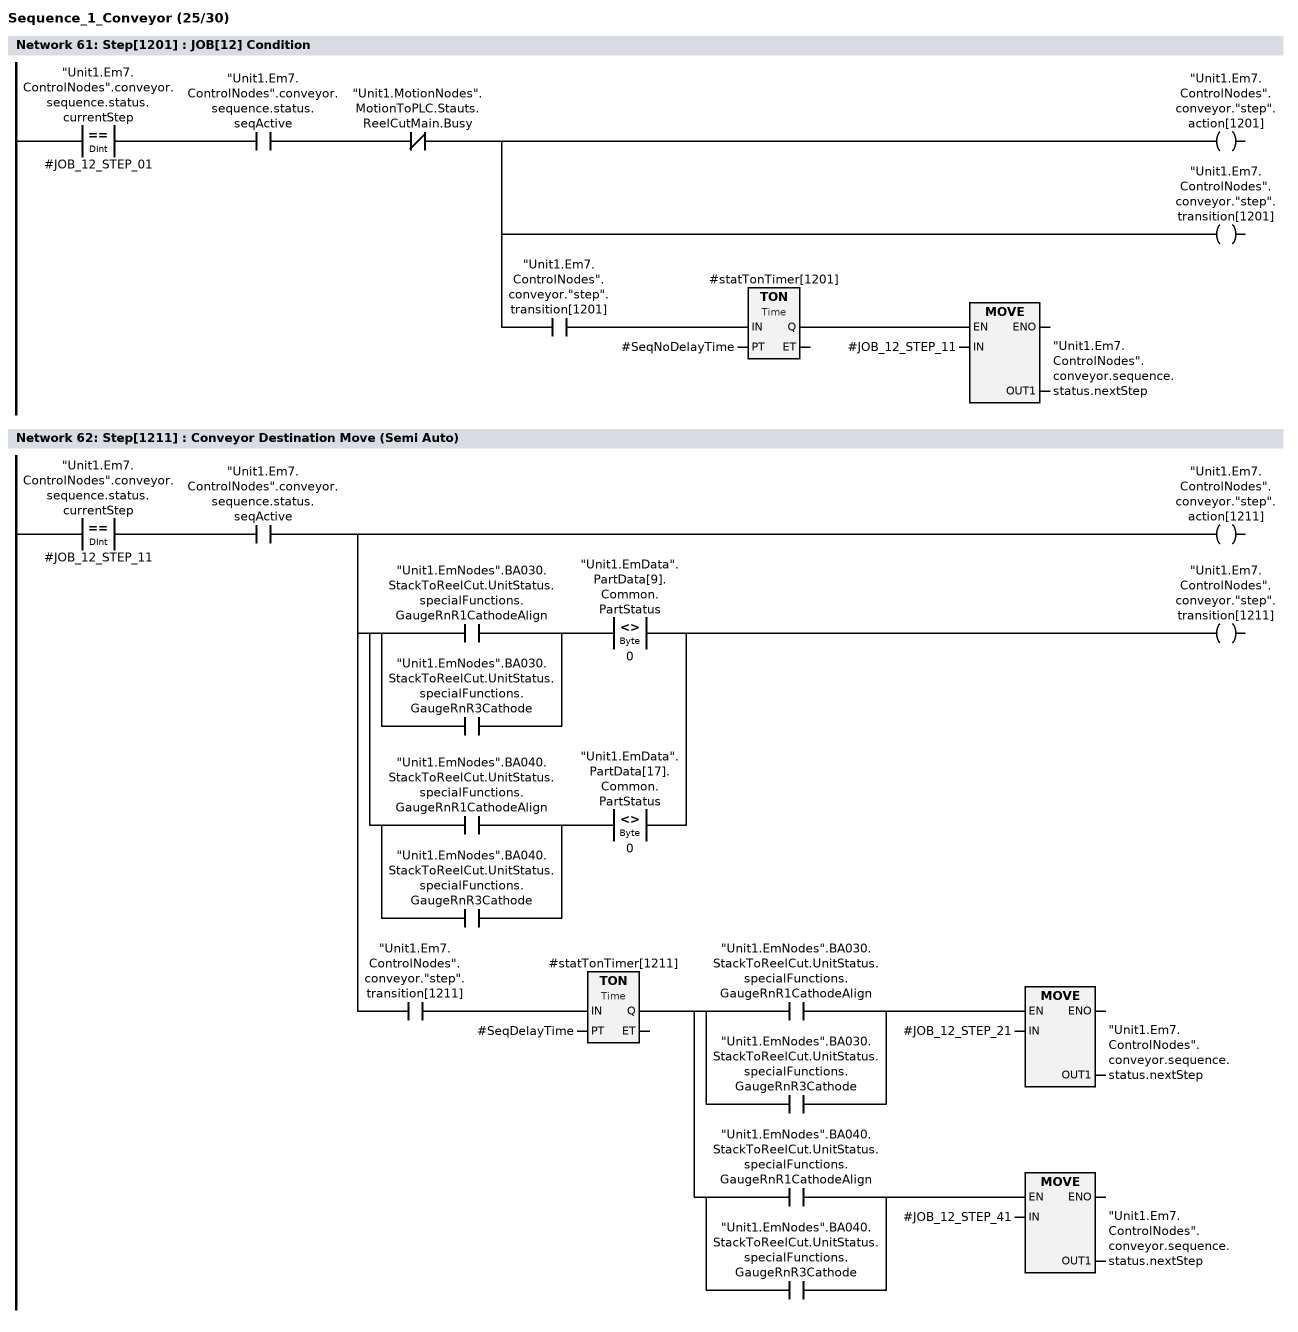
   RUNG wire#powerrail
      { S7_Templates := "SrcType := DInt" } EQ_Contact(in1 := "Unit1.Em7.ControlNodes".conveyor.sequence.status.currentStep, in2 := #JOB_12_STEP_01)
      Contact( "Unit1.Em7.ControlNodes".conveyor.sequence.status.seqActive )
      I_Contact( "Unit1.MotionNodes".MotionToPLC.Stauts.ReelCutMain.Busy )
      wire#w1
      Coil( "Unit1.Em7.ControlNodes".conveyor."step".action[1201] )
   END_RUNG
   RUNG wire#w1
      Coil( "Unit1.Em7.ControlNodes".conveyor."step".transition[1201] )
   END_RUNG
   RUNG wire#w1
      Contact( "Unit1.Em7.ControlNodes".conveyor."step".transition[1201] )
      { S7_Templates := "time_type := Time" } #statTonTimer[1201].TON(pt := #SeqNoDelayTime, et =>)
      Move(in := #JOB_12_STEP_11, out1 => "Unit1.Em7.ControlNodes".conveyor.sequence.status.nextStep)
   END_RUNG
   // the same network as SCL:
   "Unit1.Em7.ControlNodes".conveyor."step".action[1201] := ("Unit1.Em7.ControlNodes".conveyor.sequence.status.currentStep = #JOB_12_STEP_01) AND "Unit1.Em7.ControlNodes".conveyor.sequence.status.seqActive AND NOT "Unit1.MotionNodes".MotionToPLC.Stauts.ReelCutMain.Busy;
   "Unit1.Em7.ControlNodes".conveyor."step".transition[1201] := ("Unit1.Em7.ControlNodes".conveyor.sequence.status.currentStep = #JOB_12_STEP_01) AND "Unit1.Em7.ControlNodes".conveyor.sequence.status.seqActive AND NOT "Unit1.MotionNodes".MotionToPLC.Stauts.ReelCutMain.Busy;
   #statTonTimer[1201].TON(IN := ("Unit1.Em7.ControlNodes".conveyor.sequence.status.currentStep = #JOB_12_STEP_01) AND "Unit1.Em7.ControlNodes".conveyor.sequence.status.seqActive AND NOT "Unit1.MotionNodes".MotionToPLC.Stauts.ReelCutMain.Busy AND "Unit1.Em7.ControlNodes".conveyor."step".transition[1201],
                           PT := #SeqNoDelayTime);
   IF #statTonTimer[1201].Q THEN
       "Unit1.Em7.ControlNodes".conveyor.sequence.status.nextStep := #JOB_12_STEP_11;
   END_IF;
END_REGION

REGION Network 62: Step[1211] : Conveyor Destination Move (Semi Auto)
   RUNG wire#powerrail
      { S7_Templates := "SrcType := DInt" } EQ_Contact(in1 := "Unit1.Em7.ControlNodes".conveyor.sequence.status.currentStep, in2 := #JOB_12_STEP_11)
      Contact( "Unit1.Em7.ControlNodes".conveyor.sequence.status.seqActive )
      wire#w1
      Coil( "Unit1.Em7.ControlNodes".conveyor."step".action[1211] )
   END_RUNG
   RUNG wire#w1
      Contact( "Unit1.EmNodes".BA030.StackToReelCut.UnitStatus.specialFunctions.GaugeRnR1CathodeAlign )
      wire#w2
      { S7_Templates := "SrcType := Byte" } NE_Contact(in1 := "Unit1.EmData".PartData[9].Common.PartStatus, in2 := 0)
      wire#w3
      Coil( "Unit1.Em7.ControlNodes".conveyor."step".transition[1211] )
   END_RUNG
   RUNG wire#w1
      Contact( "Unit1.EmNodes".BA030.StackToReelCut.UnitStatus.specialFunctions.GaugeRnR3Cathode )
   END_RUNG wire#w2
   RUNG wire#w1
      Contact( "Unit1.EmNodes".BA040.StackToReelCut.UnitStatus.specialFunctions.GaugeRnR1CathodeAlign )
      wire#w4
      { S7_Templates := "SrcType := Byte" } NE_Contact(in1 := "Unit1.EmData".PartData[17].Common.PartStatus, in2 := 0)
   END_RUNG wire#w3
   RUNG wire#w1
      Contact( "Unit1.EmNodes".BA040.StackToReelCut.UnitStatus.specialFunctions.GaugeRnR3Cathode )
   END_RUNG wire#w4
   RUNG wire#w1
      Contact( "Unit1.Em7.ControlNodes".conveyor."step".transition[1211] )
      { S7_Templates := "time_type := Time" } #statTonTimer[1211].TON(pt := #SeqDelayTime, et =>)
      wire#w5
      Contact( "Unit1.EmNodes".BA030.StackToReelCut.UnitStatus.specialFunctions.GaugeRnR1CathodeAlign )
      wire#w6
      Move(in := #JOB_12_STEP_21, out1 => "Unit1.Em7.ControlNodes".conveyor.sequence.status.nextStep)
   END_RUNG
   RUNG wire#w5
      Contact( "Unit1.EmNodes".BA030.StackToReelCut.UnitStatus.specialFunctions.GaugeRnR3Cathode )
   END_RUNG wire#w6
   RUNG wire#w5
      Contact( "Unit1.EmNodes".BA040.StackToReelCut.UnitStatus.specialFunctions.GaugeRnR1CathodeAlign )
      wire#w7
      Move(in := #JOB_12_STEP_41, out1 => "Unit1.Em7.ControlNodes".conveyor.sequence.status.nextStep)
   END_RUNG
   RUNG wire#w5
      Contact( "Unit1.EmNodes".BA040.StackToReelCut.UnitStatus.specialFunctions.GaugeRnR3Cathode )
   END_RUNG wire#w7
   // the same network as SCL:
   "Unit1.Em7.ControlNodes".conveyor."step".action[1211] := ("Unit1.Em7.ControlNodes".conveyor.sequence.status.currentStep = #JOB_12_STEP_11) AND "Unit1.Em7.ControlNodes".conveyor.sequence.status.seqActive;
   "Unit1.Em7.ControlNodes".conveyor."step".transition[1211] := ("Unit1.Em7.ControlNodes".conveyor.sequence.status.currentStep = #JOB_12_STEP_11) AND "Unit1.Em7.ControlNodes".conveyor.sequence.status.seqActive AND ((("Unit1.EmNodes".BA030.StackToReelCut.UnitStatus.specialFunctions.GaugeRnR1CathodeAlign OR "Unit1.EmNodes".BA030.StackToReelCut.UnitStatus.specialFunctions.GaugeRnR3Cathode) AND ("Unit1.EmData".PartData[9].Common.PartStatus <> 0)) OR (("Unit1.EmNodes".BA040.StackToReelCut.UnitStatus.specialFunctions.GaugeRnR1CathodeAlign OR "Unit1.EmNodes".BA040.StackToReelCut.UnitStatus.specialFunctions.GaugeRnR3Cathode) AND ("Unit1.EmData".PartData[17].Common.PartStatus <> 0)));
   #statTonTimer[1211].TON(IN := ("Unit1.Em7.ControlNodes".conveyor.sequence.status.currentStep = #JOB_12_STEP_11) AND "Unit1.Em7.ControlNodes".conveyor.sequence.status.seqActive AND "Unit1.Em7.ControlNodes".conveyor."step".transition[1211],
                           PT := #SeqDelayTime);
   IF #statTonTimer[1211].Q AND ("Unit1.EmNodes".BA030.StackToReelCut.UnitStatus.specialFunctions.GaugeRnR1CathodeAlign OR "Unit1.EmNodes".BA030.StackToReelCut.UnitStatus.specialFunctions.GaugeRnR3Cathode) THEN
       "Unit1.Em7.ControlNodes".conveyor.sequence.status.nextStep := #JOB_12_STEP_21;
   END_IF;
   IF #statTonTimer[1211].Q AND ("Unit1.EmNodes".BA040.StackToReelCut.UnitStatus.specialFunctions.GaugeRnR1CathodeAlign OR "Unit1.EmNodes".BA040.StackToReelCut.UnitStatus.specialFunctions.GaugeRnR3Cathode) THEN
       "Unit1.Em7.ControlNodes".conveyor.sequence.status.nextStep := #JOB_12_STEP_41;
   END_IF;
END_REGION

REGION Network 63: Step[1221] : Call Stack#1 BA030 Work CMD
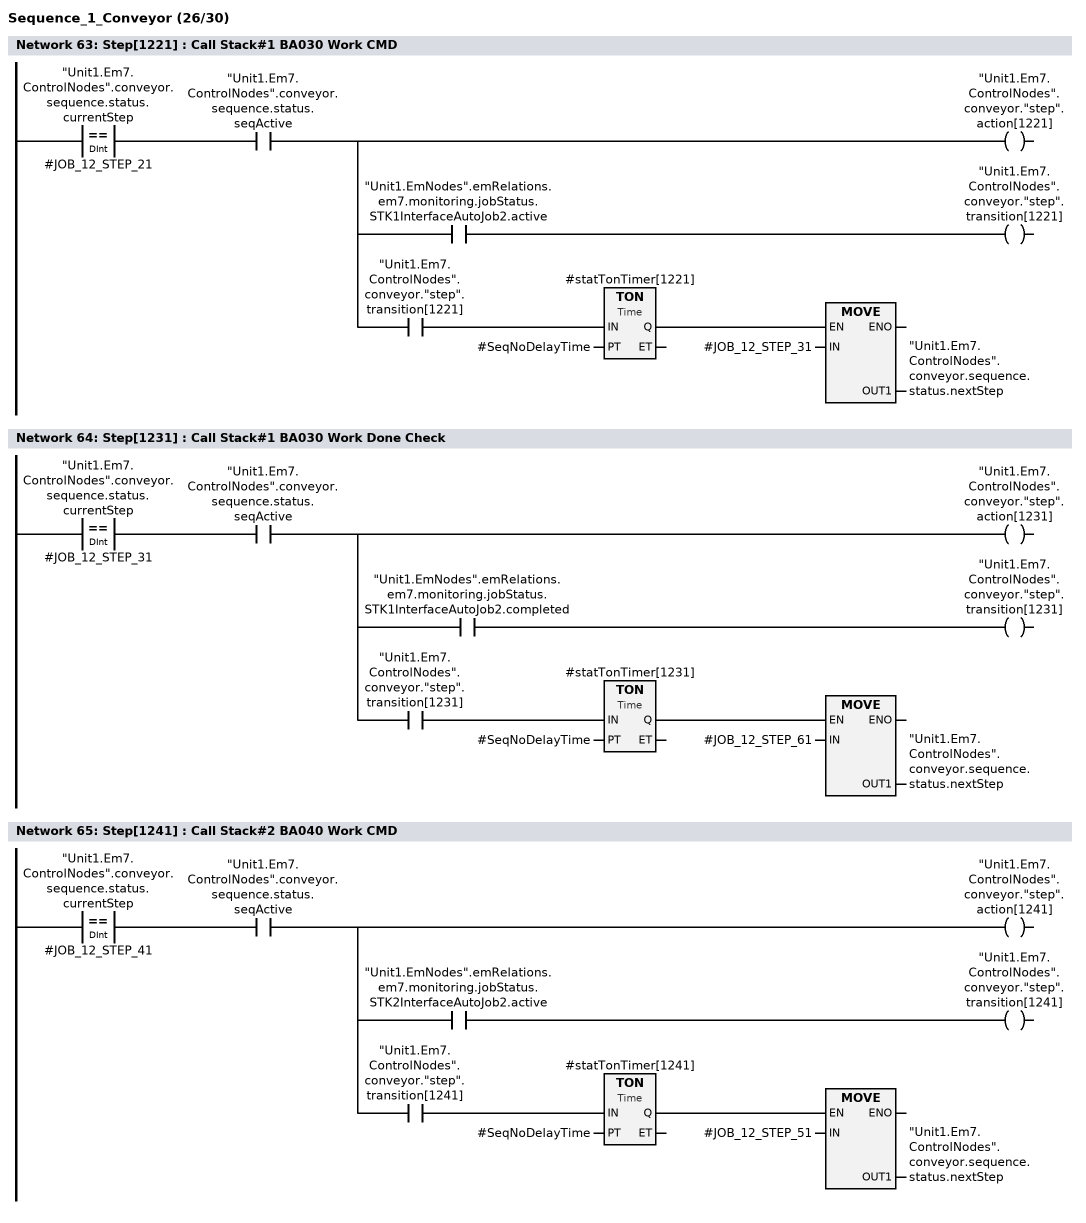
   RUNG wire#powerrail
      { S7_Templates := "SrcType := DInt" } EQ_Contact(in1 := "Unit1.Em7.ControlNodes".conveyor.sequence.status.currentStep, in2 := #JOB_12_STEP_21)
      Contact( "Unit1.Em7.ControlNodes".conveyor.sequence.status.seqActive )
      wire#w1
      Coil( "Unit1.Em7.ControlNodes".conveyor."step".action[1221] )
   END_RUNG
   RUNG wire#w1
      Contact( "Unit1.EmNodes".emRelations.em7.monitoring.jobStatus.STK1InterfaceAutoJob2.active )
      Coil( "Unit1.Em7.ControlNodes".conveyor."step".transition[1221] )
   END_RUNG
   RUNG wire#w1
      Contact( "Unit1.Em7.ControlNodes".conveyor."step".transition[1221] )
      { S7_Templates := "time_type := Time" } #statTonTimer[1221].TON(pt := #SeqNoDelayTime, et =>)
      Move(in := #JOB_12_STEP_31, out1 => "Unit1.Em7.ControlNodes".conveyor.sequence.status.nextStep)
   END_RUNG
   // the same network as SCL:
   "Unit1.Em7.ControlNodes".conveyor."step".action[1221] := ("Unit1.Em7.ControlNodes".conveyor.sequence.status.currentStep = #JOB_12_STEP_21) AND "Unit1.Em7.ControlNodes".conveyor.sequence.status.seqActive;
   "Unit1.Em7.ControlNodes".conveyor."step".transition[1221] := ("Unit1.Em7.ControlNodes".conveyor.sequence.status.currentStep = #JOB_12_STEP_21) AND "Unit1.Em7.ControlNodes".conveyor.sequence.status.seqActive AND "Unit1.EmNodes".emRelations.em7.monitoring.jobStatus.STK1InterfaceAutoJob2.active;
   #statTonTimer[1221].TON(IN := ("Unit1.Em7.ControlNodes".conveyor.sequence.status.currentStep = #JOB_12_STEP_21) AND "Unit1.Em7.ControlNodes".conveyor.sequence.status.seqActive AND "Unit1.Em7.ControlNodes".conveyor."step".transition[1221],
                           PT := #SeqNoDelayTime);
   IF #statTonTimer[1221].Q THEN
       "Unit1.Em7.ControlNodes".conveyor.sequence.status.nextStep := #JOB_12_STEP_31;
   END_IF;
END_REGION

REGION Network 64: Step[1231] : Call Stack#1 BA030 Work Done Check
   RUNG wire#powerrail
      { S7_Templates := "SrcType := DInt" } EQ_Contact(in1 := "Unit1.Em7.ControlNodes".conveyor.sequence.status.currentStep, in2 := #JOB_12_STEP_31)
      Contact( "Unit1.Em7.ControlNodes".conveyor.sequence.status.seqActive )
      wire#w1
      Coil( "Unit1.Em7.ControlNodes".conveyor."step".action[1231] )
   END_RUNG
   RUNG wire#w1
      Contact( "Unit1.EmNodes".emRelations.em7.monitoring.jobStatus.STK1InterfaceAutoJob2.completed )
      Coil( "Unit1.Em7.ControlNodes".conveyor."step".transition[1231] )
   END_RUNG
   RUNG wire#w1
      Contact( "Unit1.Em7.ControlNodes".conveyor."step".transition[1231] )
      { S7_Templates := "time_type := Time" } #statTonTimer[1231].TON(pt := #SeqNoDelayTime, et =>)
      Move(in := #JOB_12_STEP_61, out1 => "Unit1.Em7.ControlNodes".conveyor.sequence.status.nextStep)
   END_RUNG
   // the same network as SCL:
   "Unit1.Em7.ControlNodes".conveyor."step".action[1231] := ("Unit1.Em7.ControlNodes".conveyor.sequence.status.currentStep = #JOB_12_STEP_31) AND "Unit1.Em7.ControlNodes".conveyor.sequence.status.seqActive;
   "Unit1.Em7.ControlNodes".conveyor."step".transition[1231] := ("Unit1.Em7.ControlNodes".conveyor.sequence.status.currentStep = #JOB_12_STEP_31) AND "Unit1.Em7.ControlNodes".conveyor.sequence.status.seqActive AND "Unit1.EmNodes".emRelations.em7.monitoring.jobStatus.STK1InterfaceAutoJob2.completed;
   #statTonTimer[1231].TON(IN := ("Unit1.Em7.ControlNodes".conveyor.sequence.status.currentStep = #JOB_12_STEP_31) AND "Unit1.Em7.ControlNodes".conveyor.sequence.status.seqActive AND "Unit1.Em7.ControlNodes".conveyor."step".transition[1231],
                           PT := #SeqNoDelayTime);
   IF #statTonTimer[1231].Q THEN
       "Unit1.Em7.ControlNodes".conveyor.sequence.status.nextStep := #JOB_12_STEP_61;
   END_IF;
END_REGION

REGION Network 65: Step[1241] : Call Stack#2 BA040 Work CMD
   RUNG wire#powerrail
      { S7_Templates := "SrcType := DInt" } EQ_Contact(in1 := "Unit1.Em7.ControlNodes".conveyor.sequence.status.currentStep, in2 := #JOB_12_STEP_41)
      Contact( "Unit1.Em7.ControlNodes".conveyor.sequence.status.seqActive )
      wire#w1
      Coil( "Unit1.Em7.ControlNodes".conveyor."step".action[1241] )
   END_RUNG
   RUNG wire#w1
      Contact( "Unit1.EmNodes".emRelations.em7.monitoring.jobStatus.STK2InterfaceAutoJob2.active )
      Coil( "Unit1.Em7.ControlNodes".conveyor."step".transition[1241] )
   END_RUNG
   RUNG wire#w1
      Contact( "Unit1.Em7.ControlNodes".conveyor."step".transition[1241] )
      { S7_Templates := "time_type := Time" } #statTonTimer[1241].TON(pt := #SeqNoDelayTime, et =>)
      Move(in := #JOB_12_STEP_51, out1 => "Unit1.Em7.ControlNodes".conveyor.sequence.status.nextStep)
   END_RUNG
   // the same network as SCL:
   "Unit1.Em7.ControlNodes".conveyor."step".action[1241] := ("Unit1.Em7.ControlNodes".conveyor.sequence.status.currentStep = #JOB_12_STEP_41) AND "Unit1.Em7.ControlNodes".conveyor.sequence.status.seqActive;
   "Unit1.Em7.ControlNodes".conveyor."step".transition[1241] := ("Unit1.Em7.ControlNodes".conveyor.sequence.status.currentStep = #JOB_12_STEP_41) AND "Unit1.Em7.ControlNodes".conveyor.sequence.status.seqActive AND "Unit1.EmNodes".emRelations.em7.monitoring.jobStatus.STK2InterfaceAutoJob2.active;
   #statTonTimer[1241].TON(IN := ("Unit1.Em7.ControlNodes".conveyor.sequence.status.currentStep = #JOB_12_STEP_41) AND "Unit1.Em7.ControlNodes".conveyor.sequence.status.seqActive AND "Unit1.Em7.ControlNodes".conveyor."step".transition[1241],
                           PT := #SeqNoDelayTime);
   IF #statTonTimer[1241].Q THEN
       "Unit1.Em7.ControlNodes".conveyor.sequence.status.nextStep := #JOB_12_STEP_51;
   END_IF;
END_REGION

REGION Network 66: Step[1251] : Call Stack#2 BA040 Work Done Check
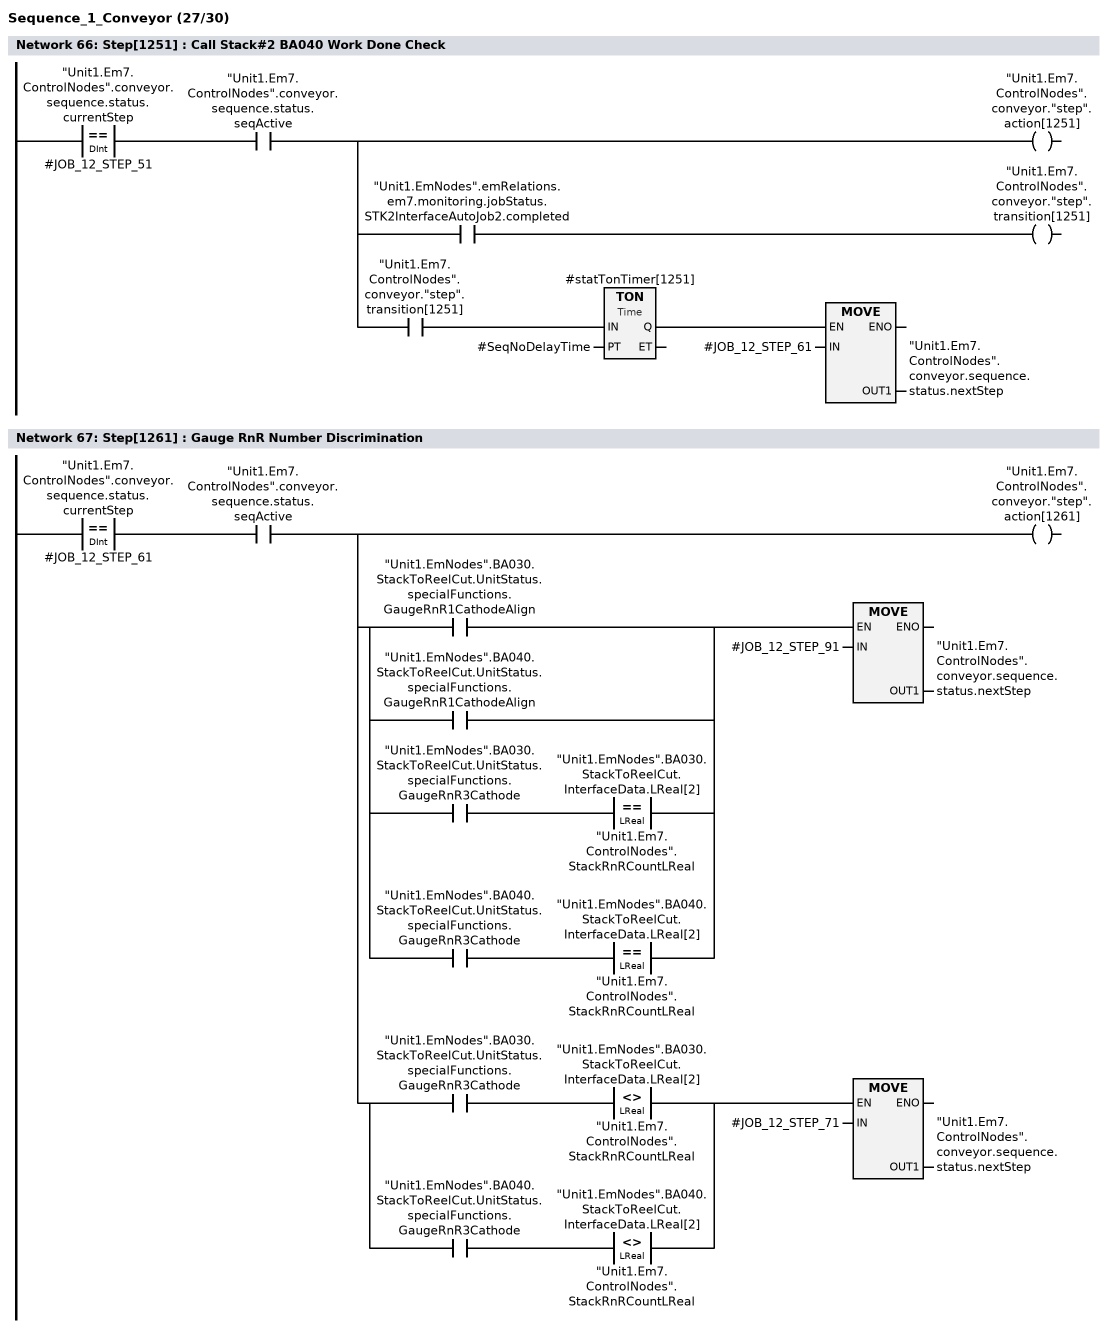
   RUNG wire#powerrail
      { S7_Templates := "SrcType := DInt" } EQ_Contact(in1 := "Unit1.Em7.ControlNodes".conveyor.sequence.status.currentStep, in2 := #JOB_12_STEP_51)
      Contact( "Unit1.Em7.ControlNodes".conveyor.sequence.status.seqActive )
      wire#w1
      Coil( "Unit1.Em7.ControlNodes".conveyor."step".action[1251] )
   END_RUNG
   RUNG wire#w1
      Contact( "Unit1.EmNodes".emRelations.em7.monitoring.jobStatus.STK2InterfaceAutoJob2.completed )
      Coil( "Unit1.Em7.ControlNodes".conveyor."step".transition[1251] )
   END_RUNG
   RUNG wire#w1
      Contact( "Unit1.Em7.ControlNodes".conveyor."step".transition[1251] )
      { S7_Templates := "time_type := Time" } #statTonTimer[1251].TON(pt := #SeqNoDelayTime, et =>)
      Move(in := #JOB_12_STEP_61, out1 => "Unit1.Em7.ControlNodes".conveyor.sequence.status.nextStep)
   END_RUNG
   // the same network as SCL:
   "Unit1.Em7.ControlNodes".conveyor."step".action[1251] := ("Unit1.Em7.ControlNodes".conveyor.sequence.status.currentStep = #JOB_12_STEP_51) AND "Unit1.Em7.ControlNodes".conveyor.sequence.status.seqActive;
   "Unit1.Em7.ControlNodes".conveyor."step".transition[1251] := ("Unit1.Em7.ControlNodes".conveyor.sequence.status.currentStep = #JOB_12_STEP_51) AND "Unit1.Em7.ControlNodes".conveyor.sequence.status.seqActive AND "Unit1.EmNodes".emRelations.em7.monitoring.jobStatus.STK2InterfaceAutoJob2.completed;
   #statTonTimer[1251].TON(IN := ("Unit1.Em7.ControlNodes".conveyor.sequence.status.currentStep = #JOB_12_STEP_51) AND "Unit1.Em7.ControlNodes".conveyor.sequence.status.seqActive AND "Unit1.Em7.ControlNodes".conveyor."step".transition[1251],
                           PT := #SeqNoDelayTime);
   IF #statTonTimer[1251].Q THEN
       "Unit1.Em7.ControlNodes".conveyor.sequence.status.nextStep := #JOB_12_STEP_61;
   END_IF;
END_REGION

REGION Network 67: Step[1261] : Gauge RnR Number Discrimination
   RUNG wire#powerrail
      { S7_Templates := "SrcType := DInt" } EQ_Contact(in1 := "Unit1.Em7.ControlNodes".conveyor.sequence.status.currentStep, in2 := #JOB_12_STEP_61)
      Contact( "Unit1.Em7.ControlNodes".conveyor.sequence.status.seqActive )
      wire#w1
      Coil( "Unit1.Em7.ControlNodes".conveyor."step".action[1261] )
   END_RUNG
   RUNG wire#w1
      Contact( "Unit1.EmNodes".BA030.StackToReelCut.UnitStatus.specialFunctions.GaugeRnR1CathodeAlign )
      wire#w2
      Move(in := #JOB_12_STEP_91, out1 => "Unit1.Em7.ControlNodes".conveyor.sequence.status.nextStep)
   END_RUNG
   RUNG wire#w1
      Contact( "Unit1.EmNodes".BA040.StackToReelCut.UnitStatus.specialFunctions.GaugeRnR1CathodeAlign )
   END_RUNG wire#w2
   RUNG wire#w1
      Contact( "Unit1.EmNodes".BA030.StackToReelCut.UnitStatus.specialFunctions.GaugeRnR3Cathode )
      { S7_Templates := "SrcType := LReal" } EQ_Contact(in1 := "Unit1.EmNodes".BA030.StackToReelCut.InterfaceData.LReal[2], in2 := "Unit1.Em7.ControlNodes".StackRnRCountLReal)
   END_RUNG wire#w2
   RUNG wire#w1
      Contact( "Unit1.EmNodes".BA040.StackToReelCut.UnitStatus.specialFunctions.GaugeRnR3Cathode )
      { S7_Templates := "SrcType := LReal" } EQ_Contact(in1 := "Unit1.EmNodes".BA040.StackToReelCut.InterfaceData.LReal[2], in2 := "Unit1.Em7.ControlNodes".StackRnRCountLReal)
   END_RUNG wire#w2
   RUNG wire#w1
      Contact( "Unit1.EmNodes".BA030.StackToReelCut.UnitStatus.specialFunctions.GaugeRnR3Cathode )
      { S7_Templates := "SrcType := LReal" } NE_Contact(in1 := "Unit1.EmNodes".BA030.StackToReelCut.InterfaceData.LReal[2], in2 := "Unit1.Em7.ControlNodes".StackRnRCountLReal)
      wire#w3
      Move(in := #JOB_12_STEP_71, out1 => "Unit1.Em7.ControlNodes".conveyor.sequence.status.nextStep)
   END_RUNG
   RUNG wire#w1
      Contact( "Unit1.EmNodes".BA040.StackToReelCut.UnitStatus.specialFunctions.GaugeRnR3Cathode )
      { S7_Templates := "SrcType := LReal" } NE_Contact(in1 := "Unit1.EmNodes".BA040.StackToReelCut.InterfaceData.LReal[2], in2 := "Unit1.Em7.ControlNodes".StackRnRCountLReal)
   END_RUNG wire#w3
   // the same network as SCL:
   "Unit1.Em7.ControlNodes".conveyor."step".action[1261] := ("Unit1.Em7.ControlNodes".conveyor.sequence.status.currentStep = #JOB_12_STEP_61) AND "Unit1.Em7.ControlNodes".conveyor.sequence.status.seqActive;
   IF ("Unit1.Em7.ControlNodes".conveyor.sequence.status.currentStep = #JOB_12_STEP_61) AND "Unit1.Em7.ControlNodes".conveyor.sequence.status.seqActive AND ("Unit1.EmNodes".BA030.StackToReelCut.UnitStatus.specialFunctions.GaugeRnR1CathodeAlign OR "Unit1.EmNodes".BA040.StackToReelCut.UnitStatus.specialFunctions.GaugeRnR1CathodeAlign OR ("Unit1.EmNodes".BA030.StackToReelCut.UnitStatus.specialFunctions.GaugeRnR3Cathode AND ("Unit1.EmNodes".BA030.StackToReelCut.InterfaceData.LReal[2] = "Unit1.Em7.ControlNodes".StackRnRCountLReal)) OR ("Unit1.EmNodes".BA040.StackToReelCut.UnitStatus.specialFunctions.GaugeRnR3Cathode AND ("Unit1.EmNodes".BA040.StackToReelCut.InterfaceData.LReal[2] = "Unit1.Em7.ControlNodes".StackRnRCountLReal))) THEN
       "Unit1.Em7.ControlNodes".conveyor.sequence.status.nextStep := #JOB_12_STEP_91;
   END_IF;
   IF ("Unit1.Em7.ControlNodes".conveyor.sequence.status.currentStep = #JOB_12_STEP_61) AND "Unit1.Em7.ControlNodes".conveyor.sequence.status.seqActive AND (("Unit1.EmNodes".BA030.StackToReelCut.UnitStatus.specialFunctions.GaugeRnR3Cathode AND ("Unit1.EmNodes".BA030.StackToReelCut.InterfaceData.LReal[2] <> "Unit1.Em7.ControlNodes".StackRnRCountLReal)) OR ("Unit1.EmNodes".BA040.StackToReelCut.UnitStatus.specialFunctions.GaugeRnR3Cathode AND ("Unit1.EmNodes".BA040.StackToReelCut.InterfaceData.LReal[2] <> "Unit1.Em7.ControlNodes".StackRnRCountLReal))) THEN
       "Unit1.Em7.ControlNodes".conveyor.sequence.status.nextStep := #JOB_12_STEP_71;
   END_IF;
END_REGION

REGION Network 68: Step[1271] : GaugeRnR3 Loading Request
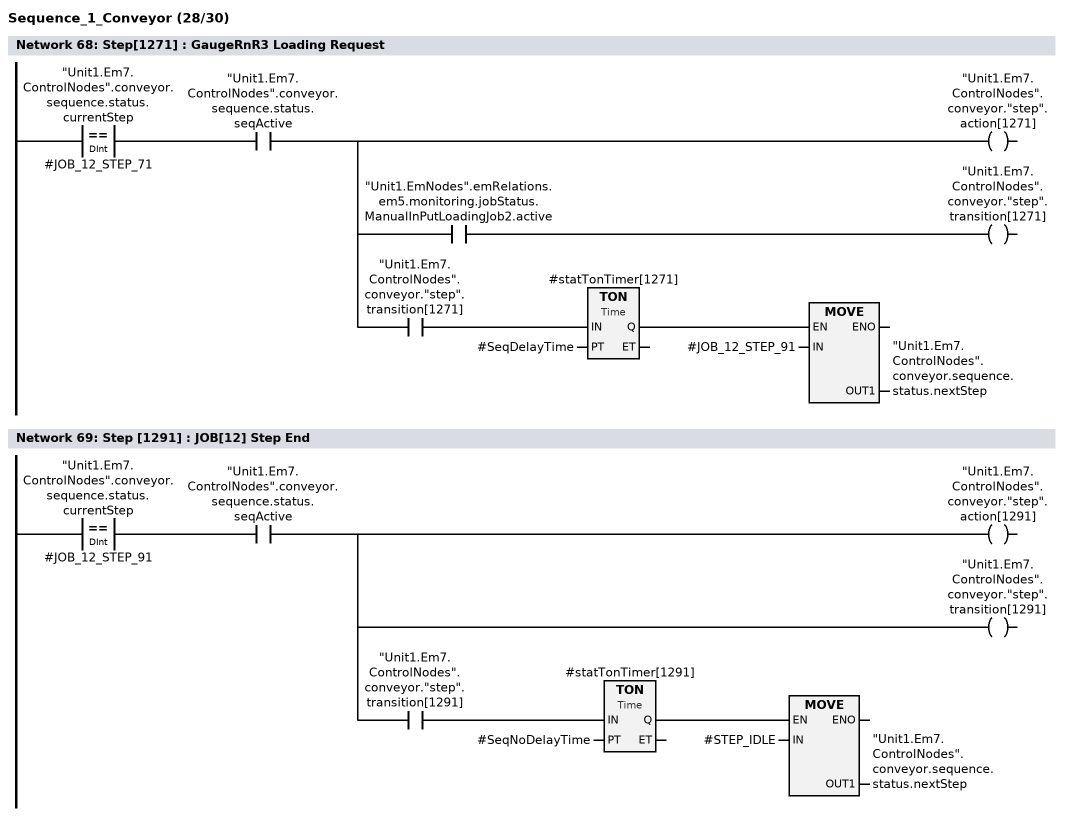
   RUNG wire#powerrail
      { S7_Templates := "SrcType := DInt" } EQ_Contact(in1 := "Unit1.Em7.ControlNodes".conveyor.sequence.status.currentStep, in2 := #JOB_12_STEP_71)
      Contact( "Unit1.Em7.ControlNodes".conveyor.sequence.status.seqActive )
      wire#w1
      Coil( "Unit1.Em7.ControlNodes".conveyor."step".action[1271] )
   END_RUNG
   RUNG wire#w1
      Contact( "Unit1.EmNodes".emRelations.em5.monitoring.jobStatus.ManualInPutLoadingJob2.active )
      Coil( "Unit1.Em7.ControlNodes".conveyor."step".transition[1271] )
   END_RUNG
   RUNG wire#w1
      Contact( "Unit1.Em7.ControlNodes".conveyor."step".transition[1271] )
      { S7_Templates := "time_type := Time" } #statTonTimer[1271].TON(pt := #SeqDelayTime, et =>)
      Move(in := #JOB_12_STEP_91, out1 => "Unit1.Em7.ControlNodes".conveyor.sequence.status.nextStep)
   END_RUNG
   // the same network as SCL:
   "Unit1.Em7.ControlNodes".conveyor."step".action[1271] := ("Unit1.Em7.ControlNodes".conveyor.sequence.status.currentStep = #JOB_12_STEP_71) AND "Unit1.Em7.ControlNodes".conveyor.sequence.status.seqActive;
   "Unit1.Em7.ControlNodes".conveyor."step".transition[1271] := ("Unit1.Em7.ControlNodes".conveyor.sequence.status.currentStep = #JOB_12_STEP_71) AND "Unit1.Em7.ControlNodes".conveyor.sequence.status.seqActive AND "Unit1.EmNodes".emRelations.em5.monitoring.jobStatus.ManualInPutLoadingJob2.active;
   #statTonTimer[1271].TON(IN := ("Unit1.Em7.ControlNodes".conveyor.sequence.status.currentStep = #JOB_12_STEP_71) AND "Unit1.Em7.ControlNodes".conveyor.sequence.status.seqActive AND "Unit1.Em7.ControlNodes".conveyor."step".transition[1271],
                           PT := #SeqDelayTime);
   IF #statTonTimer[1271].Q THEN
       "Unit1.Em7.ControlNodes".conveyor.sequence.status.nextStep := #JOB_12_STEP_91;
   END_IF;
END_REGION

